REGION Network 26: Signal conditioning — Consolidate the auto or manual state request
   // ▀▀▀▀▀▀▀▀▀▀▀▀▀▀▀▀▀▀▀▀▀▀▀▀▀▀▀▀▀▀▀▀▀▀▀▀▀▀▀▀▀▀▀▀
   // Determine the valve state required by the automatic/manual mode selection:
   // 
   //    1.  If manual mode is active set wrkCtrlAutManOpCl to match the current manual 
   //      mode requested state (ctrl_Man_OpenClose)
   // 
   //    2.  If automatic mode is active set wrkCtrlAutManOpCl to match the current automatic 
   //      mode requested state (ctrl_Aut_OpenClose)
   // ▄▄▄▄▄▄▄▄▄▄▄▄▄▄▄▄▄▄▄▄▄▄▄▄▄▄▄▄▄▄▄▄▄▄▄▄▄▄▄▄▄▄▄▄
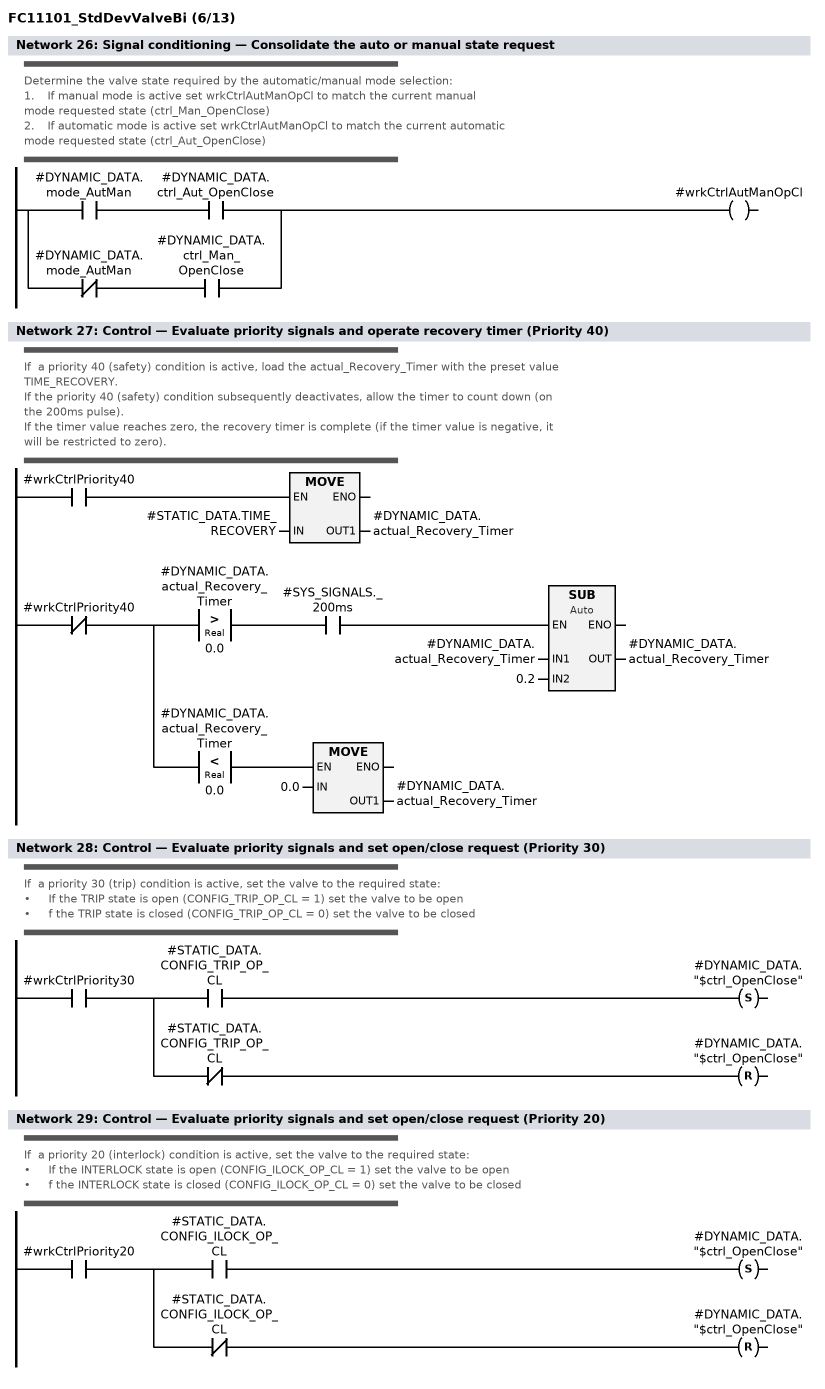
   RUNG wire#powerrail
      Contact( #DYNAMIC_DATA.mode_AutMan )
      Contact( #DYNAMIC_DATA.ctrl_Aut_OpenClose )
      wire#w1
      Coil( #wrkCtrlAutManOpCl )
   END_RUNG
   RUNG wire#powerrail
      I_Contact( #DYNAMIC_DATA.mode_AutMan )
      Contact( #DYNAMIC_DATA.ctrl_Man_OpenClose )
   END_RUNG wire#w1
   // the same network as SCL:
   #wrkCtrlAutManOpCl := (#DYNAMIC_DATA.mode_AutMan AND #DYNAMIC_DATA.ctrl_Aut_OpenClose) OR (NOT #DYNAMIC_DATA.mode_AutMan AND #DYNAMIC_DATA.ctrl_Man_OpenClose);
END_REGION

REGION Network 27: Control — Evaluate priority signals and operate recovery timer (Priority 40)
   // ▀▀▀▀▀▀▀▀▀▀▀▀▀▀▀▀▀▀▀▀▀▀▀▀▀▀▀▀▀▀▀▀▀▀▀▀▀▀▀▀▀▀▀▀
   // If  a priority 40 (safety) condition is active, load the actual_Recovery_Timer with the preset value 
   // TIME_RECOVERY.
   // 
   // If the priority 40 (safety) condition subsequently deactivates, allow the timer to count down (on 
   // the 200ms pulse).
   // 
   // If the timer value reaches zero, the recovery timer is complete (if the timer value is negative, it
   // will be restricted to zero).
   // ▄▄▄▄▄▄▄▄▄▄▄▄▄▄▄▄▄▄▄▄▄▄▄▄▄▄▄▄▄▄▄▄▄▄▄▄▄▄▄▄▄▄▄▄
   RUNG wire#powerrail
      Contact( #wrkCtrlPriority40 )
      Move(in := #STATIC_DATA.TIME_RECOVERY, out1 => #DYNAMIC_DATA.actual_Recovery_Timer)
   END_RUNG
   RUNG wire#powerrail
      I_Contact( #wrkCtrlPriority40 )
      wire#w1
      { S7_Templates := "SrcType := Real" } GT_Contact(in1 := #DYNAMIC_DATA.actual_Recovery_Timer, in2 := 0.0)
      Contact( #SYS_SIGNALS._200ms )
      Sub(in1 := #DYNAMIC_DATA.actual_Recovery_Timer, in2 := 0.2, out => #DYNAMIC_DATA.actual_Recovery_Timer)
   END_RUNG
   RUNG wire#w1
      { S7_Templates := "SrcType := Real" } LT_Contact(in1 := #DYNAMIC_DATA.actual_Recovery_Timer, in2 := 0.0)
      Move(in := 0.0, out1 => #DYNAMIC_DATA.actual_Recovery_Timer)
   END_RUNG
   // the same network as SCL:
   IF #wrkCtrlPriority40 THEN #DYNAMIC_DATA.actual_Recovery_Timer := #STATIC_DATA.TIME_RECOVERY; END_IF;
   IF NOT #wrkCtrlPriority40 AND (#DYNAMIC_DATA.actual_Recovery_Timer > 0.0) AND #SYS_SIGNALS._200ms THEN
       #DYNAMIC_DATA.actual_Recovery_Timer := #DYNAMIC_DATA.actual_Recovery_Timer - 0.2;
   END_IF;
   IF NOT #wrkCtrlPriority40 AND (#DYNAMIC_DATA.actual_Recovery_Timer < 0.0) THEN
       #DYNAMIC_DATA.actual_Recovery_Timer := 0.0;
   END_IF;
END_REGION

REGION Network 28: Control — Evaluate priority signals and set open/close request (Priority 30)
   // ▀▀▀▀▀▀▀▀▀▀▀▀▀▀▀▀▀▀▀▀▀▀▀▀▀▀▀▀▀▀▀▀▀▀▀▀▀▀▀▀▀▀▀▀
   // If  a priority 30 (trip) condition is active, set the valve to the required state:
   // 
   //    •   If the TRIP state is open (CONFIG_TRIP_OP_CL = 1) set the valve to be open
   // 
   //    •   f the TRIP state is closed (CONFIG_TRIP_OP_CL = 0) set the valve to be closed
   // ▄▄▄▄▄▄▄▄▄▄▄▄▄▄▄▄▄▄▄▄▄▄▄▄▄▄▄▄▄▄▄▄▄▄▄▄▄▄▄▄▄▄▄▄
   RUNG wire#powerrail
      Contact( #wrkCtrlPriority30 )
      wire#w1
      Contact( #STATIC_DATA.CONFIG_TRIP_OP_CL )
      S_Coil( #DYNAMIC_DATA."$ctrl_OpenClose" )
   END_RUNG
   RUNG wire#w1
      I_Contact( #STATIC_DATA.CONFIG_TRIP_OP_CL )
      R_Coil( #DYNAMIC_DATA."$ctrl_OpenClose" )
   END_RUNG
   // the same network as SCL:
   IF #wrkCtrlPriority30 AND #STATIC_DATA.CONFIG_TRIP_OP_CL THEN
       #DYNAMIC_DATA."$ctrl_OpenClose" := TRUE;
   END_IF;
   IF #wrkCtrlPriority30 AND NOT #STATIC_DATA.CONFIG_TRIP_OP_CL THEN
       #DYNAMIC_DATA."$ctrl_OpenClose" := FALSE;
   END_IF;
END_REGION

REGION Network 29: Control — Evaluate priority signals and set open/close request (Priority 20)
   // ▀▀▀▀▀▀▀▀▀▀▀▀▀▀▀▀▀▀▀▀▀▀▀▀▀▀▀▀▀▀▀▀▀▀▀▀▀▀▀▀▀▀▀▀
   // If  a priority 20 (interlock) condition is active, set the valve to the required state:
   // 
   //    •   If the INTERLOCK state is open (CONFIG_ILOCK_OP_CL = 1) set the valve to be open
   // 
   //    •   f the INTERLOCK state is closed (CONFIG_ILOCK_OP_CL = 0) set the valve to be closed
   // ▄▄▄▄▄▄▄▄▄▄▄▄▄▄▄▄▄▄▄▄▄▄▄▄▄▄▄▄▄▄▄▄▄▄▄▄▄▄▄▄▄▄▄▄
   RUNG wire#powerrail
      Contact( #wrkCtrlPriority20 )
      wire#w1
      Contact( #STATIC_DATA.CONFIG_ILOCK_OP_CL )
      S_Coil( #DYNAMIC_DATA."$ctrl_OpenClose" )
   END_RUNG
   RUNG wire#w1
      I_Contact( #STATIC_DATA.CONFIG_ILOCK_OP_CL )
      R_Coil( #DYNAMIC_DATA."$ctrl_OpenClose" )
   END_RUNG
   // the same network as SCL:
   IF #wrkCtrlPriority20 AND #STATIC_DATA.CONFIG_ILOCK_OP_CL THEN
       #DYNAMIC_DATA."$ctrl_OpenClose" := TRUE;
   END_IF;
   IF #wrkCtrlPriority20 AND NOT #STATIC_DATA.CONFIG_ILOCK_OP_CL THEN
       #DYNAMIC_DATA."$ctrl_OpenClose" := FALSE;
   END_IF;
END_REGION

REGION Network 30: Control — Evaluate priority signals and set open/close request (Priority 10)
   // ▀▀▀▀▀▀▀▀▀▀▀▀▀▀▀▀▀▀▀▀▀▀▀▀▀▀▀▀▀▀▀▀▀▀▀▀▀▀▀▀▀▀▀▀
   // If  a priority 10 (permissive) condition is active, set the valve to the required state:
   // 
   // 
   // PERMITTED STATE IS OPEN — CONDITIONS:
   // 
   //    •   If the Permitted state is open and Aut/Man request is for open, 
   //      set the valve to be open [Branch 1]
   // 
   //    •   If the Permitted state is open and Aut/Man request is for closed, and the current
   //      valve output matches this state (closed), set the valve to be closed (maintain the
   //      current state) [Branch 6]
   // 
   //    •   If the Permitted state is open and Aut/Man request is for closed, and the current
   //      valve output matches the open state, set the valve to be open (override the
   //      auto/man request [Branch 2]
   // 
   // PERMITTED STATE IS CLOSED — CONDITIONS:
   // 
   //    •   If the Permitted state is closed and Aut/Man request is for closed,
   //      set the valve to be  closed [Branch 4]
   // 
   //    •   If the Permitted state is closed and Aut/Man request is for open, and the current
   //      valve output matches this state (open), set the valve to be open (maintain the
   //      current state) [Branch 3]
   // 
   //    •   If the Permitted state is closed and Aut/Man request is for open, and the current
   //      valve output matches the closed state, set the valve to be closed (override the
   //      auto/man request [Branch 5]
   // ▄▄▄▄▄▄▄▄▄▄▄▄▄▄▄▄▄▄▄▄▄▄▄▄▄▄▄▄▄▄▄▄▄▄▄▄▄▄▄▄▄▄▄▄
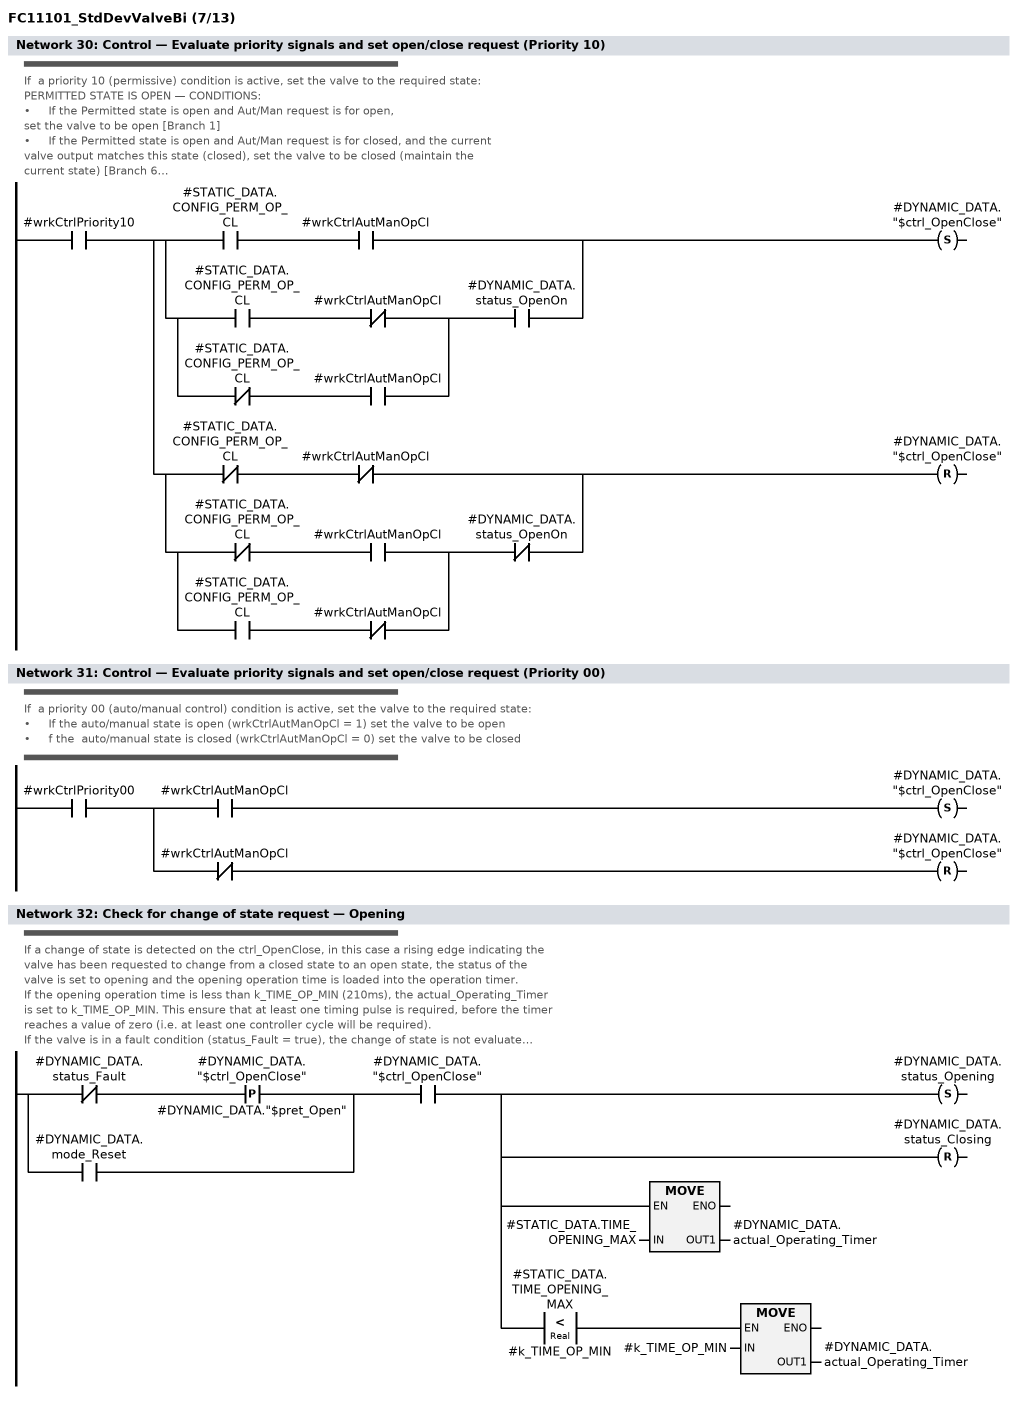
   RUNG wire#powerrail
      Contact( #wrkCtrlPriority10 )
      wire#w1
      Contact( #STATIC_DATA.CONFIG_PERM_OP_CL )
      Contact( #wrkCtrlAutManOpCl )
      wire#w2
      S_Coil( #DYNAMIC_DATA."$ctrl_OpenClose" )
   END_RUNG
   RUNG wire#w1
      Contact( #STATIC_DATA.CONFIG_PERM_OP_CL )
      I_Contact( #wrkCtrlAutManOpCl )
      wire#w3
      Contact( #DYNAMIC_DATA.status_OpenOn )
   END_RUNG wire#w2
   RUNG wire#w1
      I_Contact( #STATIC_DATA.CONFIG_PERM_OP_CL )
      Contact( #wrkCtrlAutManOpCl )
   END_RUNG wire#w3
   RUNG wire#w1
      I_Contact( #STATIC_DATA.CONFIG_PERM_OP_CL )
      I_Contact( #wrkCtrlAutManOpCl )
      wire#w4
      R_Coil( #DYNAMIC_DATA."$ctrl_OpenClose" )
   END_RUNG
   RUNG wire#w1
      I_Contact( #STATIC_DATA.CONFIG_PERM_OP_CL )
      Contact( #wrkCtrlAutManOpCl )
      wire#w5
      I_Contact( #DYNAMIC_DATA.status_OpenOn )
   END_RUNG wire#w4
   RUNG wire#w1
      Contact( #STATIC_DATA.CONFIG_PERM_OP_CL )
      I_Contact( #wrkCtrlAutManOpCl )
   END_RUNG wire#w5
   // the same network as SCL:
   IF #wrkCtrlPriority10 AND ((#STATIC_DATA.CONFIG_PERM_OP_CL AND #wrkCtrlAutManOpCl) OR (((#STATIC_DATA.CONFIG_PERM_OP_CL AND NOT #wrkCtrlAutManOpCl) OR (NOT #STATIC_DATA.CONFIG_PERM_OP_CL AND #wrkCtrlAutManOpCl)) AND #DYNAMIC_DATA.status_OpenOn)) THEN
       #DYNAMIC_DATA."$ctrl_OpenClose" := TRUE;
   END_IF;
   IF #wrkCtrlPriority10 AND ((NOT #STATIC_DATA.CONFIG_PERM_OP_CL AND NOT #wrkCtrlAutManOpCl) OR (((NOT #STATIC_DATA.CONFIG_PERM_OP_CL AND #wrkCtrlAutManOpCl) OR (#STATIC_DATA.CONFIG_PERM_OP_CL AND NOT #wrkCtrlAutManOpCl)) AND NOT #DYNAMIC_DATA.status_OpenOn)) THEN
       #DYNAMIC_DATA."$ctrl_OpenClose" := FALSE;
   END_IF;
END_REGION

REGION Network 31: Control — Evaluate priority signals and set open/close request (Priority 00)
   // ▀▀▀▀▀▀▀▀▀▀▀▀▀▀▀▀▀▀▀▀▀▀▀▀▀▀▀▀▀▀▀▀▀▀▀▀▀▀▀▀▀▀▀▀
   // If  a priority 00 (auto/manual control) condition is active, set the valve to the required state:
   // 
   //    •   If the auto/manual state is open (wrkCtrlAutManOpCl = 1) set the valve to be open
   // 
   //    •   f the  auto/manual state is closed (wrkCtrlAutManOpCl = 0) set the valve to be closed
   // ▄▄▄▄▄▄▄▄▄▄▄▄▄▄▄▄▄▄▄▄▄▄▄▄▄▄▄▄▄▄▄▄▄▄▄▄▄▄▄▄▄▄▄▄
   RUNG wire#powerrail
      Contact( #wrkCtrlPriority00 )
      wire#w1
      Contact( #wrkCtrlAutManOpCl )
      S_Coil( #DYNAMIC_DATA."$ctrl_OpenClose" )
   END_RUNG
   RUNG wire#w1
      I_Contact( #wrkCtrlAutManOpCl )
      R_Coil( #DYNAMIC_DATA."$ctrl_OpenClose" )
   END_RUNG
   // the same network as SCL:
   IF #wrkCtrlPriority00 AND #wrkCtrlAutManOpCl THEN #DYNAMIC_DATA."$ctrl_OpenClose" := TRUE; END_IF;
   IF #wrkCtrlPriority00 AND NOT #wrkCtrlAutManOpCl THEN #DYNAMIC_DATA."$ctrl_OpenClose" := FALSE; END_IF;
END_REGION

REGION Network 32: Check for change of state request — Opening
   // ▀▀▀▀▀▀▀▀▀▀▀▀▀▀▀▀▀▀▀▀▀▀▀▀▀▀▀▀▀▀▀▀▀▀▀▀▀▀▀▀▀▀▀▀
   // If a change of state is detected on the ctrl_OpenClose, in this case a rising edge indicating the
   // valve has been requested to change from a closed state to an open state, the status of the
   // valve is set to opening and the opening operation time is loaded into the operation timer.
   // 
   // If the opening operation time is less than k_TIME_OP_MIN (210ms), the actual_Operating_Timer 
   // is set to k_TIME_OP_MIN. This ensure that at least one timing pulse is required, before the timer 
   // reaches a value of zero (i.e. at least one controller cycle will be required).
   // 
   // If the valve is in a fault condition (status_Fault = true), the change of state is not evaluated
   // until the fault condition has cleared
   // 
   // Note: the timer is also triggered if the Reset signal is received and the valve is requested open.
   // ▄▄▄▄▄▄▄▄▄▄▄▄▄▄▄▄▄▄▄▄▄▄▄▄▄▄▄▄▄▄▄▄▄▄▄▄▄▄▄▄▄▄▄▄
   RUNG wire#powerrail
      I_Contact( #DYNAMIC_DATA.status_Fault )
      P_Contact(operand := #DYNAMIC_DATA."$ctrl_OpenClose", bit := #DYNAMIC_DATA."$pret_Open")
      wire#w1
      Contact( #DYNAMIC_DATA."$ctrl_OpenClose" )
      wire#w2
      S_Coil( #DYNAMIC_DATA.status_Opening )
   END_RUNG
   RUNG wire#powerrail
      Contact( #DYNAMIC_DATA.mode_Reset )
   END_RUNG wire#w1
   RUNG wire#w2
      R_Coil( #DYNAMIC_DATA.status_Closing )
   END_RUNG
   RUNG wire#w2
      Move(in := #STATIC_DATA.TIME_OPENING_MAX, out1 => #DYNAMIC_DATA.actual_Operating_Timer)
   END_RUNG
   RUNG wire#w2
      { S7_Templates := "SrcType := Real" } LT_Contact(in1 := #STATIC_DATA.TIME_OPENING_MAX, in2 := #k_TIME_OP_MIN)
      Move(in := #k_TIME_OP_MIN, out1 => #DYNAMIC_DATA.actual_Operating_Timer)
   END_RUNG
   // the same network as SCL:
   #_w1 := NOT #DYNAMIC_DATA.status_Fault AND #DYNAMIC_DATA."$ctrl_OpenClose" AND NOT #DYNAMIC_DATA."$pret_Open";   // rising edge of #DYNAMIC_DATA."$ctrl_OpenClose"
   #DYNAMIC_DATA."$pret_Open" := #DYNAMIC_DATA."$ctrl_OpenClose";
   #_w2 := (#_w1 OR #DYNAMIC_DATA.mode_Reset) AND #DYNAMIC_DATA."$ctrl_OpenClose";
   IF #_w2 THEN
       #DYNAMIC_DATA.status_Opening := TRUE;
       #DYNAMIC_DATA.status_Closing := FALSE;
       #DYNAMIC_DATA.actual_Operating_Timer := #STATIC_DATA.TIME_OPENING_MAX;
   END_IF;
   IF #_w2 AND (#STATIC_DATA.TIME_OPENING_MAX < #k_TIME_OP_MIN) THEN
       #DYNAMIC_DATA.actual_Operating_Timer := #k_TIME_OP_MIN;
   END_IF;
END_REGION

REGION Network 33: Check for change of state request — Closing
   // ▀▀▀▀▀▀▀▀▀▀▀▀▀▀▀▀▀▀▀▀▀▀▀▀▀▀▀▀▀▀▀▀▀▀▀▀▀▀▀▀▀▀▀▀
   // If a change of state is detected on the ctrl_OpenClose, in this case a falling edge indicating the
   // valve has been requested to change from an open state to a closed state, the status of the
   // valve is set to closing and the closing operation time is loaded into the operation timer.
   // 
   // If the closing operation time is less than k_TIME_OP_MIN (210ms), the actual_Operating_Timer 
   // is set to k_TIME_OP_MIN. This ensure that at least one timing pulse is required, before the timer 
   // reaches a value of zero (i.e. at least one controller cycle will be required).
   // 
   // If the valve is in a fault condition (status_Fault = true), the change of state is not evaluated
   // until the fault condition has cleared
   // 
   // Note: the timer is also triggered if the Reset signal is received and the valve is requested closed.
   // ▄▄▄▄▄▄▄▄▄▄▄▄▄▄▄▄▄▄▄▄▄▄▄▄▄▄▄▄▄▄▄▄▄▄▄▄▄▄▄▄▄▄▄▄
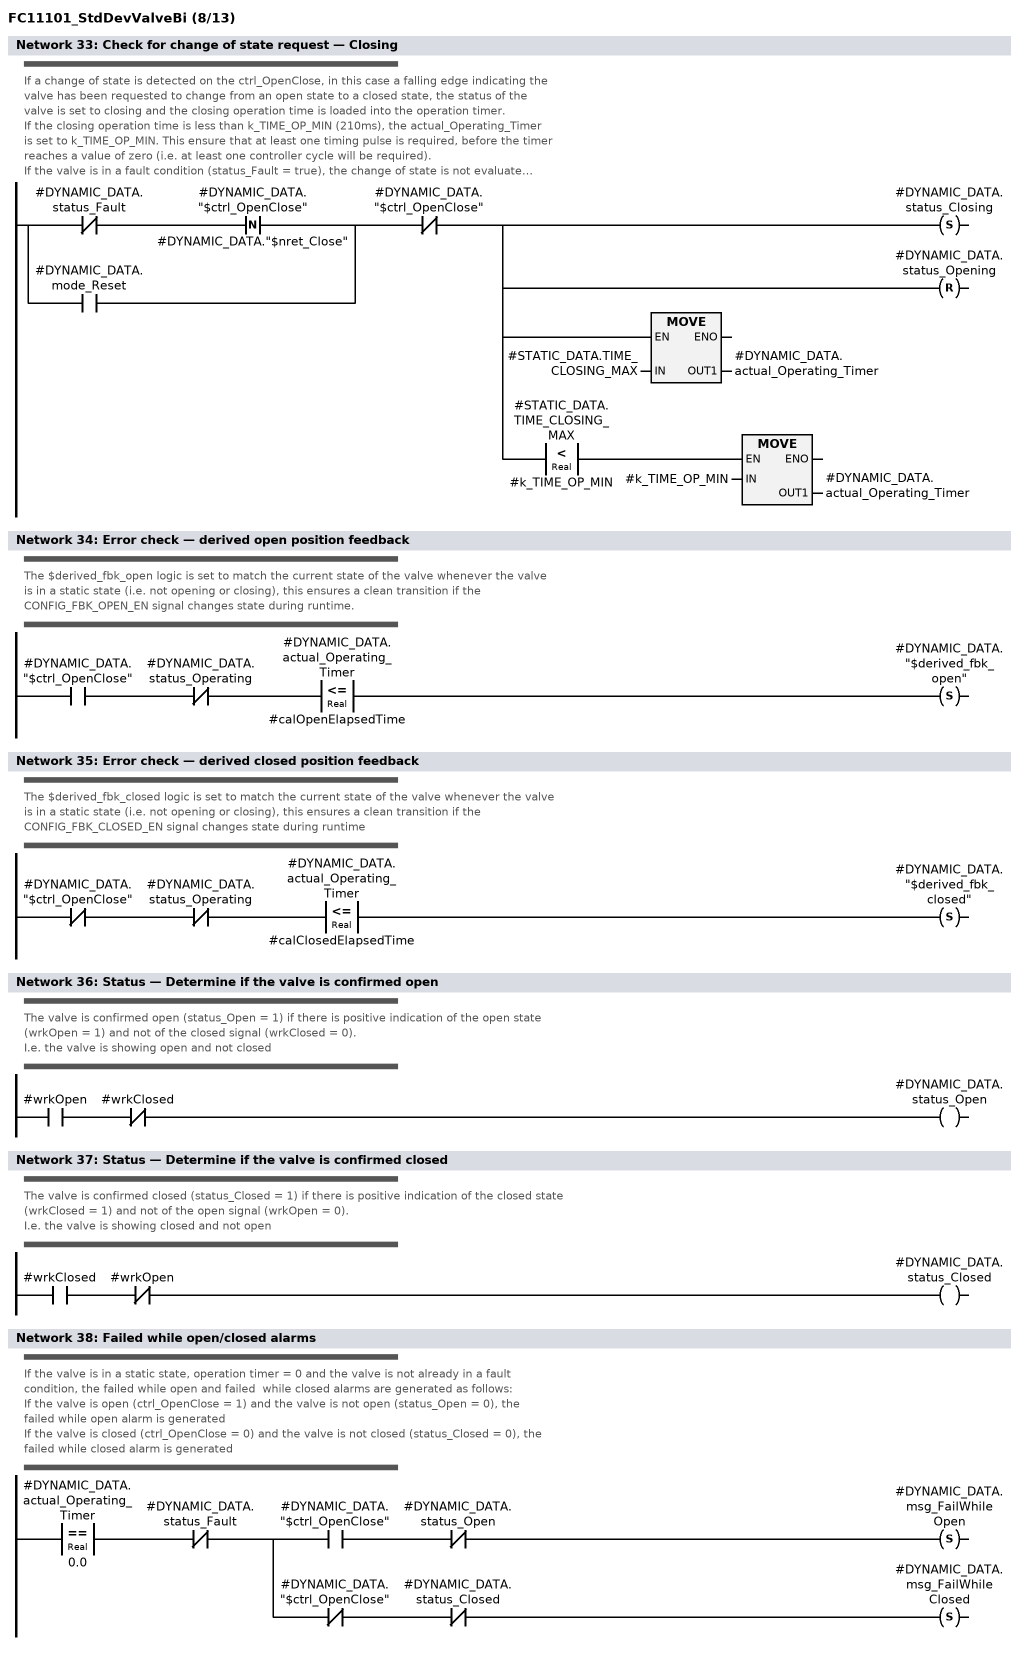
   RUNG wire#powerrail
      I_Contact( #DYNAMIC_DATA.status_Fault )
      N_Contact(operand := #DYNAMIC_DATA."$ctrl_OpenClose", bit := #DYNAMIC_DATA."$nret_Close")
      wire#w1
      I_Contact( #DYNAMIC_DATA."$ctrl_OpenClose" )
      wire#w2
      S_Coil( #DYNAMIC_DATA.status_Closing )
   END_RUNG
   RUNG wire#powerrail
      Contact( #DYNAMIC_DATA.mode_Reset )
   END_RUNG wire#w1
   RUNG wire#w2
      R_Coil( #DYNAMIC_DATA.status_Opening )
   END_RUNG
   RUNG wire#w2
      Move(in := #STATIC_DATA.TIME_CLOSING_MAX, out1 => #DYNAMIC_DATA.actual_Operating_Timer)
   END_RUNG
   RUNG wire#w2
      { S7_Templates := "SrcType := Real" } LT_Contact(in1 := #STATIC_DATA.TIME_CLOSING_MAX, in2 := #k_TIME_OP_MIN)
      Move(in := #k_TIME_OP_MIN, out1 => #DYNAMIC_DATA.actual_Operating_Timer)
   END_RUNG
   // the same network as SCL:
   #_w1 := NOT #DYNAMIC_DATA.status_Fault AND NOT #DYNAMIC_DATA."$ctrl_OpenClose" AND #DYNAMIC_DATA."$nret_Close";   // falling edge of #DYNAMIC_DATA."$ctrl_OpenClose"
   #DYNAMIC_DATA."$nret_Close" := #DYNAMIC_DATA."$ctrl_OpenClose";
   #_w2 := (#_w1 OR #DYNAMIC_DATA.mode_Reset) AND NOT #DYNAMIC_DATA."$ctrl_OpenClose";
   IF #_w2 THEN
       #DYNAMIC_DATA.status_Closing := TRUE;
       #DYNAMIC_DATA.status_Opening := FALSE;
       #DYNAMIC_DATA.actual_Operating_Timer := #STATIC_DATA.TIME_CLOSING_MAX;
   END_IF;
   IF #_w2 AND (#STATIC_DATA.TIME_CLOSING_MAX < #k_TIME_OP_MIN) THEN
       #DYNAMIC_DATA.actual_Operating_Timer := #k_TIME_OP_MIN;
   END_IF;
END_REGION

REGION Network 34: Error check — derived open position feedback
   // ▀▀▀▀▀▀▀▀▀▀▀▀▀▀▀▀▀▀▀▀▀▀▀▀▀▀▀▀▀▀▀▀▀▀▀▀▀▀▀▀▀▀▀▀
   // The $derived_fbk_open logic is set to match the current state of the valve whenever the valve
   // is in a static state (i.e. not opening or closing), this ensures a clean transition if the 
   // CONFIG_FBK_OPEN_EN signal changes state during runtime.
   // ▄▄▄▄▄▄▄▄▄▄▄▄▄▄▄▄▄▄▄▄▄▄▄▄▄▄▄▄▄▄▄▄▄▄▄▄▄▄▄▄▄▄▄▄
   RUNG wire#powerrail
      Contact( #DYNAMIC_DATA."$ctrl_OpenClose" )
      I_Contact( #DYNAMIC_DATA.status_Operating )
      { S7_Templates := "SrcType := Real" } LE_Contact(in1 := #DYNAMIC_DATA.actual_Operating_Timer, in2 := #calOpenElapsedTime)
      S_Coil( #DYNAMIC_DATA."$derived_fbk_open" )
   END_RUNG
   // the same network as SCL:
   IF #DYNAMIC_DATA."$ctrl_OpenClose" AND NOT #DYNAMIC_DATA.status_Operating AND (#DYNAMIC_DATA.actual_Operating_Timer <= #calOpenElapsedTime) THEN
       #DYNAMIC_DATA."$derived_fbk_open" := TRUE;
   END_IF;
END_REGION

REGION Network 35: Error check — derived closed position feedback
   // ▀▀▀▀▀▀▀▀▀▀▀▀▀▀▀▀▀▀▀▀▀▀▀▀▀▀▀▀▀▀▀▀▀▀▀▀▀▀▀▀▀▀▀▀
   // The $derived_fbk_closed logic is set to match the current state of the valve whenever the valve
   // is in a static state (i.e. not opening or closing), this ensures a clean transition if the 
   // CONFIG_FBK_CLOSED_EN signal changes state during runtime
   // ▄▄▄▄▄▄▄▄▄▄▄▄▄▄▄▄▄▄▄▄▄▄▄▄▄▄▄▄▄▄▄▄▄▄▄▄▄▄▄▄▄▄▄▄
   RUNG wire#powerrail
      I_Contact( #DYNAMIC_DATA."$ctrl_OpenClose" )
      I_Contact( #DYNAMIC_DATA.status_Operating )
      { S7_Templates := "SrcType := Real" } LE_Contact(in1 := #DYNAMIC_DATA.actual_Operating_Timer, in2 := #calClosedElapsedTime)
      S_Coil( #DYNAMIC_DATA."$derived_fbk_closed" )
   END_RUNG
   // the same network as SCL:
   IF NOT #DYNAMIC_DATA."$ctrl_OpenClose" AND NOT #DYNAMIC_DATA.status_Operating AND (#DYNAMIC_DATA.actual_Operating_Timer <= #calClosedElapsedTime) THEN
       #DYNAMIC_DATA."$derived_fbk_closed" := TRUE;
   END_IF;
END_REGION

REGION Network 36: Status — Determine if the valve is confirmed open
   // ▀▀▀▀▀▀▀▀▀▀▀▀▀▀▀▀▀▀▀▀▀▀▀▀▀▀▀▀▀▀▀▀▀▀▀▀▀▀▀▀▀▀▀▀
   // The valve is confirmed open (status_Open = 1) if there is positive indication of the open state 
   // (wrkOpen = 1) and not of the closed signal (wrkClosed = 0). 
   // 
   // I.e. the valve is showing open and not closed
   // ▄▄▄▄▄▄▄▄▄▄▄▄▄▄▄▄▄▄▄▄▄▄▄▄▄▄▄▄▄▄▄▄▄▄▄▄▄▄▄▄▄▄▄▄
   RUNG wire#powerrail
      Contact( #wrkOpen )
      I_Contact( #wrkClosed )
      Coil( #DYNAMIC_DATA.status_Open )
   END_RUNG
   // the same network as SCL:
   #DYNAMIC_DATA.status_Open := #wrkOpen AND NOT #wrkClosed;
END_REGION

REGION Network 37: Status — Determine if the valve is confirmed closed
   // ▀▀▀▀▀▀▀▀▀▀▀▀▀▀▀▀▀▀▀▀▀▀▀▀▀▀▀▀▀▀▀▀▀▀▀▀▀▀▀▀▀▀▀▀
   // The valve is confirmed closed (status_Closed = 1) if there is positive indication of the closed state 
   // (wrkClosed = 1) and not of the open signal (wrkOpen = 0). 
   // 
   // I.e. the valve is showing closed and not open
   // ▄▄▄▄▄▄▄▄▄▄▄▄▄▄▄▄▄▄▄▄▄▄▄▄▄▄▄▄▄▄▄▄▄▄▄▄▄▄▄▄▄▄▄▄
   RUNG wire#powerrail
      Contact( #wrkClosed )
      I_Contact( #wrkOpen )
      Coil( #DYNAMIC_DATA.status_Closed )
   END_RUNG
   // the same network as SCL:
   #DYNAMIC_DATA.status_Closed := #wrkClosed AND NOT #wrkOpen;
END_REGION

REGION Network 38: Failed while open/closed alarms
   // ▀▀▀▀▀▀▀▀▀▀▀▀▀▀▀▀▀▀▀▀▀▀▀▀▀▀▀▀▀▀▀▀▀▀▀▀▀▀▀▀▀▀▀▀
   // If the valve is in a static state, operation timer = 0 and the valve is not already in a fault
   // condition, the failed while open and failed  while closed alarms are generated as follows:
   // 
   // If the valve is open (ctrl_OpenClose = 1) and the valve is not open (status_Open = 0), the 
   // failed while open alarm is generated
   // 
   // If the valve is closed (ctrl_OpenClose = 0) and the valve is not closed (status_Closed = 0), the 
   // failed while closed alarm is generated
   // ▄▄▄▄▄▄▄▄▄▄▄▄▄▄▄▄▄▄▄▄▄▄▄▄▄▄▄▄▄▄▄▄▄▄▄▄▄▄▄▄▄▄▄▄
   RUNG wire#powerrail
      { S7_Templates := "SrcType := Real" } EQ_Contact(in1 := #DYNAMIC_DATA.actual_Operating_Timer, in2 := 0.0)
      I_Contact( #DYNAMIC_DATA.status_Fault )
      wire#w1
      Contact( #DYNAMIC_DATA."$ctrl_OpenClose" )
      I_Contact( #DYNAMIC_DATA.status_Open )
      S_Coil( #DYNAMIC_DATA.msg_FailWhileOpen )
   END_RUNG
   RUNG wire#w1
      I_Contact( #DYNAMIC_DATA."$ctrl_OpenClose" )
      I_Contact( #DYNAMIC_DATA.status_Closed )
      S_Coil( #DYNAMIC_DATA.msg_FailWhileClosed )
   END_RUNG
   // the same network as SCL:
   #_w1 := (#DYNAMIC_DATA.actual_Operating_Timer = 0.0) AND NOT #DYNAMIC_DATA.status_Fault;
   IF #_w1 AND #DYNAMIC_DATA."$ctrl_OpenClose" AND NOT #DYNAMIC_DATA.status_Open THEN
       #DYNAMIC_DATA.msg_FailWhileOpen := TRUE;
   END_IF;
   IF #_w1 AND NOT #DYNAMIC_DATA."$ctrl_OpenClose" AND NOT #DYNAMIC_DATA.status_Closed THEN
       #DYNAMIC_DATA.msg_FailWhileClosed := TRUE;
   END_IF;
END_REGION

REGION Network 39: Operation timer and Failed to open/close alarms
   // ▀▀▀▀▀▀▀▀▀▀▀▀▀▀▀▀▀▀▀▀▀▀▀▀▀▀▀▀▀▀▀▀▀▀▀▀▀▀▀▀▀▀▀▀
   // If the valve is opening or closing, decrement the current operation timer value on each 200ms
   // pulse.
   // 
   // If the timer reaches zero, and the valve is opening, generate the failed to open alarm.
   // 
   // If the timer reaches zero, and the valve is closing, generate the failed to close alarm
   // ▄▄▄▄▄▄▄▄▄▄▄▄▄▄▄▄▄▄▄▄▄▄▄▄▄▄▄▄▄▄▄▄▄▄▄▄▄▄▄▄▄▄▄▄
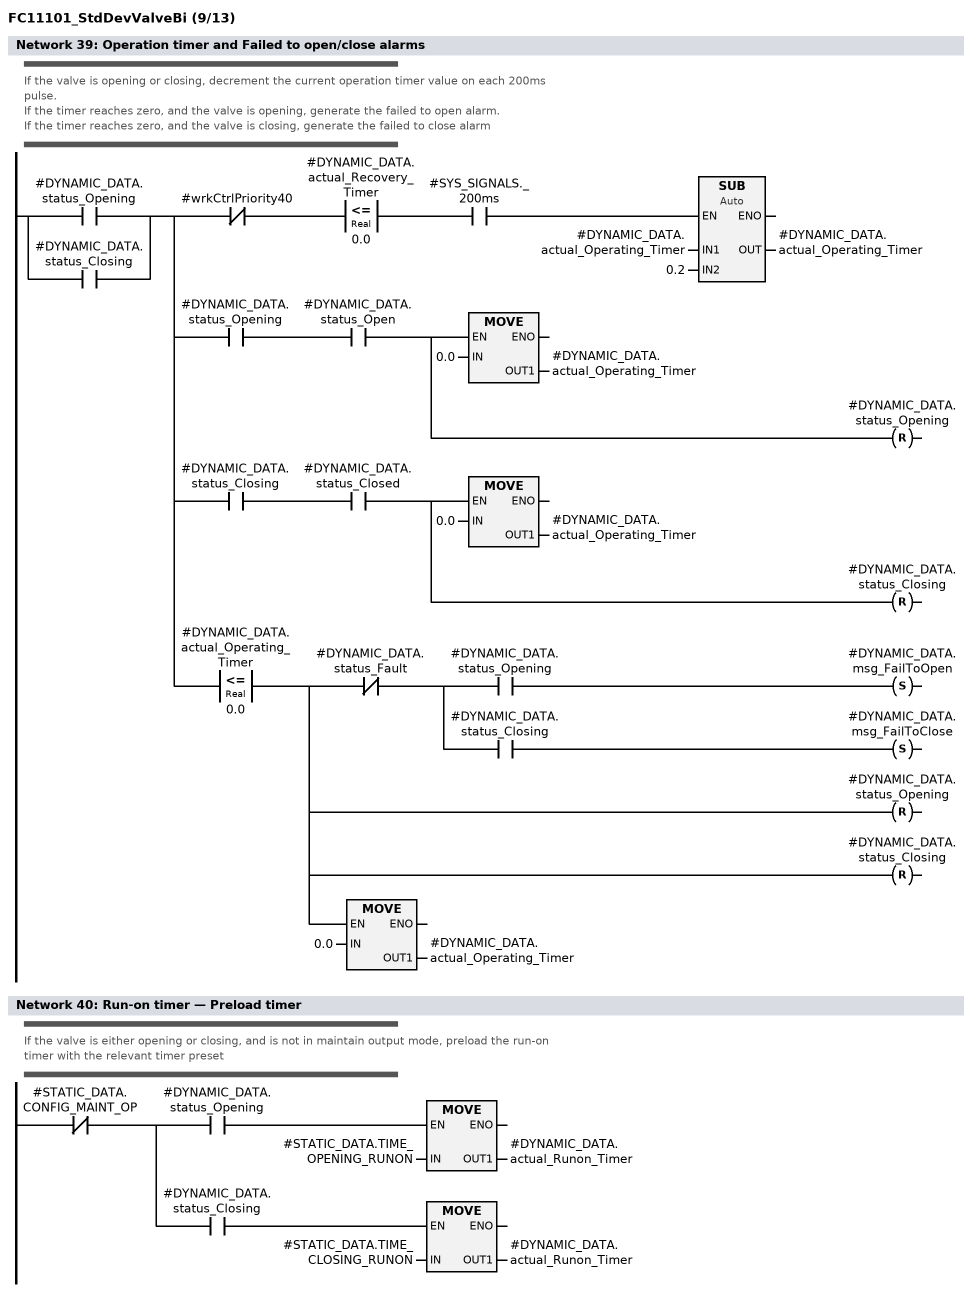
   RUNG wire#powerrail
      Contact( #DYNAMIC_DATA.status_Opening )
      wire#w1
      I_Contact( #wrkCtrlPriority40 )
      { S7_Templates := "SrcType := Real" } LE_Contact(in1 := #DYNAMIC_DATA.actual_Recovery_Timer, in2 := 0.0)
      Contact( #SYS_SIGNALS._200ms )
      Sub(in1 := #DYNAMIC_DATA.actual_Operating_Timer, in2 := 0.2, out => #DYNAMIC_DATA.actual_Operating_Timer)
   END_RUNG
   RUNG wire#powerrail
      Contact( #DYNAMIC_DATA.status_Closing )
   END_RUNG wire#w1
   RUNG wire#w1
      Contact( #DYNAMIC_DATA.status_Opening )
      Contact( #DYNAMIC_DATA.status_Open )
      wire#w2
      Move(in := 0.0, out1 => #DYNAMIC_DATA.actual_Operating_Timer)
   END_RUNG
   RUNG wire#w2
      R_Coil( #DYNAMIC_DATA.status_Opening )
   END_RUNG
   RUNG wire#w1
      Contact( #DYNAMIC_DATA.status_Closing )
      Contact( #DYNAMIC_DATA.status_Closed )
      wire#w3
      Move(in := 0.0, out1 => #DYNAMIC_DATA.actual_Operating_Timer)
   END_RUNG
   RUNG wire#w3
      R_Coil( #DYNAMIC_DATA.status_Closing )
   END_RUNG
   RUNG wire#w1
      { S7_Templates := "SrcType := Real" } LE_Contact(in1 := #DYNAMIC_DATA.actual_Operating_Timer, in2 := 0.0)
      wire#w4
      I_Contact( #DYNAMIC_DATA.status_Fault )
      wire#w5
      Contact( #DYNAMIC_DATA.status_Opening )
      S_Coil( #DYNAMIC_DATA.msg_FailToOpen )
   END_RUNG
   RUNG wire#w5
      Contact( #DYNAMIC_DATA.status_Closing )
      S_Coil( #DYNAMIC_DATA.msg_FailToClose )
   END_RUNG
   RUNG wire#w4
      R_Coil( #DYNAMIC_DATA.status_Opening )
   END_RUNG
   RUNG wire#w4
      R_Coil( #DYNAMIC_DATA.status_Closing )
   END_RUNG
   RUNG wire#w4
      Move(in := 0.0, out1 => #DYNAMIC_DATA.actual_Operating_Timer)
   END_RUNG
   // the same network as SCL:
   #_w1 := #DYNAMIC_DATA.status_Opening OR #DYNAMIC_DATA.status_Closing;
   IF #_w1 AND NOT #wrkCtrlPriority40 AND (#DYNAMIC_DATA.actual_Recovery_Timer <= 0.0) AND #SYS_SIGNALS._200ms THEN
       #DYNAMIC_DATA.actual_Operating_Timer := #DYNAMIC_DATA.actual_Operating_Timer - 0.2;
   END_IF;
   IF #_w1 AND #DYNAMIC_DATA.status_Opening AND #DYNAMIC_DATA.status_Open THEN
       #DYNAMIC_DATA.actual_Operating_Timer := 0.0;
       #DYNAMIC_DATA.status_Opening := FALSE;
   END_IF;
   IF #_w1 AND #DYNAMIC_DATA.status_Closing AND #DYNAMIC_DATA.status_Closed THEN
       #DYNAMIC_DATA.actual_Operating_Timer := 0.0;
       #DYNAMIC_DATA.status_Closing := FALSE;
   END_IF;
   #_w2 := #_w1 AND (#DYNAMIC_DATA.actual_Operating_Timer <= 0.0);
   #_w3 := #_w2 AND NOT #DYNAMIC_DATA.status_Fault;
   IF #_w3 AND #DYNAMIC_DATA.status_Opening THEN #DYNAMIC_DATA.msg_FailToOpen := TRUE; END_IF;
   IF #_w3 AND #DYNAMIC_DATA.status_Closing THEN #DYNAMIC_DATA.msg_FailToClose := TRUE; END_IF;
   IF #_w2 THEN
       #DYNAMIC_DATA.status_Opening := FALSE;
       #DYNAMIC_DATA.status_Closing := FALSE;
       #DYNAMIC_DATA.actual_Operating_Timer := 0.0;
   END_IF;
END_REGION

REGION Network 40: Run-on timer — Preload timer
   // ▀▀▀▀▀▀▀▀▀▀▀▀▀▀▀▀▀▀▀▀▀▀▀▀▀▀▀▀▀▀▀▀▀▀▀▀▀▀▀▀▀▀▀▀
   // If the valve is either opening or closing, and is not in maintain output mode, preload the run-on
   // timer with the relevant timer preset
   // ▄▄▄▄▄▄▄▄▄▄▄▄▄▄▄▄▄▄▄▄▄▄▄▄▄▄▄▄▄▄▄▄▄▄▄▄▄▄▄▄▄▄▄▄
   RUNG wire#powerrail
      I_Contact( #STATIC_DATA.CONFIG_MAINT_OP )
      wire#w1
      Contact( #DYNAMIC_DATA.status_Opening )
      Move(in := #STATIC_DATA.TIME_OPENING_RUNON, out1 => #DYNAMIC_DATA.actual_Runon_Timer)
   END_RUNG
   RUNG wire#w1
      Contact( #DYNAMIC_DATA.status_Closing )
      Move(in := #STATIC_DATA.TIME_CLOSING_RUNON, out1 => #DYNAMIC_DATA.actual_Runon_Timer)
   END_RUNG
   // the same network as SCL:
   #_w1 := NOT #STATIC_DATA.CONFIG_MAINT_OP;
   IF #_w1 AND #DYNAMIC_DATA.status_Opening THEN
       #DYNAMIC_DATA.actual_Runon_Timer := #STATIC_DATA.TIME_OPENING_RUNON;
   END_IF;
   IF #_w1 AND #DYNAMIC_DATA.status_Closing THEN
       #DYNAMIC_DATA.actual_Runon_Timer := #STATIC_DATA.TIME_CLOSING_RUNON;
   END_IF;
END_REGION

REGION Network 41: Run-on timer — Count down
   // ▀▀▀▀▀▀▀▀▀▀▀▀▀▀▀▀▀▀▀▀▀▀▀▀▀▀▀▀▀▀▀▀▀▀▀▀▀▀▀▀▀▀▀▀
   // If the valve is either closed or open, is not in fault and is not configured to maintain outputs, the 
   // run-on timer will count down from its preset value.
   // 
   // If an emergency stop is activated whilst the run-on timer is active, it will pause at the last 
   // elapsed value.
   // 
   // If a fault condition is active or if the valve is configured to maintain outputs, the run-on timer is
   // set to zero.
   // ▄▄▄▄▄▄▄▄▄▄▄▄▄▄▄▄▄▄▄▄▄▄▄▄▄▄▄▄▄▄▄▄▄▄▄▄▄▄▄▄▄▄▄▄
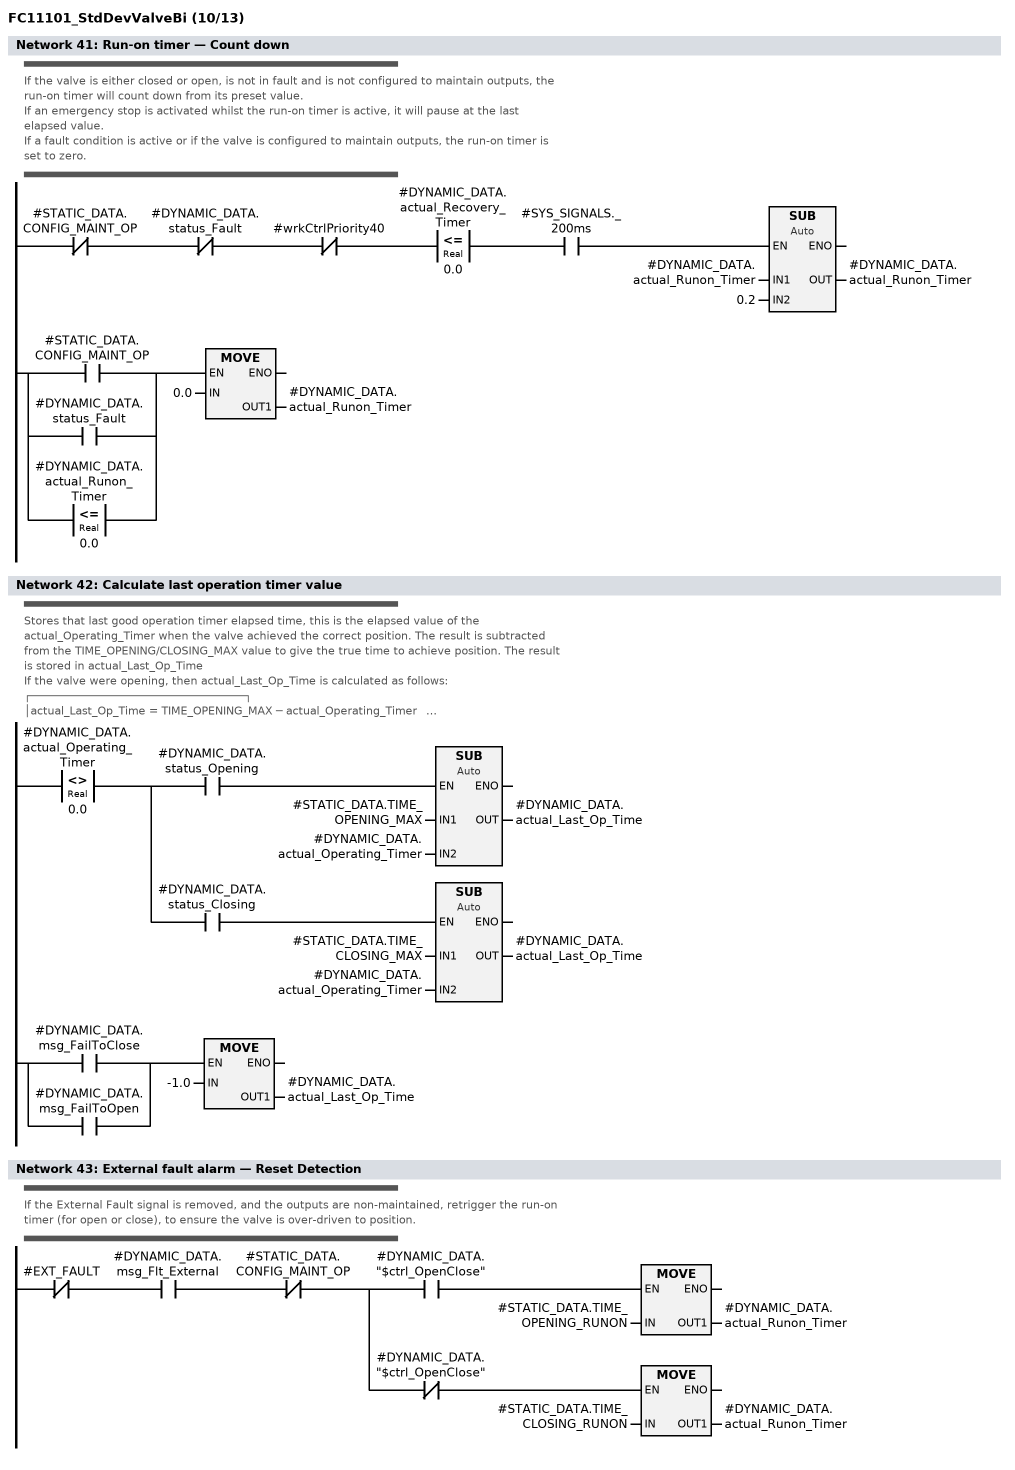
   RUNG wire#powerrail
      I_Contact( #STATIC_DATA.CONFIG_MAINT_OP )
      I_Contact( #DYNAMIC_DATA.status_Fault )
      I_Contact( #wrkCtrlPriority40 )
      { S7_Templates := "SrcType := Real" } LE_Contact(in1 := #DYNAMIC_DATA.actual_Recovery_Timer, in2 := 0.0)
      Contact( #SYS_SIGNALS._200ms )
      Sub(in1 := #DYNAMIC_DATA.actual_Runon_Timer, in2 := 0.2, out => #DYNAMIC_DATA.actual_Runon_Timer)
   END_RUNG
   RUNG wire#powerrail
      Contact( #STATIC_DATA.CONFIG_MAINT_OP )
      wire#w1
      Move(in := 0.0, out1 => #DYNAMIC_DATA.actual_Runon_Timer)
   END_RUNG
   RUNG wire#powerrail
      Contact( #DYNAMIC_DATA.status_Fault )
   END_RUNG wire#w1
   RUNG wire#powerrail
      { S7_Templates := "SrcType := Real" } LE_Contact(in1 := #DYNAMIC_DATA.actual_Runon_Timer, in2 := 0.0)
   END_RUNG wire#w1
   // the same network as SCL:
   IF NOT #STATIC_DATA.CONFIG_MAINT_OP AND NOT #DYNAMIC_DATA.status_Fault AND NOT #wrkCtrlPriority40 AND (#DYNAMIC_DATA.actual_Recovery_Timer <= 0.0) AND #SYS_SIGNALS._200ms THEN
       #DYNAMIC_DATA.actual_Runon_Timer := #DYNAMIC_DATA.actual_Runon_Timer - 0.2;
   END_IF;
   IF #STATIC_DATA.CONFIG_MAINT_OP OR #DYNAMIC_DATA.status_Fault OR (#DYNAMIC_DATA.actual_Runon_Timer <= 0.0) THEN
       #DYNAMIC_DATA.actual_Runon_Timer := 0.0;
   END_IF;
END_REGION

REGION Network 42: Calculate last operation timer value
   // ▀▀▀▀▀▀▀▀▀▀▀▀▀▀▀▀▀▀▀▀▀▀▀▀▀▀▀▀▀▀▀▀▀▀▀▀▀▀▀▀▀▀▀▀
   // Stores that last good operation timer elapsed time, this is the elapsed value of the 
   // actual_Operating_Timer when the valve achieved the correct position. The result is subtracted
   // from the TIME_OPENING/CLOSING_MAX value to give the true time to achieve position. The result
   // is stored in actual_Last_Op_Time
   // 
   // If the valve were opening, then actual_Last_Op_Time is calculated as follows:
   // 
   // ┌─────────────────────────────────┐
   // │actual_Last_Op_Time = TIME_OPENING_MAX ─ actual_Operating_Timer   │
   // └─────────────────────────────────┘
   // 
   // If the valve were closing, then actual_Last_Op_Time is calculated as follows:
   // 
   // ┌─────────────────────────────────┐
   // │actual_Last_Op_Time = TIME_CLOSING_MAX ─ actual_Operating_Timer   │
   // └─────────────────────────────────┘
   // 
   // If the valve either fails to open or fails to close,  then actual_Last_Op_Time is set to -1.0 to 
   // indicate a fault state.
   // ▄▄▄▄▄▄▄▄▄▄▄▄▄▄▄▄▄▄▄▄▄▄▄▄▄▄▄▄▄▄▄▄▄▄▄▄▄▄▄▄▄▄▄▄
   RUNG wire#powerrail
      { S7_Templates := "SrcType := Real" } NE_Contact(in1 := #DYNAMIC_DATA.actual_Operating_Timer, in2 := 0.0)
      wire#w1
      Contact( #DYNAMIC_DATA.status_Opening )
      Sub(in1 := #STATIC_DATA.TIME_OPENING_MAX, in2 := #DYNAMIC_DATA.actual_Operating_Timer, out => #DYNAMIC_DATA.actual_Last_Op_Time)
   END_RUNG
   RUNG wire#w1
      Contact( #DYNAMIC_DATA.status_Closing )
      Sub(in1 := #STATIC_DATA.TIME_CLOSING_MAX, in2 := #DYNAMIC_DATA.actual_Operating_Timer, out => #DYNAMIC_DATA.actual_Last_Op_Time)
   END_RUNG
   RUNG wire#powerrail
      Contact( #DYNAMIC_DATA.msg_FailToClose )
      wire#w2
      Move(in := -1.0, out1 => #DYNAMIC_DATA.actual_Last_Op_Time)
   END_RUNG
   RUNG wire#powerrail
      Contact( #DYNAMIC_DATA.msg_FailToOpen )
   END_RUNG wire#w2
   // the same network as SCL:
   #_w1 := #DYNAMIC_DATA.actual_Operating_Timer <> 0.0;
   IF #_w1 AND #DYNAMIC_DATA.status_Opening THEN
       #DYNAMIC_DATA.actual_Last_Op_Time := #STATIC_DATA.TIME_OPENING_MAX - #DYNAMIC_DATA.actual_Operating_Timer;
   END_IF;
   IF #_w1 AND #DYNAMIC_DATA.status_Closing THEN
       #DYNAMIC_DATA.actual_Last_Op_Time := #STATIC_DATA.TIME_CLOSING_MAX - #DYNAMIC_DATA.actual_Operating_Timer;
   END_IF;
   IF #DYNAMIC_DATA.msg_FailToClose OR #DYNAMIC_DATA.msg_FailToOpen THEN
       #DYNAMIC_DATA.actual_Last_Op_Time := -1.0;
   END_IF;
END_REGION

REGION Network 43: External fault alarm — Reset Detection
   // ▀▀▀▀▀▀▀▀▀▀▀▀▀▀▀▀▀▀▀▀▀▀▀▀▀▀▀▀▀▀▀▀▀▀▀▀▀▀▀▀▀▀▀▀
   // If the External Fault signal is removed, and the outputs are non-maintained, retrigger the run-on 
   // timer (for open or close), to ensure the valve is over-driven to position.
   // ▄▄▄▄▄▄▄▄▄▄▄▄▄▄▄▄▄▄▄▄▄▄▄▄▄▄▄▄▄▄▄▄▄▄▄▄▄▄▄▄▄▄▄▄
   RUNG wire#powerrail
      I_Contact( #EXT_FAULT )
      Contact( #DYNAMIC_DATA.msg_Flt_External )
      I_Contact( #STATIC_DATA.CONFIG_MAINT_OP )
      wire#w1
      Contact( #DYNAMIC_DATA."$ctrl_OpenClose" )
      Move(in := #STATIC_DATA.TIME_OPENING_RUNON, out1 => #DYNAMIC_DATA.actual_Runon_Timer)
   END_RUNG
   RUNG wire#w1
      I_Contact( #DYNAMIC_DATA."$ctrl_OpenClose" )
      Move(in := #STATIC_DATA.TIME_CLOSING_RUNON, out1 => #DYNAMIC_DATA.actual_Runon_Timer)
   END_RUNG
   // the same network as SCL:
   #_w1 := NOT #EXT_FAULT AND #DYNAMIC_DATA.msg_Flt_External AND NOT #STATIC_DATA.CONFIG_MAINT_OP;
   IF #_w1 AND #DYNAMIC_DATA."$ctrl_OpenClose" THEN
       #DYNAMIC_DATA.actual_Runon_Timer := #STATIC_DATA.TIME_OPENING_RUNON;
   END_IF;
   IF #_w1 AND NOT #DYNAMIC_DATA."$ctrl_OpenClose" THEN
       #DYNAMIC_DATA.actual_Runon_Timer := #STATIC_DATA.TIME_CLOSING_RUNON;
   END_IF;
END_REGION

REGION Network 44: External fault alarm
   // ▀▀▀▀▀▀▀▀▀▀▀▀▀▀▀▀▀▀▀▀▀▀▀▀▀▀▀▀▀▀▀▀▀▀▀▀▀▀▀▀▀▀▀▀
   // If the external fault signal (EXT_FAULT) is active, generate the external fault alarm
   // ▄▄▄▄▄▄▄▄▄▄▄▄▄▄▄▄▄▄▄▄▄▄▄▄▄▄▄▄▄▄▄▄▄▄▄▄▄▄▄▄▄▄▄▄
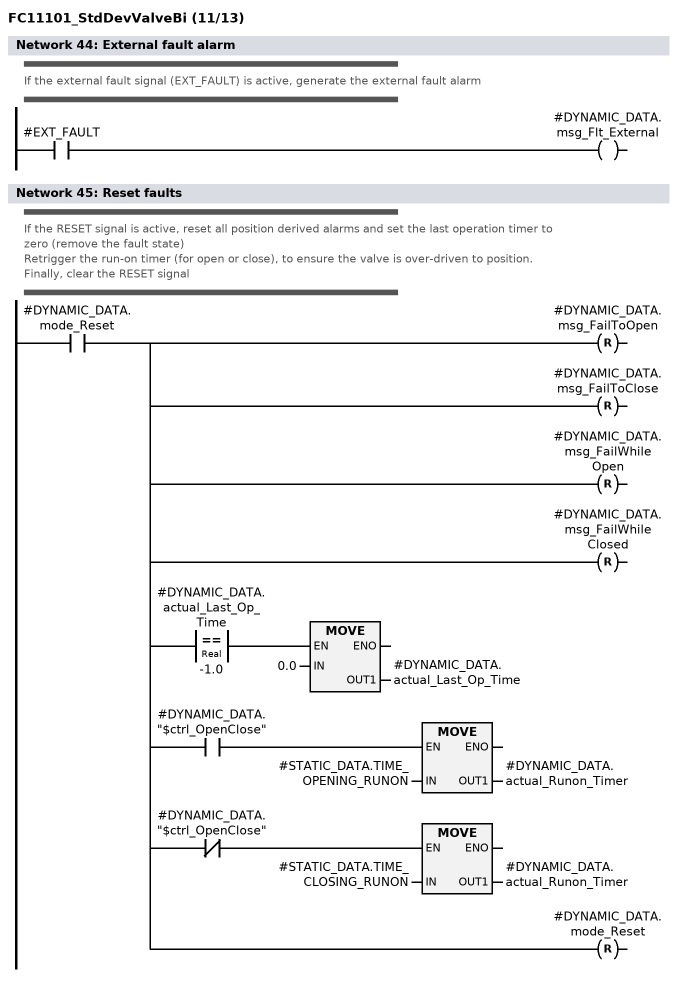
   RUNG wire#powerrail
      Contact( #EXT_FAULT )
      Coil( #DYNAMIC_DATA.msg_Flt_External )
   END_RUNG
   // the same network as SCL:
   #DYNAMIC_DATA.msg_Flt_External := #EXT_FAULT;
END_REGION

REGION Network 45: Reset faults
   // ▀▀▀▀▀▀▀▀▀▀▀▀▀▀▀▀▀▀▀▀▀▀▀▀▀▀▀▀▀▀▀▀▀▀▀▀▀▀▀▀▀▀▀▀
   // If the RESET signal is active, reset all position derived alarms and set the last operation timer to
   // zero (remove the fault state)
   // 
   // Retrigger the run-on timer (for open or close), to ensure the valve is over-driven to position.
   // 
   // Finally, clear the RESET signal
   // ▄▄▄▄▄▄▄▄▄▄▄▄▄▄▄▄▄▄▄▄▄▄▄▄▄▄▄▄▄▄▄▄▄▄▄▄▄▄▄▄▄▄▄▄
   RUNG wire#powerrail
      Contact( #DYNAMIC_DATA.mode_Reset )
      wire#w1
      R_Coil( #DYNAMIC_DATA.msg_FailToOpen )
   END_RUNG
   RUNG wire#w1
      R_Coil( #DYNAMIC_DATA.msg_FailToClose )
   END_RUNG
   RUNG wire#w1
      R_Coil( #DYNAMIC_DATA.msg_FailWhileOpen )
   END_RUNG
   RUNG wire#w1
      R_Coil( #DYNAMIC_DATA.msg_FailWhileClosed )
   END_RUNG
   RUNG wire#w1
      { S7_Templates := "SrcType := Real" } EQ_Contact(in1 := #DYNAMIC_DATA.actual_Last_Op_Time, in2 := -1.0)
      Move(in := 0.0, out1 => #DYNAMIC_DATA.actual_Last_Op_Time)
   END_RUNG
   RUNG wire#w1
      Contact( #DYNAMIC_DATA."$ctrl_OpenClose" )
      Move(in := #STATIC_DATA.TIME_OPENING_RUNON, out1 => #DYNAMIC_DATA.actual_Runon_Timer)
   END_RUNG
   RUNG wire#w1
      I_Contact( #DYNAMIC_DATA."$ctrl_OpenClose" )
      Move(in := #STATIC_DATA.TIME_CLOSING_RUNON, out1 => #DYNAMIC_DATA.actual_Runon_Timer)
   END_RUNG
   RUNG wire#w1
      R_Coil( #DYNAMIC_DATA.mode_Reset )
   END_RUNG
   // the same network as SCL:
   IF #DYNAMIC_DATA.mode_Reset THEN
       #DYNAMIC_DATA.msg_FailToOpen := FALSE;
       #DYNAMIC_DATA.msg_FailToClose := FALSE;
       #DYNAMIC_DATA.msg_FailWhileOpen := FALSE;
       #DYNAMIC_DATA.msg_FailWhileClosed := FALSE;
   END_IF;
   IF #DYNAMIC_DATA.mode_Reset AND (#DYNAMIC_DATA.actual_Last_Op_Time = (-1.0)) THEN
       #DYNAMIC_DATA.actual_Last_Op_Time := 0.0;
   END_IF;
   IF #DYNAMIC_DATA.mode_Reset AND #DYNAMIC_DATA."$ctrl_OpenClose" THEN
       #DYNAMIC_DATA.actual_Runon_Timer := #STATIC_DATA.TIME_OPENING_RUNON;
   END_IF;
   IF #DYNAMIC_DATA.mode_Reset AND NOT #DYNAMIC_DATA."$ctrl_OpenClose" THEN
       #DYNAMIC_DATA.actual_Runon_Timer := #STATIC_DATA.TIME_CLOSING_RUNON;
   END_IF;
   IF #DYNAMIC_DATA.mode_Reset THEN #DYNAMIC_DATA.mode_Reset := FALSE; END_IF;
END_REGION

REGION Network 46: Status signals
   // ▀▀▀▀▀▀▀▀▀▀▀▀▀▀▀▀▀▀▀▀▀▀▀▀▀▀▀▀▀▀▀▀▀▀▀▀▀▀▀▀▀▀▀▀
   // The status signals for faults, alarms and warnings are either duplicates of the message signals 
   // (signals beginning with msg_) or logical combinations of them.
   // 
   // The following is a full list of the status signals:
   // 
   //  UT31101_Dy_DevValveBi (full contents)
   //  ――――――――――――――――――――――――――――――――――――――――――
   //  SIGNAL NAME          FUNCTION                     TYPE
   //  ――――――――――――――――――――――――――――――――――――――――――
   //  status_Operating        STATUS — Valve is changing state           Bool
   //                      (1 = changing state, 0 = fixed state)
   //  status_Fault            STATUS — Valve is in fault              Bool
   //                      (1 = fault present, 0 = healthy)
   //  status_Energised        STATUS — Valve output is on              Bool
   //                      (1 = energised, 0 = deenergised)
   //  status_Aut           STATUS — Automatic mode active           Bool
   //                      (1 = auto mode on, 0 = auto mode off)
   //  status_Man          STATUS — Manual mode active             Bool
   //                      (1 = man mode on, 0 = man mode off)
   //  status_EStop          STATUS — E_STOP safety signal is active         Bool
   //                      (1 = active, 0 = healthy)
   //  status_Trip        STATUS — TRIP signal is active             Bool
   //                      (1 = active, 0 = healthy)
   //  status_Ilock         STATUS — INTERLOCK signal is active            Bool
   //                      (1 = active, 0 = healthy)
   //  status_Perm        STATUS — PERMISSIVE signal is active           Bool
   //                      (1 = active, 0 = healthy)
   //  status_BypassOn        STATUS — Valve is in bypass mode          Bool
   //                      (1 = Simulation mode, 0 = normal)
   //  status_SimOn           STATUS — Valve is in simulation mode               Bool
   //                      (1 = Simulation mode, 0 = normal)
   //  status_RemoteOn       STATUS — Valve is in remote mode                  Bool
   //                      (1 = Remote mode, 0 = normal)
   //  status_LocalOn         STATUS — Valve is in local mode                    Bool
   //                      (1 = Local mode, 0 = normal)
   //  status_RLOff         STATUS — Valve is in ALL mode                   Bool
   //                      (1 = ALL mode, 0 = normal)
   //  ――――――――――――――――――――――――――――――――――――――――――
   // ▄▄▄▄▄▄▄▄▄▄▄▄▄▄▄▄▄▄▄▄▄▄▄▄▄▄▄▄▄▄▄▄▄▄▄▄▄▄▄▄▄▄▄▄
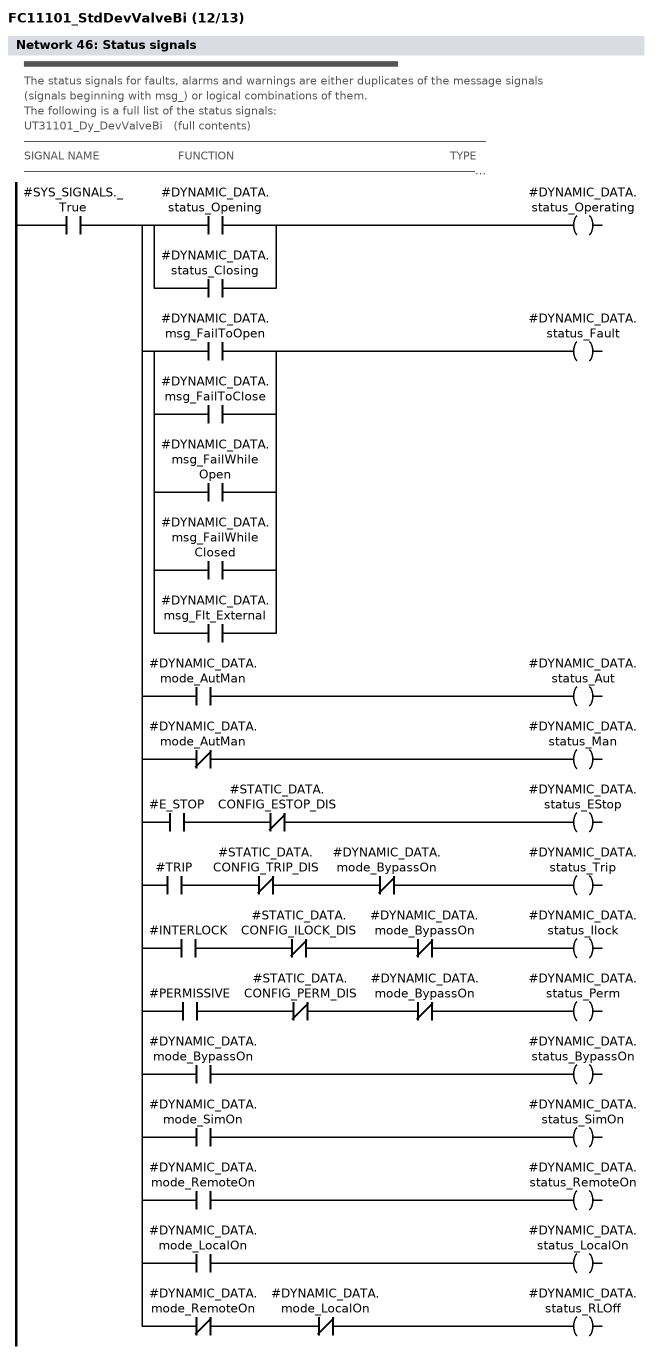
   RUNG wire#powerrail
      Contact( #SYS_SIGNALS._True )
      wire#w1
      Contact( #DYNAMIC_DATA.status_Opening )
      wire#w2
      Coil( #DYNAMIC_DATA.status_Operating )
   END_RUNG
   RUNG wire#w1
      Contact( #DYNAMIC_DATA.status_Closing )
   END_RUNG wire#w2
   RUNG wire#w1
      Contact( #DYNAMIC_DATA.msg_FailToOpen )
      wire#w3
      Coil( #DYNAMIC_DATA.status_Fault )
   END_RUNG
   RUNG wire#w1
      Contact( #DYNAMIC_DATA.msg_FailToClose )
   END_RUNG wire#w3
   RUNG wire#w1
      Contact( #DYNAMIC_DATA.msg_FailWhileOpen )
   END_RUNG wire#w3
   RUNG wire#w1
      Contact( #DYNAMIC_DATA.msg_FailWhileClosed )
   END_RUNG wire#w3
   RUNG wire#w1
      Contact( #DYNAMIC_DATA.msg_Flt_External )
   END_RUNG wire#w3
   RUNG wire#w1
      Contact( #DYNAMIC_DATA.mode_AutMan )
      Coil( #DYNAMIC_DATA.status_Aut )
   END_RUNG
   RUNG wire#w1
      I_Contact( #DYNAMIC_DATA.mode_AutMan )
      Coil( #DYNAMIC_DATA.status_Man )
   END_RUNG
   RUNG wire#w1
      Contact( #E_STOP )
      I_Contact( #STATIC_DATA.CONFIG_ESTOP_DIS )
      Coil( #DYNAMIC_DATA.status_EStop )
   END_RUNG
   RUNG wire#w1
      Contact( #TRIP )
      I_Contact( #STATIC_DATA.CONFIG_TRIP_DIS )
      I_Contact( #DYNAMIC_DATA.mode_BypassOn )
      Coil( #DYNAMIC_DATA.status_Trip )
   END_RUNG
   RUNG wire#w1
      Contact( #INTERLOCK )
      I_Contact( #STATIC_DATA.CONFIG_ILOCK_DIS )
      I_Contact( #DYNAMIC_DATA.mode_BypassOn )
      Coil( #DYNAMIC_DATA.status_Ilock )
   END_RUNG
   RUNG wire#w1
      Contact( #PERMISSIVE )
      I_Contact( #STATIC_DATA.CONFIG_PERM_DIS )
      I_Contact( #DYNAMIC_DATA.mode_BypassOn )
      Coil( #DYNAMIC_DATA.status_Perm )
   END_RUNG
   RUNG wire#w1
      Contact( #DYNAMIC_DATA.mode_BypassOn )
      Coil( #DYNAMIC_DATA.status_BypassOn )
   END_RUNG
   RUNG wire#w1
      Contact( #DYNAMIC_DATA.mode_SimOn )
      Coil( #DYNAMIC_DATA.status_SimOn )
   END_RUNG
   RUNG wire#w1
      Contact( #DYNAMIC_DATA.mode_RemoteOn )
      Coil( #DYNAMIC_DATA.status_RemoteOn )
   END_RUNG
   RUNG wire#w1
      Contact( #DYNAMIC_DATA.mode_LocalOn )
      Coil( #DYNAMIC_DATA.status_LocalOn )
   END_RUNG
   RUNG wire#w1
      I_Contact( #DYNAMIC_DATA.mode_RemoteOn )
      I_Contact( #DYNAMIC_DATA.mode_LocalOn )
      Coil( #DYNAMIC_DATA.status_RLOff )
   END_RUNG
   // the same network as SCL:
   #DYNAMIC_DATA.status_Operating := #SYS_SIGNALS._True AND (#DYNAMIC_DATA.status_Opening OR #DYNAMIC_DATA.status_Closing);
   #DYNAMIC_DATA.status_Fault := #SYS_SIGNALS._True AND (#DYNAMIC_DATA.msg_FailToOpen OR #DYNAMIC_DATA.msg_FailToClose OR #DYNAMIC_DATA.msg_FailWhileOpen OR #DYNAMIC_DATA.msg_FailWhileClosed OR #DYNAMIC_DATA.msg_Flt_External);
   #DYNAMIC_DATA.status_Aut := #SYS_SIGNALS._True AND #DYNAMIC_DATA.mode_AutMan;
   #DYNAMIC_DATA.status_Man := #SYS_SIGNALS._True AND NOT #DYNAMIC_DATA.mode_AutMan;
   #DYNAMIC_DATA.status_EStop := #SYS_SIGNALS._True AND #E_STOP AND NOT #STATIC_DATA.CONFIG_ESTOP_DIS;
   #DYNAMIC_DATA.status_Trip := #SYS_SIGNALS._True AND #TRIP AND NOT #STATIC_DATA.CONFIG_TRIP_DIS AND NOT #DYNAMIC_DATA.mode_BypassOn;
   #DYNAMIC_DATA.status_Ilock := #SYS_SIGNALS._True AND #INTERLOCK AND NOT #STATIC_DATA.CONFIG_ILOCK_DIS AND NOT #DYNAMIC_DATA.mode_BypassOn;
   #DYNAMIC_DATA.status_Perm := #SYS_SIGNALS._True AND #PERMISSIVE AND NOT #STATIC_DATA.CONFIG_PERM_DIS AND NOT #DYNAMIC_DATA.mode_BypassOn;
   #DYNAMIC_DATA.status_BypassOn := #SYS_SIGNALS._True AND #DYNAMIC_DATA.mode_BypassOn;
   #DYNAMIC_DATA.status_SimOn := #SYS_SIGNALS._True AND #DYNAMIC_DATA.mode_SimOn;
   #DYNAMIC_DATA.status_RemoteOn := #SYS_SIGNALS._True AND #DYNAMIC_DATA.mode_RemoteOn;
   #DYNAMIC_DATA.status_LocalOn := #SYS_SIGNALS._True AND #DYNAMIC_DATA.mode_LocalOn;
   #DYNAMIC_DATA.status_RLOff := #SYS_SIGNALS._True AND NOT #DYNAMIC_DATA.mode_RemoteOn AND NOT #DYNAMIC_DATA.mode_LocalOn;
END_REGION

REGION Network 47: OPEN_CMD output driver
   // ▀▀▀▀▀▀▀▀▀▀▀▀▀▀▀▀▀▀▀▀▀▀▀▀▀▀▀▀▀▀▀▀▀▀▀▀▀▀▀▀▀▀▀▀
   // The OPEN_CMD output drive will activate if all the following are true:
   // 
   //    1.  ESTOP is healthy or disabled (#wrkCtrlPriority40 = 1)
   // 
   //    2.  There is no fault condition (status_Fault = 0)
   // 
   //    3.  The valve is requested open ($ctrl_OpenClose = 1)
   // 
   //    4. The valve is opening (status_Opening =1)
   //         OR
   //      The valve is open (status_Open = 1) and either the run-on timer is active
   //      or the valve is configured to maintain outputs (CONFIG_MAINT_OP = 1)
   // 
   // The status_OpenOn signal is set to match the state of the OPEN_CMD
   // ▄▄▄▄▄▄▄▄▄▄▄▄▄▄▄▄▄▄▄▄▄▄▄▄▄▄▄▄▄▄▄▄▄▄▄▄▄▄▄▄▄▄▄▄
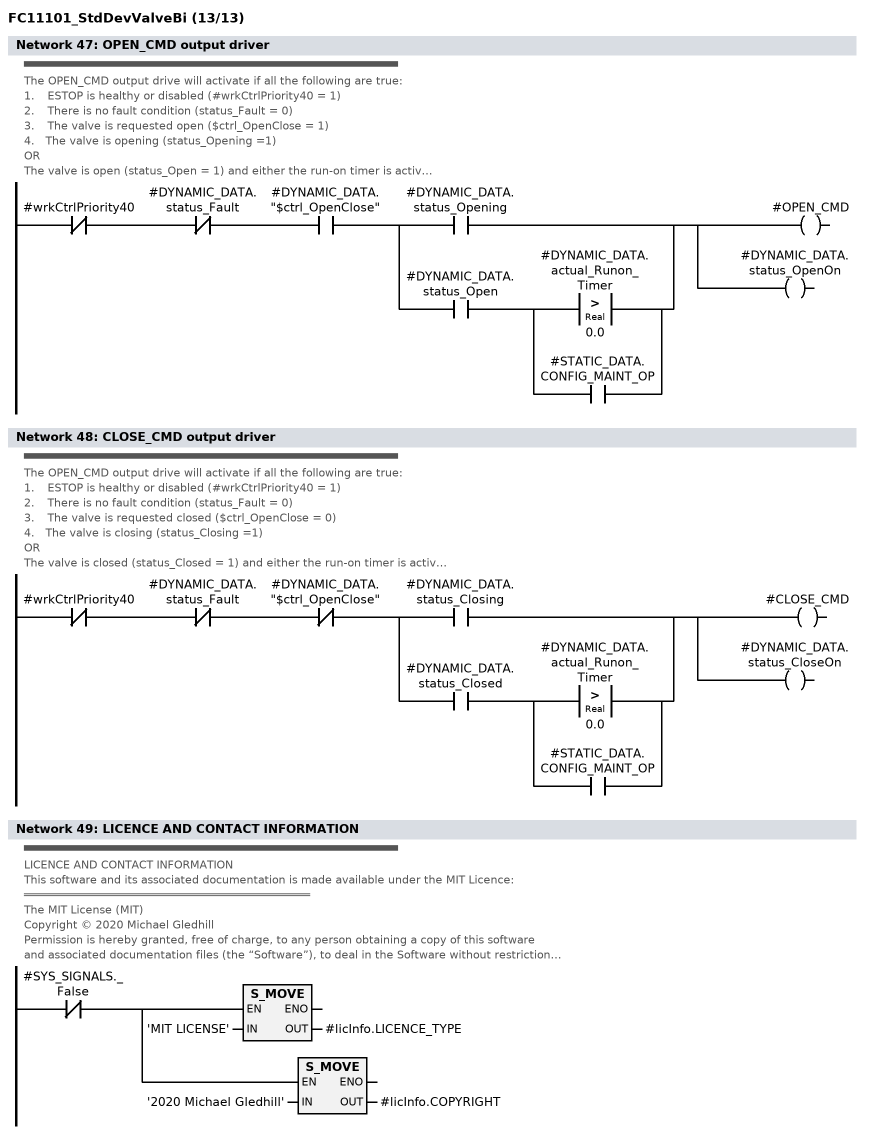
   RUNG wire#powerrail
      I_Contact( #wrkCtrlPriority40 )
      I_Contact( #DYNAMIC_DATA.status_Fault )
      Contact( #DYNAMIC_DATA."$ctrl_OpenClose" )
      wire#w1
      Contact( #DYNAMIC_DATA.status_Opening )
      wire#w2
      Coil( #OPEN_CMD )
   END_RUNG
   RUNG wire#w1
      Contact( #DYNAMIC_DATA.status_Open )
      wire#w3
      { S7_Templates := "SrcType := Real" } GT_Contact(in1 := #DYNAMIC_DATA.actual_Runon_Timer, in2 := 0.0)
   END_RUNG wire#w2
   RUNG wire#w3
      Contact( #STATIC_DATA.CONFIG_MAINT_OP )
   END_RUNG wire#w2
   RUNG wire#w2
      Coil( #DYNAMIC_DATA.status_OpenOn )
   END_RUNG
   // the same network as SCL:
   #OPEN_CMD := NOT #wrkCtrlPriority40 AND NOT #DYNAMIC_DATA.status_Fault AND #DYNAMIC_DATA."$ctrl_OpenClose" AND (#DYNAMIC_DATA.status_Opening OR (#DYNAMIC_DATA.status_Open AND ((#DYNAMIC_DATA.actual_Runon_Timer > 0.0) OR #STATIC_DATA.CONFIG_MAINT_OP)));
   #DYNAMIC_DATA.status_OpenOn := #OPEN_CMD;
END_REGION

REGION Network 48: CLOSE_CMD output driver
   // ▀▀▀▀▀▀▀▀▀▀▀▀▀▀▀▀▀▀▀▀▀▀▀▀▀▀▀▀▀▀▀▀▀▀▀▀▀▀▀▀▀▀▀▀
   // The OPEN_CMD output drive will activate if all the following are true:
   // 
   //    1.  ESTOP is healthy or disabled (#wrkCtrlPriority40 = 1)
   // 
   //    2.  There is no fault condition (status_Fault = 0)
   // 
   //    3.  The valve is requested closed ($ctrl_OpenClose = 0)
   // 
   //    4. The valve is closing (status_Closing =1)
   //         OR
   //      The valve is closed (status_Closed = 1) and either the run-on timer is active
   //      or the valve is configured to maintain outputs (CONFIG_MAINT_OP = 1)
   // 
   // The status_CloseOn signal is set to match the state of the CLOSE_CMD
   // ▄▄▄▄▄▄▄▄▄▄▄▄▄▄▄▄▄▄▄▄▄▄▄▄▄▄▄▄▄▄▄▄▄▄▄▄▄▄▄▄▄▄▄▄
   RUNG wire#powerrail
      I_Contact( #wrkCtrlPriority40 )
      I_Contact( #DYNAMIC_DATA.status_Fault )
      I_Contact( #DYNAMIC_DATA."$ctrl_OpenClose" )
      wire#w1
      Contact( #DYNAMIC_DATA.status_Closing )
      wire#w2
      Coil( #CLOSE_CMD )
   END_RUNG
   RUNG wire#w1
      Contact( #DYNAMIC_DATA.status_Closed )
      wire#w3
      { S7_Templates := "SrcType := Real" } GT_Contact(in1 := #DYNAMIC_DATA.actual_Runon_Timer, in2 := 0.0)
   END_RUNG wire#w2
   RUNG wire#w3
      Contact( #STATIC_DATA.CONFIG_MAINT_OP )
   END_RUNG wire#w2
   RUNG wire#w2
      Coil( #DYNAMIC_DATA.status_CloseOn )
   END_RUNG
   // the same network as SCL:
   #CLOSE_CMD := NOT #wrkCtrlPriority40 AND NOT #DYNAMIC_DATA.status_Fault AND NOT #DYNAMIC_DATA."$ctrl_OpenClose" AND (#DYNAMIC_DATA.status_Closing OR (#DYNAMIC_DATA.status_Closed AND ((#DYNAMIC_DATA.actual_Runon_Timer > 0.0) OR #STATIC_DATA.CONFIG_MAINT_OP)));
   #DYNAMIC_DATA.status_CloseOn := #CLOSE_CMD;
END_REGION

REGION Network 49: LICENCE AND CONTACT INFORMATION
   // ▀▀▀▀▀▀▀▀▀▀▀▀▀▀▀▀▀▀▀▀▀▀▀▀▀▀▀▀▀▀▀▀▀▀▀▀▀▀▀▀▀▀▀▀
   // LICENCE AND CONTACT INFORMATION
   // 
   // This software and its associated documentation is made available under the MIT Licence:
   // 
   // ════════════════════════════════════════════
   // 
   // The MIT License (MIT)
   // 
   // Copyright © 2020 Michael Gledhill
   // 
   // Permission is hereby granted, free of charge, to any person obtaining a copy of this software 
   // and associated documentation files (the “Software”), to deal in the Software without restriction, 
   // including without limitation the rights to use, copy, modify, merge, publish, distribute, 
   // sublicense, and/or sell copies of the Software, and to permit persons to whom the Software is 
   // furnished to do so, subject to the following conditions: 
   // 
   // The above copyright notice and this permission notice shall be included in all copies or 
   // substantial portions of the Software.
   // 
   // THE SOFTWARE IS PROVIDED “AS IS”, WITHOUT WARRANTY OF ANY KIND, EXPRESS OR IMPLIED, 
   // INCLUDING BUT NOT LIMITED TO THE WARRANTIES OF MERCHANTABILITY, FITNESS FOR A 
   // PARTICULAR PURPOSE AND NON-INFRINGEMENT. IN NO EVENT SHALL THE AUTHORS OR COPYRIGHT 
   // HOLDERS BE LIABLE FOR ANY CLAIM, DAMAGES OR OTHER LIABILITY, WHETHER IN AN ACTION OF 
   // CONTRACT, TORT OR OTHERWISE, ARISING FROM, OUT OF OR IN CONNECTION WITH THE SOFTWARE 
   // OR THE USE OR OTHER DEALINGS IN THE SOFTWARE.
   // 
   // ════════════════════════════════════════════
   //                    ┌────────────┐
   // You can reach the author by email here:   │  mg@practicalseries.com  │
   //                    └────────────┘
   // Questions, corrections, constructive criticism and complaints (polite ones) are invited.
   RUNG wire#powerrail
      I_Contact( #SYS_SIGNALS._False )
      wire#w1
      S_Move(in := 'MIT LICENSE', out => #licInfo.LICENCE_TYPE)
   END_RUNG
   RUNG wire#w1
      S_Move(in := '2020 Michael Gledhill', out => #licInfo.COPYRIGHT)
   END_RUNG
   // the same network as SCL:
   IF NOT #SYS_SIGNALS._False THEN
       #licInfo.LICENCE_TYPE := 'MIT LICENSE';
       #licInfo.COPYRIGHT := '2020 Michael Gledhill';
   END_IF;
END_REGION
END_FUNCTION

FUNCTION "FC19511_StdDebugInst1Order" : Void   // FC19511, LAD
TITLE = Standard Module [DEBUG] — First Order Response Simulation
{ S7_Optimized_Access := 'TRUE' }
AUTHOR : M_Gledhill
FAMILY : Debug
NAME : StdDebugInst1Order
VERSION : 0.1
// PRACTICAL SERIES AUTOMATION LIBRARY (PAL)   —   COPYRIGHT 2020 – M. GLEDHILL (MIT LICENCE)
//                   ———— ◆ ————
// FULL ONLINE DOCUMENTATION IS AVAILABLE AT: https://practicalseries.com/2001-pal/index.html
// stored: AutoNumber false, IsIECCheckEnabled true, SetENOAutomatically false, UDAEnableTagReadback false
   VAR_INPUT
      SYS_SIGNALS : "UT21000_Dy_SysSignals";   // Common system signals — logic and timing signals
      TRIGGER : Bool;   // Starts the simulation (rising edge starts the sim)
      INPUT : Real;   // The input function, x in the calculations
   END_VAR
   VAR_OUTPUT
      OUTPUT : Real;   // The output response, y in the calculations
   END_VAR
   VAR_IN_OUT
      DYNAMIC_DATA : "UT39511_Dy_DebugInst1Order";   // Dynamic data storage (UDT)
   END_VAR
   VAR_TEMP
      revInfo : "UT01000_St_SysRevision";   // Revision information for this block
      licInfo : "UT01001_St_SysLicence";   // Licensing information for this block
      act_CPUTime : DTL;   // Current CPU time (this block call)
      cal_01 : Real;   // Partial calculation see § 3.5 for details
      cal_02 : Real;   // Partial calculation see § 3.5 for details
      cal_03 : Real;   // Partial calculation see § 3.5 for details
      cal_04 : Real;   // Partial calculation see § 3.5 for details
      cal_05 : Real;   // Partial calculation see § 3.5 for details
      cal_06 : Real;   // Partial calculation see § 3.5 for details
      wrkElapsedTime : LTime;   // Working storage area (current elapsed time)
      wrkDeltaTime : LTime;   // Working storage area (current ΔT)
      wrkInt : Int;   // Working storage area (integer)
      wrkLInt : ULInt;   // Working storage area (long integer)
      wrkReal : Real;   // Working storage (real)
   END_VAR
   VAR CONSTANT
      k_NEG_MAX : Real := 3.4E-38;   // Largest negative number available to the REAL type
   END_VAR
   VAR_TEMP   // added for the SCL form of the ladder/FBD networks
      _w1 : Bool;
   END_VAR
BEGIN

REGION Network 1: Block description — Sections 1 to 2 inclusive
   // ▄▄▄▄▄▄▄▄▄▄▄▄▄▄▄▄▄▄▄▄▄▄▄▄▄▄▄▄▄▄▄▄▄  ＳＴＡＮＤＡＲＤ  ▄▄ 
   // 
   // 
   // TITLE:    DEBUG — FIRST ORDER RESPONSE SIMULATION
   // 
   // 
   // ▀▀▀▀▀▀▀▀▀▀▀▀▀▀▀▀▀▀▀▀▀▀▀▀▀▀▀▀▀▀▀▀▀▀▀▀▀▀▀▀▀▀▀▀ 
   // 
   // ┌──────────────────────────────────────────┐
   // │                                          │
   // │          FC19511 — SOFTWARE MODULE DESIGN SPECIFICATION (SMDS)            │
   // │                                          │
   // │      The PDF version of the SMDS for this module is available online here:        │
   // │              https://psop.uk/pal-smds-fc19511-p               │
   // │                                          │
   // │      It is also available as part of the Project User Defined Documentation,      │
   // │      it can be accessed by selecting this module in the Project Tree          │
   // │      (on the left) and pressing SHIFT+F1                        │
   // │                                          │
   // └─────────────────────────────────────── ʷᴵᴰ⁻ᶜᵇᶻ ┘
   // 
   // FC19511_StdDebugInst1Order is a debug simulation subroutine.
   // 
   // The module simulates a first order process reaction in response to an input signal.
   // 
   // The simulation is adjustable in terms of the system gain and the system time constant.
   // The output of the first order response simulation is in the form of a real number and is 
   // constrained to the resolution and range limits applicable to this number type within the Siemens 
   // Simatic S7-1500 controller.
   // 
   // The module will simulate a 1st order response to any type of input signal (step, ramp, sinusoid, 
   // freeform &c.).
   // 
   // The module also has a manual mode that can simulate an output at any specific time in 
   // response to a step input.
   // 
   // 
   // 
   // 
   // 
   // ▄▄▄▄▄▄▄▄▄▄▄▄▄▄▄▄▄▄▄▄▄▄▄▄▄▄▄▄▄▄▄▄▄▄▄▄▄▄▄▄▄▄▄▄
   // 1.     BLOCK TECHNICAL SUMMARY
   // 
   // 
   //  ――――――――――――――――――――――――――――――――――――――――――
   //  NOMENCLATURE & ADDRESSING
   //  ――――――――――――――――――――――――――――――――――――――――――
   //  BLOCK TITLE         1st Order Response Simulation
   //  BLOCK FUNCTION GROUP    Debug  
   //  BLOCK ADDRESS       FC19511
   //  BLOCK SYMBOL        FC19511_StdDebugInst1Order
   //  BLOCK USER ID         StdDebugInst1Order
   // 
   //  ――――――――――――――――――――――――――――――――――――――――――
   //  BLOCK TYPE & USAGE
   //  ――――――――――――――――――――――――――――――――――――――――――
   //  BLOCK TYPE         Function (FC)
   //  BLOCK NUMBER        19511
   //  LANGUAGE           LAD
   //  OPTIMISED ACCESS     Yes
   //  PAL USAGE TYPE       Standard block
   // 
   //  ――――――――――――――――――――――――――――――――――――――――――
   //  METRICS
   //  ――――――――――――――――――――――――――――――――――――――――――
   //  EXECUTION TIME        091.0 μs¹    (Note: = 14.4µs if TRIGGER is FALSE)
   //  LOAD MEMORY       46.0 kB
   //  WORK MEMORY           0.9 kB  
   //  ――――――――――――――――――――――――――――――――――――――――――
   //                ¹ Measured on: CPU-1515-2PN (order no. 6ES7512-2AM02-0AB0) 
   //                             https://psop.uk/pal-ds-cpu1515
   // 
   // 
   // 
   // ▂▂▂▂▂▂▂▂▂▂▂▂▂▂▂▂▂▂▂▂▂▂▂▂▂▂▂▂▂▂▂▂▂▂▂▂▂▂▂▂▂▂▂▂
   // 1.1      Additional referenced documents
   // 
   // 
   // In addition to the documents referenced in OB1 (section DOCUMENT REFERENCES), the 
   // following documents are associated with this module:
   // 
   // 
   //  ――――――――――――――――――――――――――――――――――――――――――
   //  REF.     DOCUMENT NO.         TITLE
   //  ――――――――――――――――――――――――――――――――――――――――――
   //  101  PS2001-5-2331-fc19511      FC19511 Calculation Sheet
   //  102  PS2001-5-2331-fc19511-011    FC19511 1st Order Response Simulation Spreadsheet
   //  ――――――――――――――――――――――――――――――――――――――――――
   // 
   // 
   // 
   //                ━━━   ⬙⬙⬙⬙⬙⬙   ━━━
   // 
   // 
   // 
   // ▄▄▄▄▄▄▄▄▄▄▄▄▄▄▄▄▄▄▄▄▄▄▄▄▄▄▄▄▄▄▄▄▄▄▄▄▄▄▄▄▄▄▄▄
   // 2.     FUNCTIONAL DESCRIPTION
   // 
   // 
   // ████████████████████████████████████████████
   // █                                          █
   // █ Note:   The following descriptions are taken from the associated Software Module     █
   // █     Design Specification [PS2001-5-2312-fc19511], the SMDS contains various     █
   // █     graphs that cannot be easily reproduced in these module comments. Where    █
   // █     essential, some rudimentary images have been included; however,        █
   // █     these are better viewed directly in the SMDS.                   █
   // █                                          █
   // █     Where images of the graphs are included, these are generated using           █
   // █     the Unicode braille characters and were generated by the following web site:     █
   // █     https://505e06b2.github.io/Image-to-Braille/                  █
   // █     (the images are 100 braille characters wide)                   █
   // █                                          █
   // █     The SMDS can be accessed directly by selecting this module (FC19511) in the     █
   // █     Project Tree (on the left) and pressing SHIFT+F1.                 █
   // █                                          █
   // █      The PDF version of the SMDS for this module is available online here:        █
   // █              https://psop.uk/pal-smds-fc19511-p               █
   // █                                          █
   // ████████████████████████████████████████████
   // 
   // FC19511 is the 1st Order Response Simulation module. The purpose of this module is to simulate 
   // a “first order” process reaction in response to an input signal.
   // 
   // First order systems are the most common type of system response for process control systems 
   // (for example the response generated when heating a tank of liquid). First order systems are often 
   // referred to as “first order lag” systems and generally reflect systems whereby the response of the 
   // system (the temperature of the water in the above example) follows the input (the temperature 
   // of the heating element) but with some delay (or lag). First order systems do not produce an 
   // oscillatory response to a step change of input and do not overshoot the input.
   // 
   // First order systems are so called because the equation linking the input to the out-put is always 
   // defined by a first order differential equation.
   // 
   // The following graphs show typical first order responses to a step change input:
   // 
   // 
   // 
   // Output y(t)
   // │⠄⠄⠄⠄⠄⠄⠄⠄⠄⠄⠄⠄⠄⠄⠄⠄⠄⠄⠄⠄⠄⠄⠄⠄⠄⠄⠄⠄⠄⠄⠄⠄⠄⠄⠄⠄⠄⠄⠄⠄⠄⠄⠄⠄⠄⠄⠄⠄⠄⠄⠄⠄⠄⠄⠄⠄⠄⠄⠄⠄⠄⠄⠄⠄⠄⠄⠄⠄⠄⠄⠄⠄⠄⠄⠄⠄⠄⠄⠄⠄⠄⠄⠄⠄⠄⠄⠄⠄⠄⠄⠄⠄⠄⠄⠄⠄⠄⠄⠄⠄
   // │⠤⠤⠤⠤⠤⠤⠤⠤⠤⠤⠤⠤⠤⠤⠤⠤⠤⠤⠤⠤⠤⠤⠤⠤⠤⠤⠤⠤⠤⠤⠤⠤⠤⠤⠤⠤⠤⠤⠤⠤⠤⠤⠤⠤⠤⠤⠤⠤⠤⠤⠤⢀⣀⣀⣀⣀⣀⣠⣤⣤⣤⣤⣤⣤⣤⣤⣤⣤⣤⣤⣤⣤⣤⣤⣤⠤⠤⠤⠤⠤⠤⠤⠤⠤⠤⠤⠤⠤⠤⠤⠤⠤⠤⠤⠤⠤⠤⠤⠤⠤
   // │⡇⠄⠄⠄⠄⠄⠄⠄⠄⠄⠄⠄⠄⠄⠄⠄⠄⠄⠄⠄⠄⠄⠄⠄⠄⠄⠄⠄⠄⠄⠄⠄⠄⠄⠄⠄⠄⠄⠄⣀⣀⣤⣤⡶⠶⠶⠒⠒⠛⠉⠉⠉⠉⠉⠉⠉⠉⠉⠉⠁⠄⠄⠄⠄⠄⠄⠄⠄⠄⠄⠄⠄⠄⠄⠄⠄⠄⠄⠄⠄⠄⠄⠄⠄⠄⠄⠄⠄⠄⠄⠄⠄⠄⠄⠄⠄⠄⠄⠄⠄
   // │⡇←— STEP INPUT  ⠄⠄⠄⠄⠄⠄⠄⠄⠄⠄⠄⠄⠄⠄⠄⠄⠄⠄⠄⠄⣀⣤⡶⠖⠚⠉⠉⠉⠁⠄⠄⠄⠄⠄⠄⠄⠄⠄⠄⠄⠄⠄⠄⠄⠄⠄⠄⠄⠄⠄⠄⠄⠄⠄⠄⠄⠄⠄⠄⠄⠄⠄⠄⠄⠄⠄⠄⠄⠄⠄⠄⠄⠄⠄⠄⠄⠄⠄⠄⠄⠄⠄⠄⠄⠄⠄⠄
   // │⡇⠄⠄⠄⠄⠄⠄⠄⠄⠄⠄⠄⠄⠄⠄⠄⠄⠄⠄⠄⠄⠄⠄⠄⠄⠄⠄⠄⢀⣠⡴⠖⠋⠉⠁⠄⠄⠄⠄⠄⠄⠄⠄⠄⠄⠄⠄⠄⠄⠄⠄⠄⠄⠄⠄⠄⠄⠄⠄⠄⠄⠄⠄⠄⠄⠄⠄⠄⠄⠄⠄⠄⠄⠄⠄⠄⠄⠄⠄⠄⠄⠄⠄⠄⠄⠄⠄⠄⠄⠄⠄⠄⠄⠄⠄⠄⠄⠄⠄⠄
   // │⡇⠄⠄⠄⠄⠄⠄⠄⠄⠄⠄⠄⠄⠄⠄⠄⠄⠄⠄⠄⠄⠄⠄⠄⠄⠄⣠⠾⠋⠄⠄⠄⠄⠄⠄⠄⠄⠄⠄⠄⠄⠄⠄⠄⠄⠄⠄⠄⠄⠄⠄⠄⠄⠄⠄⠄⠄⠄⠄⠄⠄⠄⠄⠄⠄⠄⠄⠄⠄⠄⠄⠄⠄⠄⠄⠄⠄⠄⠄⠄⠄⠄⠄⠄⠄⠄⠄⠄⠄⠄⠄⠄⠄⠄⠄⠄⠄⠄⠄⠄
   // │⡇⠄⠄⠄⠄⠄⠄⠄⠄⠄⠄⠄⠄⠄⠄⠄⠄⠄⠄⠄⠄⠄⠄⣀⡴⠋⠁⠄⠄⠄⠄⠄⠄⠄⠄⠄⠄⠄⠄⠄⠄⠄⠄⠄⠄⠄⠄⠄⠄⠄⠄⠄⠄⠄⠄⠄⠄⠄⠄⠄⠄⠄⠄⠄⠄⠄⠄⠄⠄⠄⠄⠄⠄⠄⠄⠄⠄⠄⠄⠄⠄⠄⠄⠄⠄⠄⠄⠄⠄⠄⠄⠄⠄⠄⠄⠄⠄⠄⠄⠄
   // │⡇⠄⠄⠄⠄⠄⠄⠄⠄⠄⠄⠄⠄⠄⠄⠄⠄⠄⠄⠄⠄⣠⠾⠁←— DELAYED OUTPUT  ⠄⠄⠄⠄⠄⠄⠄⠄⠄⠄⠄⠄⠄⠄⠄⠄⠄⠄⠄⠄⠄⠄⠄⠄⠄⠄⠄⠄⠄⠄⠄⠄⠄⠄⠄⠄⠄⠄⠄⠄⠄⠄⠄⠄⠄⠄⠄⠄⠄⠄⠄⠄⠄⠄⠄⠄⠄⠄
   // │⡇⠄⠄⠄⠄⠄⠄⠄⠄⠄⠄⠄⠄⠄⠄⠄⠄⠄⠄⢀⡴⠏⠄⠄⠄⠄⠄⠄⠄⠄⠄⠄⠄⠄⠄⠄⠄⠄⠄⠄⠄⠄⠄⠄⠄⠄⠄⠄⠄⠄⠄⠄⠄⠄⠄⠄⠄⠄⠄⠄⠄⠄⠄⠄⠄⠄⠄⠄⠄⠄⠄⠄⠄⠄⠄⠄⠄⠄⠄⠄⠄⠄⠄⠄⠄⠄⠄⠄⠄⠄⠄⠄⠄⠄⠄⠄⠄⠄⠄⠄
   // │⡇⠄⠄⠄⠄⠄⠄⠄⠄⠄⠄⠄⠄⠄⠄⠄⠄⢀⣴⠏⠄⠄⠄⠄⠄⠄⠄⠄⠄⠄⠄⠄⠄⠄⠄⠄⠄⠄⠄⠄⠄⠄⠄⠄⠄⠄⠄⠄⠄⠄⠄⠄⠄⠄⠄⠄⠄⠄⠄⠄⠄⠄⠄⠄⠄⠄⠄⠄⠄⠄⠄⠄⠄⠄⠄⠄⠄⠄⠄⠄⠄⠄⠄⠄⠄⠄⠄⠄⠄⠄⠄⠄⠄⠄⠄⠄⠄⠄⠄⠄
   // │⡇⠄⠄⠄⠄⠄⠄⠄⠄⠄⠄⠄⠄⠄⠄⠄⢠⡜⠃⠄⠄⠄⠄⠄⠄⠄⠄⠄⠄⠄⠄⠄⠄⠄⠄⠄⠄⠄⠄⠄⠄⠄⠄⠄⠄⠄⠄⠄⠄⠄⠄⠄⠄⠄⠄⠄⠄⠄⠄⠄⠄⠄⠄⠄⠄⠄⠄⠄⠄⠄⠄⠄⠄⠄⠄⠄⠄⠄⠄⠄⠄⠄⠄⠄⠄⠄⠄⠄⠄⠄⠄⠄⠄⠄⠄⠄⠄⠄⠄⠄
   // │⡇⠄⠄⠄⠄⠄⠄⠄⠄⠄⠄⠄⠄⠄⠄⢰⠟⠁⠄⠄⠄⠄⠄⠄⠄⠄⠄⠄⠄⠄⠄⠄⠄⠄⠄⠄⠄⠄⠄⠄⠄⠄⠄⠄⠄⠄⠄⠄⠄⠄⠄⠄⠄⠄⠄⠄⠄⠄⠄⠄⠄⠄⠄⠄⠄⠄⠄⠄⠄⠄⠄⠄⠄⠄⠄⠄⠄⠄⠄⠄⠄⠄⠄⠄⠄⠄⠄⠄⠄⠄⠄⠄⠄⠄⠄⠄⠄⠄⠄⠄
   // │⡇⠄⠄⠄⠄⠄⠄⠄⠄⠄⠄⠄⠄⠄⣰⡏⠄⠄⠄⠄⠄⠄⠄⠄⠄⠄⠄⠄⠄⠄⠄⠄⠄⠄⠄⠄⠄⠄⠄⠄⠄⠄⠄⠄⠄⠄⠄⠄⠄⠄⠄⠄⠄⠄⠄⠄⠄⠄⠄⠄⠄⠄⠄⠄⠄⠄⠄⠄⠄⠄⠄⠄⠄⠄⠄⠄⠄⠄⠄⠄⠄⠄⠄⠄⠄⠄⠄⠄⠄⠄⠄⠄⠄⠄⠄⠄⠄⠄⠄⠄
   // │⡇⠄⠄⠄⠄⠄⠄⠄⠄⠄⠄⠄⠄⢠⠏⠄⠄⠄⠄⠄⠄⠄⠄⠄⠄⠄⠄⠄⠄⠄⠄⠄⠄⠄⠄⠄⠄⠄⠄⠄⠄⠄⠄⠄⠄⠄⠄⠄⠄⠄⠄⠄⠄⠄⠄⠄⠄⠄⠄⠄⠄⠄⠄⠄⠄⠄⠄⠄⠄⠄⠄⠄⠄⠄⠄⠄⠄⠄⠄⠄⠄⠄⠄⠄⠄⠄⠄⠄⠄⠄⠄⠄⠄⠄⠄⠄⠄⠄⠄⠄
   // │⡇⠄⠄⠄⠄⠄⠄⠄⠄⠄⠄⠄⣰⡟⠄⠄⠄⠄⠄⠄⠄⠄⠄⠄⠄⠄⠄⠄⠄⠄⠄⠄⠄⠄⠄⠄⠄⠄⠄⠄⠄⠄⠄⠄⠄⠄⠄⠄⠄⠄⠄⠄⠄⠄⠄⠄⠄⠄⠄⠄⠄⠄⠄⠄⠄⠄⠄⠄⠄⠄⠄⠄⠄⠄⠄⠄⠄⠄⠄⠄⠄⠄⠄⠄⠄⠄⠄⠄⠄⠄⠄⠄⠄⠄⠄⠄⠄⠄⠄⠄
   // │⡇⠄⠄⠄⠄⠄⠄⠄⠄⠄⠄⢠⠏⠄⠄⠄⠄⠄⠄⠄⠄⠄⠄⠄⠄⠄⠄⠄⠄⠄⠄⠄⠄⠄⠄⠄⠄⠄⠄⠄⠄⠄⠄⠄⠄⠄⠄⠄⠄⠄⠄⠄⠄⠄⠄⠄⠄⠄⠄⠄⠄⠄⠄⠄⠄⠄⠄⠄⠄⠄⠄⠄⠄⠄⠄⠄⠄⠄⠄⠄⠄⠄⠄⠄⠄⠄⠄⠄⠄⠄⠄⠄⠄⠄⠄⠄⠄⠄⠄⠄
   // │⡇⠄⠄⠄⠄⠄⠄⠄⠄⠄⢠⡿⠄⠄⠄⠄⠄⠄⠄⠄⠄⠄⠄⠄⠄⠄⠄⠄⠄⠄⠄⠄⠄⠄⠄⠄⠄⠄⠄⠄⠄⠄⠄⠄⠄⠄⠄⠄⠄⠄⠄⠄⠄⠄⠄⠄⠄⠄⠄⠄⠄⠄⠄⠄⠄⠄⠄⠄⠄⠄⠄⠄⠄⠄⠄⠄⠄⠄⠄⠄⠄⠄⠄⠄⠄⠄⠄⠄⠄⠄⠄⠄⠄⠄⠄⠄⠄⠄⠄⠄
   // │⡇⠄⠄⠄⠄⠄⠄⠄⠄⠄⡿⠁⠄⠄⠄⠄⠄⠄⠄⠄⠄⠄⠄⠄⠄⠄⠄⠄⠄⠄⠄⠄⠄⠄⠄⠄⠄⠄⠄⠄⠄⠄⠄⠄⠄⠄⠄⠄⠄⠄⠄⠄⠄⠄⠄⠄⠄⠄⠄⠄⠄⠄⠄⠄⠄⠄⠄⠄⠄⠄⠄⠄⠄⠄⠄⠄⠄⠄⠄⠄⠄⠄⠄⠄⠄⠄⠄⠄⠄⠄⠄⠄⠄⠄⠄⠄⠄⠄⠄⠄
   // │⡇⠄⠄⠄⠄⠄⠄⠄⠄⣼⠃⠄⠄⠄⠄⠄⠄⠄⠄⠄⠄⠄⠄⠄⠄⠄⠄⠄⠄⠄⠄⠄⠄⠄⠄⠄⠄⠄⠄⠄⠄⠄⠄⠄⠄⠄⠄⠄⠄⠄⠄⠄⠄⠄⠄⠄⠄⠄⠄⠄⠄⠄⠄⠄⠄⠄⠄⠄⠄⠄⠄⠄⠄⠄⠄⠄⠄⠄⠄⠄⠄⠄⠄⠄⠄⠄⠄⠄⠄⠄⠄⠄⠄⠄⠄⠄⠄⠄⠄⠄
   // │⡇⠄⠄⠄⠄⠄⠄⠄⢰⡟⠄⠄⠄⠄⠄⠄⠄⠄⠄⠄⠄⠄⠄⠄⠄⠄⠄⠄⠄⠄⠄⠄⠄⠄⠄⠄⠄⠄⠄⠄⠄⠄⠄⠄⠄⠄⠄⠄⠄⠄⠄⠄⠄⠄⠄⠄⠄⠄⠄⠄⠄⠄⠄⠄⠄⠄⠄⠄⠄⠄⠄⠄⠄⠄⠄⠄⠄⠄⠄⠄⠄⠄⠄⠄⠄⠄⠄⠄⠄⠄⠄⠄⠄⠄⠄⠄⠄⠄⠄⠄
   // │⡇⠄⠄⠄⠄⠄⠄⠄⡞⠄⠄⠄⠄⠄⠄⠄⠄⠄⠄⠄⠄⠄⠄⠄⠄⠄⠄⠄⠄⠄⠄⠄⠄⠄⠄⠄⠄⠄⠄⠄⠄⠄⠄⠄⠄⠄⠄⠄⠄⠄⠄⠄⠄⠄⠄⠄⠄⠄⠄⠄⠄⠄⠄⠄⠄⠄⠄⠄⠄⠄⠄⠄⠄⠄⠄⠄⠄⠄⠄⠄⠄⠄⠄⠄⠄⠄⠄⠄⠄⠄⠄⠄⠄⠄⠄⠄⠄⠄⠄⠄
   // │⡇⠄⠄⠄⠄⠄⠄⣰⡇⠄⠄⠄⠄⠄⠄⠄⠄⠄⠄⠄⠄⠄⠄⠄⠄⠄⠄⠄⠄⠄⠄⠄⠄⠄⠄⠄⠄⠄⠄⠄⠄⠄⠄⠄⠄⠄⠄⠄⠄⠄⠄⠄⠄⠄⠄⠄⠄⠄⠄⠄⠄⠄⠄⠄⠄⠄⠄⠄⠄⠄⠄⠄⠄⠄⠄⠄⠄⠄⠄⠄⠄⠄⠄⠄⠄⠄⠄⠄⠄⠄⠄⠄⠄⠄⠄⠄⠄⠄⠄⠄
   // │⡇⠄⠄⠄⠄⠄⢰⡟⠄⠄⠄⠄⠄⠄⠄⠄⠄⠄⠄⠄⠄⠄⠄⠄⠄⠄⠄⠄⠄⠄⠄⠄⠄⠄⠄⠄⠄⠄⠄⠄⠄⠄⠄⠄⠄⠄⠄⠄⠄⠄⠄⠄⠄⠄⠄⠄⠄⠄⠄⠄⠄⠄⠄⠄⠄⠄⠄⠄⠄⠄⠄⠄⠄⠄⠄⠄⠄⠄⠄⠄⠄⠄⠄⠄⠄⠄⠄⠄⠄⠄⠄⠄⠄⠄⠄⠄⠄⠄⠄⠄
   // │⡇⠄⠄⠄⠄⠄⣸⠁⠄⠄⠄⠄⠄⠄⠄⠄⠄⠄⠄⠄⠄⠄⠄⠄⠄⠄⠄⠄⠄⠄⠄⠄⠄⠄⠄⠄⠄⠄⠄⠄⠄⠄⠄⠄⠄⠄⠄⠄⠄⠄⠄⠄⠄⠄⠄⠄⠄⠄⠄⠄⠄⠄⠄⠄⠄⠄⠄⠄⠄⠄⠄⠄⠄⠄⠄⠄⠄⠄⠄⠄⠄⠄⠄⠄⠄⠄⠄⠄⠄⠄⠄⠄⠄⠄⠄⠄⠄⠄⠄⠄
   // │⡇⠄⠄⠄⠄⢠⡇⠄⠄⠄⠄⠄⠄⠄⠄⠄⠄⠄⠄⠄⠄⠄⠄⠄⠄⠄⠄⠄⠄⠄⠄⠄⠄⠄⠄⠄⠄⠄⠄⠄⠄⠄⠄⠄⠄⠄⠄⠄⠄⠄⠄⠄⠄⠄⠄⠄⠄⠄⠄⠄⠄⠄⠄⠄⠄⠄⠄⠄⠄⠄⠄⠄⠄⠄⠄⠄⠄⠄⠄⠄⠄⠄⠄⠄⠄⠄⠄⠄⠄⠄⠄⠄⠄⠄⠄⠄⠄⠄⠄⠄
   // │⡇⠄⠄⠄⠄⣿⠃⠄⠄⠄⠄⠄⠄⠄⠄⠄⠄⠄⠄⠄⠄⠄⠄⠄⠄⠄⠄⠄⠄⠄⠄⠄⠄⠄⠄⠄⠄⠄⠄⠄⠄⠄⠄⠄⠄⠄⠄⠄⠄⠄⠄⠄⠄⠄⠄⠄⠄⠄⠄⠄⠄⠄⠄⠄⠄⠄⠄⠄⠄⠄⠄⠄⠄⠄⠄⠄⠄⠄⠄⠄⠄⠄⠄⠄⠄⠄⠄⠄⠄⠄⠄⠄⠄⠄⠄⠄⠄⠄⠄⠄
   // │⡇⠄⠄⠄⢸⡏⠄⠄⠄⠄⠄⠄⠄⠄⠄⠄⠄⠄⠄⠄⠄⠄⠄⠄⠄⠄⠄⠄⠄⠄⠄⠄⠄⠄⠄⠄⠄⠄⠄⠄⠄⠄⠄⠄⠄⠄⠄⠄⠄⠄⠄⠄⠄⠄⠄⠄⠄⠄⠄⠄⠄⠄⠄⠄⠄⠄⠄⠄⠄⠄⠄⠄⠄⠄⠄⠄⠄⠄⠄⠄⠄⠄⠄⠄⠄⠄⠄⠄⠄⠄⠄⠄⠄⠄⠄⠄⠄⠄⠄⠄
   // │⡇⠄⠄⠄⣸⠁⠄⠄⠄⠄⠄⠄⠄⠄⠄⠄⠄⠄⠄⠄⠄⠄⠄⠄⠄⠄⠄⠄⠄⠄⠄⠄⠄⠄⠄⠄⠄⠄⠄⠄⠄⠄⠄⠄⠄⠄⠄⠄⠄⠄⠄⠄⠄⠄⠄⠄⠄⠄⠄⠄⠄⠄⠄⠄⠄⠄⠄⠄⠄⠄⠄⠄⠄⠄⠄⠄⠄⠄⠄⠄⠄⠄⠄⠄⠄⠄⠄⠄⠄⠄⠄⠄⠄⠄⠄⠄⠄⠄⠄⠄
   // │⡇⠄⠄⢠⡇⠄⠄⠄⠄⠄⠄⠄⠄⠄⠄⠄⠄⠄⠄⠄⠄⠄⠄⠄⠄⠄⠄⠄⠄⠄⠄⠄⠄⠄⠄⠄⠄⠄⠄⠄⠄⠄⠄⠄⠄⠄⠄⠄⠄⠄⠄⠄⠄⠄⠄⠄⠄⠄⠄⠄⠄⠄⠄⠄⠄⠄⠄⠄⠄⠄⠄⠄⠄⠄⠄⠄⠄⠄⠄⠄⠄⠄⠄⠄⠄⠄⠄⠄⠄⠄⠄⠄⠄⠄⠄⠄⠄⠄⠄⠄
   // │⡇⠄⠄⣼⠇⠄⠄⠄⠄⠄⠄⠄⠄⠄⠄⠄⠄⠄⠄⠄⠄⠄⠄⠄⠄⠄⠄⠄⠄⠄⠄⠄⠄⠄⠄⠄⠄⠄⠄⠄⠄⠄⠄⠄⠄⠄⠄⠄⠄⠄⠄⠄⠄⠄⠄⠄⠄⠄⠄⠄⠄⠄⠄⠄⠄⠄⠄⠄⠄⠄⠄⠄⠄⠄⠄⠄⠄⠄⠄⠄⠄⠄⠄⠄⠄⠄⠄⠄⠄⠄⠄⠄⠄⠄⠄⠄⠄⠄⠄⠄
   // │⡇⠄⠄⡿⠄⠄⠄⠄⠄⠄⠄⠄⠄⠄⠄⠄⠄⠄⠄⠄⠄⠄⠄⠄⠄⠄⠄⠄⠄⠄⠄⠄⠄⠄⠄⠄⠄⠄⠄⠄⠄⠄⠄⠄⠄⠄⠄⠄⠄⠄⠄⠄⠄⠄⠄⠄⠄⠄⠄⠄⠄⠄⠄⠄⠄⠄⠄⠄⠄⠄⠄⠄⠄⠄⠄⠄⠄⠄⠄⠄⠄⠄⠄⠄⠄⠄⠄⠄⠄⠄⠄⠄⠄⠄⠄⠄⠄⠄⠄⠄
   // │⡇⠄⢰⠃⠄⠄⠄⠄⠄⠄⠄⠄⠄⠄⠄⠄⠄⠄⠄⠄⠄⠄⠄⠄⠄⠄⠄⠄⠄⠄⠄⠄⠄⠄⠄⠄⠄⠄⠄⠄⠄⠄⠄⠄⠄⠄⠄⠄⠄⠄⠄⠄⠄⠄⠄⠄⠄⠄⠄⠄⠄⠄⠄⠄⠄⠄⠄⠄⠄⠄⠄⠄⠄⠄⠄⠄⠄⠄⠄⠄⠄⠄⠄⠄⠄⠄⠄⠄⠄⠄⠄⠄⠄⠄⠄⠄⠄⠄⠄⠄
   // │⡇⠄⣾⠄⠄⠄⠄⠄⠄⠄⠄⠄⠄⠄⠄⠄⠄⠄⠄⠄⠄⠄⠄⠄⠄⠄⠄⠄⠄⠄⠄⠄⠄⠄⠄⠄⠄⠄⠄⠄⠄⠄⠄⠄⠄⠄⠄⠄⠄⠄⠄⠄⠄⠄⠄⠄⠄⠄⠄⠄⠄⠄⠄⠄⠄⠄⠄⠄⠄⠄⠄⠄⠄⠄⠄⠄⠄⠄⠄⠄⠄⠄⠄⠄⠄⠄⠄⠄⠄⠄⠄⠄⠄⠄⠄⠄⠄⠄⠄⠄
   // │⡇⢰⡟⠄⠄⠄⠄⠄⠄⠄⠄⠄⠄⠄⠄⠄⠄⠄⠄⠄⠄⠄⠄⠄⠄⠄⠄⠄⠄⠄⠄⠄⠄⠄⠄⠄⠄⠄⠄⠄⠄⠄⠄⠄⠄⠄⠄⠄⠄⠄⠄⠄⠄⠄⠄⠄⠄⠄⠄⠄⠄⠄⠄⠄⠄⠄⠄⠄⠄⠄⠄⠄⠄⠄⠄⠄⠄⠄⠄⠄⠄⠄⠄⠄⠄⠄⠄⠄⠄⠄⠄⠄⠄⠄⠄⠄⠄⠄⠄⠄
   // │⡇⣾⠇⠄⠄⠄⠄⠄⠄⠄⠄⠄⠄⠄⠄⠄⠄⠄⠄⠄⠄⠄⠄⠄⠄⠄⠄⠄⠄⠄⠄⠄⠄⠄⠄⠄⠄⠄⠄⠄⠄⠄⠄⠄⠄⠄⠄⠄⠄⠄⠄⠄⠄⠄⠄⠄⠄⠄⠄⠄⠄⠄⠄⠄⠄⠄⠄⠄⠄⠄⠄⠄⠄⠄⠄⠄⠄⠄⠄⠄⠄⠄⠄⠄⠄⠄⠄⠄⠄⠄⠄⠄⠄⠄⠄⠄⠄⠄⠄⠄
   // │⡇⡿⠄⠄⠄⠄⠄⠄⠄⠄⠄⠄⠄⠄⠄⠄⠄⠄⠄⠄⠄⠄⠄⠄⠄⠄⠄⠄⠄⠄⠄⠄⠄⠄⠄⠄⠄⠄⠄⠄⠄⠄⠄⠄⠄⠄⠄⠄⠄⠄⠄⠄⠄⠄⠄⠄⠄⠄⠄⠄⠄⠄⠄⠄⠄⠄⠄⠄⠄⠄⠄⠄⠄⠄⠄⠄⠄⠄⠄⠄⠄⠄⠄⠄⠄⠄⠄⠄⠄⠄⠄⠄⠄⠄⠄⠄⠄⠄⠄⠄
   // │⡇⠃⠄⠄⠄⠄⠄⠄⠄⠄⠄⠄⠄⠄⠄⠄⠄⠄⠄⠄⠄⠄⠄⠄⠄⠄⠄⠄⠄⠄⠄⠄⠄⠄⠄⠄⠄⠄⠄⠄⠄⠄⠄⠄⠄⠄⠄⠄⠄⠄⠄⠄⠄⠄⠄⠄⠄⠄⠄⠄⠄⠄⠄⠄⠄⠄⠄⠄⠄⠄⠄⠄⠄⠄⠄⠄⠄⠄⠄⠄⠄⠄⠄⠄⠄⠄⠄⠄⠄⠄⠄⠄⠄⠄⠄⠄⠄⠄⠄⠄
   // ┼ ─ ─ ─ ─ ─ ─ ─ ─ ─ ─ ─ ─ ─ ─ ─ ─ ─ ─ ─ ─ ─ ─ ─ ─ ─ ─ ─ ─ ─ ─ ─ ─ ─ ─ ─ ─ ─ ─ ─ ─ ─ ─  ─ ─ ─ ─    Time (t)
   // 
   // 
   // 
   // ▂▂▂▂▂▂▂▂▂▂▂▂▂▂▂▂▂▂▂▂▂▂▂▂▂▂▂▂▂▂▂▂▂▂▂▂▂▂▂▂▂▂▂▂
   // 2.1      Scope and limitations of the simulation
   // 
   // 
   // The first order response simulation will provide a real time response for a first order simulation.
   // 
   // The simulation will be adjustable in terms of the system gain (K) and the time constant of the 
   // system (τ).
   // 
   // The output of the first order response simulation will be in the form of a real number.
   // 
   // 
   // 
   // 
   // ▁▁▁▁▁▁▁▁▁▁▁▁▁▁▁▁▁▁▁▁▁▁▁▁▁▁▁▁▁▁▁▁▁▁▁▁▁▁▁▁▁▁▁▁
   // 2.1.1     The limitations of the simulation
   // 
   // 
   // The output of the second order response simulation will be in the form of a real number and will 
   // be constrained to the limits applicable to this number type within the Siemens controller.
   // 
   // The S7-1500 range of Controllers supports real numbers as values, these are 32-bit numbers 
   // and, within a Controller, have the following range limits:
   // 
   // 
   //  ――――――――――――――――――――――――――――――――――――――――――
   //              LOWER RANGE LIMIT     UPPER RANGE LIMIT
   //  ――――――――――――――――――――――――――――――――――――――――――
   //  S7-1500 real number:     ±3.402323×10^(-38)           ±3.402323×10^(+38)
   //  ――――――――――――――――――――――――――――――――――――――――――
   // 
   // This range is considered acceptable for all practical uses of the module.
   // 
   // 
   // 
   // ▁▁▁▁▁▁▁▁▁▁▁▁▁▁▁▁▁▁▁▁▁▁▁▁▁▁▁▁▁▁▁▁▁▁▁▁▁▁▁▁▁▁▁▁
   // 2.1.2     The nature of the simulation calculations
   // 
   // 
   // The module will generate the correct responses for any first order system. The module uses a 
   // discrete time approximation calculation to determine the correct output for any given input. The 
   // calculation is an iterative algorithm, the formulae for which is derived in full in the associated 
   // calculations sheet [Ref. 101], available here:
   // 
   //          https://psop.uk/pal-calc-fc19511-p
   // 
   // These calculations are based around the mathematical functions available to the Controller 
   // (these are in addition to the standard mathematical operations: addition, subtraction, 
   // multiplication and division).
   // 
   // Each Controller supports the following common mathematical functions:
   // 
   // 
   //  ――――――――――――――――――――――――――――――――――――――――――
   //  OPERATION    EXAMPLE         DESCRIPTION
   //  ――――――――――――――――――――――――――――――――――――――――――
   //  SQR        x^2          Form the square
   //  SQRT         √x            Form the square root
   //  EXP        e^x          Exponential
   //  LN          log_e(⁡x)        Natural logarithm
   //  SIN         sin(⁡x)         Sine
   //  ASIN          sin^-1(x)          Arcsine, inverse sine
   //  COS          cos(⁡x)        Cosine
   //  ACOS        cos^-1(x)         Arccosine, inverse cosine
   //  TAN           tan(⁡x)         Tangent
   //  ATAN         tan^-1(x)         Arctangent, inverse tangent
   //  ABS        |x|            Modulus
   //  ――――――――――――――――――――――――――――――――――――――――――
   //  Table 2.1 S7 Controller — common mathematical functions
   // 
   // 
   // 
   // ▂▂▂▂▂▂▂▂▂▂▂▂▂▂▂▂▂▂▂▂▂▂▂▂▂▂▂▂▂▂▂▂▂▂▂▂▂▂▂▂▂▂▂▂
   // 2.2      The second order response
   // 
   // 
   // The response of a second order system (y) to an input (x) is defined using the general form of a 
   // second order system transfer function, this is expressed below in the time domain as a second 
   // order differential equation (see the calculation sheet [Ref. 101], Appendix B for details):
   // 
   //                 dy
   //             τ ----- ┼  y  =  Kx  (2.1)
   //                 dt
   // 
   // Where:    K is the system gain
   //      τ is referred to as the system time constant (seconds)
   // 
   // 
   // 
   // ▂▂▂▂▂▂▂▂▂▂▂▂▂▂▂▂▂▂▂▂▂▂▂▂▂▂▂▂▂▂▂▂▂▂▂▂▂▂▂▂▂▂▂▂
   // 2.3      The calculations
   // 
   // 
   // Two forms of calculation are needed to produce a model for a first order system. The first being a 
   // continuous simulation running in real-time with a varying or constant input signal.
   // 
   // The second being the discrete result for a step input under manual conditions (i.e. a fixed input 
   // and specific time are provided and a single, corresponding output value generated).
   // 
   // Both of these calculations are discussed in the following sections:
   // 
   // 
   // 
   // ▁▁▁▁▁▁▁▁▁▁▁▁▁▁▁▁▁▁▁▁▁▁▁▁▁▁▁▁▁▁▁▁▁▁▁▁▁▁▁▁▁▁▁▁
   // 2.3.1     Real-time simulation calculation for any input type
   // 
   // 
   // The normal operation of the module (in automatic mode) is to produce a continuous real-time 
   // model of a first order system that once triggered, runs continuously, producing an output 
   // response that mimics a first order system responding to a variable (or constant) input as time 
   // progresses, the simulation continues until the triggering condition is removed.
   // 
   // The calculation needed to produce a first order system response to any type of input signal is 
   // best achieved using a discrete time approximation method. The details of this method are given 
   // in [Ref. 101], Section 2.1, and the results are given below:
   // 
   // The final form of the calculations that will be used in the FC19511 software module for a real time 
   // simulation to any input type is:
   // 
   //    y[n] = Ka x[n]  ┼ (1-a) y[n-1]  (2.2)
   // 
   //              ΔT
   //    where:   a = ----------
   //            τ+ΔT
   // 
   //    K is the system gain (a constant number)
   //    τ is the system time constant (in seconds)
   //    Δt is the sampling interval between calculations (in seconds)
   //    x[n] is the input at the current iteration 
   //    y[n] is the output at the current iteration 
   //    y[n-1] is the output at the previous iteration 
   // 
   // 
   // It should be noted that this is an iterative algorithm, the previous value of the output must 
   // be retained between calculations.
   // 
   // For best results, Δt should be very much smaller than the system time constant, i.e.:
   // 
   //                    τ
   //    Δt ≪ τ      Typically, Δt ≤ ----
   //                      10
   // 
   // Note also, that Δt need not be constant between samples.
   // 
   // 
   // 
   // ▁▁▁▁▁▁▁▁▁▁▁▁▁▁▁▁▁▁▁▁▁▁▁▁▁▁▁▁▁▁▁▁▁▁▁▁▁▁▁▁▁▁▁▁
   // 2.3.2     Manual simulation calculation for a step input at a particular time
   // 
   // 
   // In manual mode, an instantaneous calculation is carried out using the first order equation at a 
   // particular time and for a particular input value.
   // 
   // Since, under manual control, both the time and the input are fixed single values, it is not possible 
   // to determine the nature of the input (i.e. is it a ramp, sinusoid &c.), hence for all manual 
   // operations within the simulation, the input is considered to be a step input that changed to the 
   // manually specified input value at time = 0, and that prior to this the input was zero¹. I.e. a step 
   // input that changed from zero to the specified value at time = 0.
   // 
   // To produce a specific output value in response to a fixed step input at a particular time, it is 
   // necessary to solve the first order differential equation given in equation (2.1), as a non-iterative, 
   // discreate calculation. To do this, it is necessary to convert the equation into the Laplace domain² 
   // (using standard Laplace transforms, see [Ref. 101], Appendix A) algebraically solve the equation 
   // and then convert the result back to the time domain (using the standard inverse Laplace 
   // transforms, again see [Ref. 101], Appendix A).
   // 
   // The final form of the manual calculations that will be used in the FC19511 software module for a 
   // single point input type is:
   // 
   //          ┌      -t/τ  ┐
   //    y(t) = KX│ 1 ─  e   │
   //          └       ┘
   // 
   //    K is the system gain (a constant number)
   //    τ is the system time constant (in seconds)
   //    X is the fixed input value
   // 
   // 
   // ――――――――――
   // ¹         A step response is the most common type of response
   // 
   // ²         The calculation sheet associated with this module [Ref. 101], explains the Laplace 
   //      transform mechanisms and how they are used within the calculations necessary for 
   //      the functioning of this module. Further explanation of the Laplace transform is not 
   //      given in this document, again the reader is referred to the calculation 
   //      sheet [Ref. 101].
   // ――――――――――
   // 
   // 
   // 
   // ▁▁▁▁▁▁▁▁▁▁▁▁▁▁▁▁▁▁▁▁▁▁▁▁▁▁▁▁▁▁▁▁▁▁▁▁▁▁▁▁▁▁▁▁
   // 2.3.3     Calculation spreadsheet model
   // 
   // 
   // An accompanying spreadsheet [Ref. 016] is available, this allows all the various responses to be 
   // graphically simulated with adjustable values (it was this spreadsheet that produced the various 
   // response plots used within this document), this spreadsheet is available here:
   // 
   //      http://psop.uk/pal-calc-fc19511-p
   // 
   // 
   // 
   // ▂▂▂▂▂▂▂▂▂▂▂▂▂▂▂▂▂▂▂▂▂▂▂▂▂▂▂▂▂▂▂▂▂▂▂▂▂▂▂▂▂▂▂▂
   // 2.4      Real-time responses for typical inputs
   // 
   // 
   // First order systems respond to various types of input (step, ramp, sinusoidal) in very predictable 
   // ways. First order systems never produce oscillatory responses (unless the input itself is 
   // oscillating) and never overshoot the input (cf. 2nd order systems, see FC19512). The general 
   // response of a first order system is that of an inherent delay (or lag) in the response of the output 
   // compared with the input.
   // 
   // This inherent delay is reflected in the system time constant (τ), measured in seconds.
   // 
   // The following sections consider how the system time constant affects the output for several 
   // typical input types:
   // 
   // 
   // STEP INPUT
   // 
   // │⠄⠄⠄⠄⠄⠄⠄⠄⠄⠄⠄⠄⠄⠄⠄⠄⠄⠄⠄⠄⠄⠄⠄τ = 20s⠄⠄⠄⠄⠄⠄⠄⠄⠄⠄⠄⠄⠄⠄⠄⠄⠄⠄⠄⠄⠄⠄⠄⠄⠄⠄⠄⠄⠄⠄⠄⠄⠄⠄⠄⠄⠄⠄⠄⠄⠄⠄⠄⠄⠄⠄⠄⠄⠄⠄⠄⠄⠄⠄⠄⠄⠄⠄⠄⠄⠄⠄⠄⠄⠄⠄⠄⠄⠄⠄⠄⠄
   // X─ ─ ─ ─ ─ ─ ─ ─ ─ ─ ─ ─ ─ ─ ─ ─ ─ ─ ─ ─ ─ ─ ─ ─ ─ ─ ─ ─ ─ ─ ─ ─ ─ ─ ─ ─ ─ ─ ─ ─ ─ ─ ─ ─ ─ ─ ─
   // │⠄⠄⠄⠄⠄⠄⠄⠄⠄⠄⠄⠄⠄⠄⠄⠄⠄⠄⠄⠄⠄⠄⠄⠄⠄⠄⠄⠄⠄⠄⠄⠄⠄⠄⠄⠄⠄⠄⠄⠄⠄⠄⠄⠄⠄⠄⠄⠄⠄⠄⠄⠄⠄⠄⠄⠄⠄⠄⠄⠄⠄⣀⣀⣀⣀⣠⣤⡤⠤⠤⠶⠶⠶⠶⠒⠒⠒⠒⠚⠛⠛⠛⠛⠉⠉⠉⠉⠉⠉⠉⠉⠉⠉⠉⠉⠉⠉⠉⠉⠉
   // │⠄⠄⠄⠄⠄⠄⠄⠄⠄⠄⠄⠄⠄⠄⠄⠄⠄⠄⠄⠄⠄⠄⠄⠄⠄⠄⠄⠄⠄⠄⠄⠄⠄⠄⠄⠄⠄⠄⠄⠄⠄⠄⠄⠄⠄⠄⠄⠄⠄⠄⢀⣀⣠⡤⠤⠶⠖⠒⠛⠄⠄⠄⠄⠄⠄⠄⠄⠄⠄⠄⠄⠄⠄⠄99% of steady state ─ ─ ─ ─ ╎⠄
   // │⠄⠄⠄⠄⠄⠄⠄⠄⠄⠄⠄⠄⠄⠄⠄⠄⠄⠄⠄⠄⠄⠄⠄⠄⠄⠄⠄⠄⠄⠄⠄⠄⠄⠄⠄⠄⠄⠄⠄⠄⠄⠄⠄⢀⣀⣠⠴⠖⠚⠋⠉⠁⠄⠄⠄⠄⠄⠄⠄⠄⠄⠄⠄⠄⠄⠄⠄⠄⠄⠄⠄⠄⠄⠄⠄⠄⠄⠄⠄⠄⠄⠄⠄⠄⠄⠄⠄⠄⠄⠄⠄⠄⠄⠄⠄⠄⠄⠄╎⠄
   // │⠄⠄⠄⠄⠄⠄⠄⠄⠄⠄⠄⠄⠄⠄⠄⠄⠄⠄⠄⠄⠄⠄⠄⠄⠄⠄⠄⠄⠄⠄⠄⠄⠄⠄⠄⠄⠄⠄⢀⣠⡤⠖⠚⠉⠁⠄⠄⠄⠄⠄⠄⠄⠄⠄⠄⠄⠄⠄⠄⠄⠄⠄⠄⠄⠄⠄⠄⠄⠄⠄⠄⠄⠄⠄⠄⠄⠄⠄⠄⠄⠄⠄⠄⠄⠄⠄⠄⠄⠄⠄⠄⠄⠄⠄⠄⠄⠄⠄╎⠄
   // │⠄⠄⠄⠄⠄⠄⠄⠄⠄⠄⠄⠄⠄⠄⠄⠄⠄⠄⠄⠄⠄⠄⠄⠄⠄⠄⠄⠄⠄⠄⠄⠄⠄⠄⠄⣠⡴⠚⠋⠁⠄⠄⠄⠄⠄⠄⠄⠄⠄⠄⠄⠄⠄⠄⠄⠄⠄⠄⠄⠄⠄⠄⠄⠄⠄⠄⠄⠄⠄⠄⠄⠄⠄⠄⠄⠄⠄⠄⠄⠄⠄⠄⠄⠄⠄⠄⠄⠄⠄⠄⠄⠄⠄⠄⠄⠄⠄⠄╎⠄
   // │⠄⠄⠄⠄⠄⠄⠄⠄⠄⠄⠄⠄⠄⠄⠄⠄⠄⠄⠄⠄⠄⠄⠄⠄⠄⠄⠄⠄⠄⠄⠄⢀⣠⠖⠋⠁⠄⠄⠄⠄⠄⠄⠄⠄⠄⠄⠄⠄⠄⠄⠄⠄⠄⠄⠄⠄⠄⠄⠄⠄⠄⠄⠄⠄⠄⠄⠄⠄⠄⠄⠄⠄⠄⠄⠄⠄⠄⠄⠄⠄⠄⠄⠄⠄⠄⠄⠄⠄⠄⠄⠄⠄⠄⠄⠄⠄⠄⠄╎⠄
   // │⠄⠄⠄⠄⠄⠄⠄⠄⠄⠄⠄⠄⠄⠄⠄⠄⠄⠄⠄⠄⠄⠄⠄⠄⠄⠄⠄⠄⠄⣠⠴⠋⠄⠄⠄⠄⠄⠄⠄⠄⠄⠄⠄⠄⠄⠄⠄⠄⠄⠄⠄⠄⠄⠄⠄⠄⠄⠄⠄⠄⠄⠄⠄⠄⠄⠄⠄⠄⠄⠄⠄⠄⠄⠄⠄⠄⠄⠄⠄⠄⠄⠄⠄⠄⠄⠄⠄⠄⠄⠄⠄⠄⠄⠄⠄⠄⠄⠄╎⠄
   // │⠄⠄⠄⠄⠄⠄⠄⠄⠄⠄⠄⠄⠄⠄⠄⠄⠄⠄⠄⠄⠄⠄⠄⠄⠄⠄⢀⡤⠚⠁⠄⠄⠄⠄⠄⠄⠄⠄⠄⠄⠄⠄⠄⠄⠄⠄⠄⠄⠄⠄⠄⠄⠄⠄⠄⠄⠄⠄⠄⠄⠄⠄⠄⠄⠄⠄⠄⠄⠄⠄⠄⠄⠄⠄⠄⠄⠄⠄⠄⠄⠄⠄⠄⠄⠄⠄⠄⠄⠄⠄⠄⠄⠄⠄⠄⠄⠄⠄╎⠄
   // │⠄⠄⠄⠄⠄⠄⠄⠄⠄⠄⠄⠄⠄⠄⠄⠄⠄⠄⠄⠄⠄⠄⠄⠄⢀⡴⠋⠄⠄⠄⠄⠄⠄⠄⠄⠄⠄⠄⠄⠄⠄⠄⠄⠄⠄⠄⠄⠄⠄⠄⠄⠄⠄⠄⠄⠄⠄⠄⠄⠄⠄⠄⠄⠄⠄⠄⠄⠄⠄⠄⠄⠄⠄⠄⠄⠄⠄⠄⠄⠄⠄⠄⠄⠄⠄⠄⠄⠄⠄⠄⠄⠄⠄⠄⠄⠄⠄⠄╎⠄
   // │⠄⠄⠄⠄⠄⠄⠄⠄⠄⠄⠄⠄⠄⠄⠄⠄⠄⠄⠄⠄⠄⠄⢀⡴⠋⠄⠄⠄⠄⠄⠄⠄⠄⠄⠄⠄⠄⠄⠄⠄⠄⠄⠄⠄⠄⠄⠄⠄⠄⠄⠄⠄⠄⠄⠄⠄⠄⠄⠄⠄⠄⠄⠄⠄⠄⠄⠄⠄⠄⠄⠄⠄⠄⠄⠄⠄⠄⠄⠄⠄⠄⠄⠄⠄⠄⠄⠄⠄⠄⠄⠄⠄⠄⠄⠄⠄⠄⠄╎⠄
   // │⠄⠄⠄⠄⠄⠄⠄⠄⠄⠄⠄⠄⠄⠄⠄⠄⠄⠄⠄⠄⠄⣠⠋⠄⠄⠄⠄⠄⠄⠄⠄⠄⠄⠄⠄⠄⠄⠄⠄⠄⠄⠄⠄⠄⠄⠄⠄⠄⠄⠄⠄⠄⠄⠄⠄⠄⠄⠄⠄⠄⠄⠄⠄⠄⠄⠄⠄⠄⠄⠄⠄⠄⠄⠄⠄⠄⠄⠄⠄⠄⠄⠄⠄⠄⠄⠄⠄⠄⠄⠄⠄⠄⠄⠄⠄⠄⠄⠄╎⠄
   // │⠄⠄⠄⠄⠄⠄⠄⠄⠄⠄⠄⠄⠄⠄⠄⠄⠄⠄⠄⢀⠞⠁⠄⠄⠄⠄⠄⠄⠄⠄⠄⠄⠄⠄⠄⠄⠄⠄⠄⠄⠄⠄⠄⠄⠄⠄⠄⠄⠄⠄⠄⠄⠄⠄⠄⠄⠄⠄⠄⠄⠄⠄⠄⠄⠄⠄⠄⠄⠄⠄⠄⠄⠄⠄⠄⠄⠄⠄⠄⠄⠄⠄⠄⠄⠄⠄⠄⠄⠄⠄⠄⠄⠄⠄⠄⠄⠄⠄╎⠄
   // │⠄⠄⠄⠄⠄⠄⠄⠄⠄⠄⠄⠄⠄⠄⠄⠄⠄⠄⣴⠋─ ─ ─ ─ ─  63% of steady state  ⠄⠄⠄⠄⠄⠄⠄⠄⠄⠄⠄⠄⠄⠄⠄⠄⠄⠄⠄⠄⠄⠄⠄⠄⠄⠄⠄⠄⠄⠄⠄⠄⠄⠄⠄⠄⠄⠄⠄⠄⠄⠄⠄⠄⠄⠄⠄⠄⠄⠄⠄╎⠄
   // │⠄⠄⠄⠄⠄⠄⠄⠄⠄⠄⠄⠄⠄⠄⠄⠄⢀⡾⠁⠄⠄⠄⠄⠄⠄⠄⠄⠄⠄⠄⠄⠄⠄⠄⠄⠄⠄⠄⠄⠄⠄⠄⠄⠄⠄⠄⠄⠄⠄⠄⠄⠄⠄⠄⠄⠄⠄⠄⠄⠄⠄⠄⠄⠄⠄⠄⠄⠄⠄⠄⠄⠄⠄⠄⠄⠄⠄⠄⠄⠄⠄⠄⠄⠄⠄⠄⠄⠄⠄⠄⠄⠄⠄⠄⠄⠄⠄⠄╎⠄
   // │⠄⠄⠄⠄⠄⠄⠄⠄⠄⠄⠄⠄⠄⠄⠄⢠⠞⠄ ╎⠄⠄⠄⠄⠄⠄⠄⠄⠄⠄⠄⠄⠄⠄⠄⠄⠄⠄⠄⠄⠄⠄⠄⠄⠄⠄⠄⠄⠄⠄⠄⠄⠄⠄⠄⠄⠄⠄⠄⠄⠄⠄⠄⠄⠄⠄⠄⠄⠄⠄⠄⠄⠄⠄⠄⠄⠄⠄⠄⠄⠄⠄⠄⠄⠄⠄⠄⠄⠄⠄⠄⠄⠄⠄⠄⠄⠄⠄╎⠄
   // │⠄⠄⠄⠄⠄⠄⠄⠄⠄⠄⠄⠄⠄⠄⣠⠏⠄⠄ ╎⠄⠄⠄⠄⠄⠄⠄⠄⠄⠄⠄⠄⠄⠄⠄⠄⠄⠄⠄⠄⠄⠄⠄⠄⠄⠄⠄⠄⠄⠄⠄⠄⠄⠄⠄⠄⠄⠄⠄⠄⠄⠄⠄⠄⠄⠄⠄⠄⠄⠄⠄⠄⠄⠄⠄⠄⠄⠄⠄⠄⠄⠄⠄⠄⠄⠄⠄⠄⠄⠄⠄⠄⠄⠄⠄⠄⠄⠄╎⠄
   // │⠄⠄⠄⠄⠄⠄⠄⠄⠄⠄⠄⠄⠄⣰⠋⠄⠄⠄ ╎⠄⠄⠄⠄⠄⠄⠄⠄⠄⠄⠄⠄⠄⠄⠄⠄⠄⠄⠄⠄⠄⠄⠄⠄⠄⠄⠄⠄⠄⠄⠄⠄⠄⠄⠄⠄⠄⠄⠄⠄⠄⠄⠄⠄⠄⠄⠄⠄⠄⠄⠄⠄⠄⠄⠄⠄⠄⠄⠄⠄⠄⠄⠄⠄⠄⠄⠄⠄⠄⠄⠄⠄⠄⠄⠄⠄⠄⠄╎⠄
   // │⠄⠄⠄⠄⠄⠄⠄⠄⠄⠄⠄⠄⣰⠃⠄⠄⠄⠄ ╎⠄⠄⠄⠄⠄⠄⠄⠄⠄⠄⠄⠄⠄⠄⠄⠄⠄⠄⠄⠄⠄⠄⠄⠄⠄⠄⠄⠄⠄⠄⠄⠄⠄⠄⠄⠄⠄⠄⠄⠄⠄⠄⠄⠄⠄⠄⠄⠄⠄⠄⠄⠄⠄⠄⠄⠄⠄⠄⠄⠄⠄⠄⠄⠄⠄⠄⠄⠄⠄⠄⠄⠄⠄⠄⠄⠄⠄⠄╎⠄
   // │⠄⠄⠄⠄⠄⠄⠄⠄⠄⠄⠄⣸⠃⠄⠄⠄⠄⠄ ╎⠄⠄⠄⠄⠄⠄⠄⠄⠄⠄⠄⠄⠄⠄⠄⠄⠄⠄⠄⠄⠄⠄⠄⠄⠄⠄⠄⠄⠄⠄⠄⠄⠄⠄⠄⠄⠄⠄⠄⠄⠄⠄⠄⠄⠄⠄⠄⠄⠄⠄⠄⠄⠄⠄⠄⠄⠄⠄⠄⠄⠄⠄⠄⠄⠄⠄⠄⠄⠄⠄⠄⠄⠄⠄⠄⠄⠄⠄╎⠄
   // │⠄⠄⠄⠄⠄⠄⠄⠄⠄⠄⣰⠃⠄⠄⠄⠄⠄⠄ ╎⠄⠄⠄⠄⠄⠄⠄⠄⠄⠄⠄⠄⠄⠄⠄⠄⠄⠄⠄⠄⠄⠄⠄⠄⠄⠄⠄⠄⠄⠄⠄⠄⠄⠄⠄⠄⠄⠄⠄⠄⠄⠄⠄⠄⠄⠄⠄⠄⠄⠄⠄⠄⠄⠄⠄⠄⠄⠄⠄⠄⠄⠄⠄⠄⠄⠄⠄⠄⠄⠄⠄⠄⠄⠄⠄⠄⠄⠄╎⠄
   // │⠄⠄⠄⠄⠄⠄⠄⠄⠄⣰⠃⠄⠄⠄⠄⠄⠄⠄ ╎⠄⠄⠄⠄⠄⠄⠄⠄⠄⠄⠄⠄⠄⠄⠄⠄⠄⠄⠄⠄⠄⠄⠄⠄⠄⠄⠄⠄⠄⠄⠄⠄⠄⠄⠄⠄⠄⠄⠄⠄⠄⠄⠄⠄⠄⠄⠄⠄⠄⠄⠄⠄⠄⠄⠄⠄⠄⠄⠄⠄⠄⠄⠄⠄⠄⠄⠄⠄⠄⠄⠄⠄⠄⠄⠄⠄⠄⠄╎⠄
   // │⠄⠄⠄⠄⠄⠄⠄⠄⢰⠇⠄⠄⠄⠄⠄⠄⠄⠄ ╎⠄⠄⠄⠄⠄⠄⠄⠄⠄⠄⠄⠄⠄⠄⠄⠄⠄⠄⠄⠄⠄⠄⠄⠄⠄⠄⠄⠄⠄⠄⠄⠄⠄⠄⠄⠄⠄⠄⠄⠄⠄⠄⠄⠄⠄⠄⠄⠄⠄⠄⠄⠄⠄⠄⠄⠄⠄⠄⠄⠄⠄⠄⠄⠄⠄⠄⠄⠄⠄⠄⠄⠄⠄⠄⠄⠄⠄⠄╎⠄
   // │⠄⠄⠄⠄⠄⠄⠄⢠⡏⠄⠄⠄⠄⠄⠄⠄⠄⠄ ╎⠄⠄⠄⠄⠄⠄⠄⠄⠄⠄⠄⠄⠄⠄⠄⠄⠄⠄⠄⠄⠄⠄⠄⠄⠄⠄⠄⠄⠄⠄⠄⠄⠄⠄⠄⠄⠄⠄⠄⠄⠄⠄⠄⠄⠄⠄⠄⠄⠄⠄⠄⠄⠄⠄⠄⠄⠄⠄⠄⠄⠄⠄⠄⠄⠄⠄⠄⠄⠄⠄⠄⠄⠄⠄⠄⠄⠄⠄╎⠄
   // │⠄⠄⠄⠄⠄⠄⠄⡞⠄⠄⠄⠄⠄⠄⠄⠄⠄⠄ ╎⠄⠄⠄⠄⠄⠄⠄⠄⠄⠄⠄⠄⠄⠄⠄⠄⠄⠄⠄⠄⠄⠄⠄⠄⠄⠄⠄⠄⠄⠄⠄⠄⠄⠄⠄⠄⠄⠄⠄⠄⠄⠄⠄⠄⠄⠄⠄⠄⠄⠄⠄⠄⠄⠄⠄⠄⠄⠄⠄⠄⠄⠄⠄⠄⠄⠄⠄⠄⠄⠄⠄⠄⠄⠄⠄⠄⠄⠄╎⠄
   // │⠄⠄⠄⠄⠄⠄⣸⠃⠄⠄⠄⠄⠄⠄⠄⠄⠄⠄ ╎⠄⠄⠄⠄⠄⠄⠄⠄⠄⠄⠄⠄⠄⠄⠄⠄⠄⠄⠄⠄⠄⠄⠄⠄⠄⠄⠄⠄⠄⠄⠄⠄⠄⠄⠄⠄⠄⠄⠄⠄⠄⠄⠄⠄⠄⠄⠄⠄⠄⠄⠄⠄⠄⠄⠄⠄⠄⠄⠄⠄⠄⠄⠄⠄⠄⠄⠄⠄⠄⠄⠄⠄⠄⠄⠄⠄⠄⠄╎⠄
   // │⠄⠄⠄⠄⠄⢰⠇⠄⠄⠄⠄⠄⠄⠄⠄⠄⠄⠄ ╎⠄⠄⠄⠄⠄⠄⠄⠄⠄⠄⠄⠄⠄⠄⠄⠄⠄⠄⠄⠄⠄⠄⠄⠄⠄⠄⠄⠄⠄⠄⠄⠄⠄⠄⠄⠄⠄⠄⠄⠄⠄⠄⠄⠄⠄⠄⠄⠄⠄⠄⠄⠄⠄⠄⠄⠄⠄⠄⠄⠄⠄⠄⠄⠄⠄⠄⠄⠄⠄⠄⠄⠄⠄⠄⠄⠄⠄⠄╎⠄
   // │⠄⠄⠄⠄⢀⡟⠄⠄⠄⠄⠄⠄⠄⠄⠄⠄⠄⠄ ╎⠄⠄⠄⠄⠄⠄⠄⠄⠄⠄⠄⠄⠄⠄⠄⠄⠄⠄⠄⠄⠄⠄⠄⠄⠄⠄⠄⠄⠄⠄⠄⠄⠄⠄⠄⠄⠄⠄⠄⠄⠄⠄⠄⠄⠄⠄⠄⠄⠄⠄⠄⠄⠄⠄⠄⠄⠄⠄⠄⠄⠄⠄⠄⠄⠄⠄⠄⠄⠄⠄⠄⠄⠄⠄⠄⠄⠄⠄╎⠄
   // │⠄⠄⠄⠄⡼⠁⠄⠄⠄⠄⠄⠄⠄⠄⠄⠄⠄⠄ ╎⠄⠄⠄⠄⠄⠄⠄⠄⠄⠄⠄⠄⠄⠄⠄⠄⠄⠄⠄⠄⠄⠄⠄⠄⠄⠄⠄⠄⠄⠄⠄⠄⠄⠄⠄⠄⠄⠄⠄⠄⠄⠄⠄⠄⠄⠄⠄⠄⠄⠄⠄⠄⠄⠄⠄⠄⠄⠄⠄⠄⠄⠄⠄⠄⠄⠄⠄⠄⠄⠄⠄⠄⠄⠄⠄⠄⠄⠄╎⠄
   // │⠄⠄⠄⢰⠇⠄⠄⠄⠄⠄⠄⠄⠄⠄⠄⠄⠄⠄ ╎⠄⠄⠄⠄⠄⠄⠄⠄⠄⠄⠄⠄⠄⠄⠄⠄⠄⠄⠄⠄⠄⠄⠄⠄⠄⠄⠄⠄⠄⠄⠄⠄⠄⠄⠄⠄⠄⠄⠄⠄⠄⠄⠄⠄⠄⠄⠄⠄⠄⠄⠄⠄⠄⠄⠄⠄⠄⠄⠄⠄⠄⠄⠄⠄⠄⠄⠄⠄⠄⠄⠄⠄⠄⠄⠄⠄⠄⠄╎⠄
   // │⠄⠄⢀⡏⠄⠄⠄⠄⠄⠄⠄⠄⠄⠄⠄⠄⠄⠄ ╎⠄⠄⠄⠄⠄⠄⠄⠄⠄⠄⠄⠄⠄⠄⠄⠄⠄⠄⠄⠄⠄⠄⠄⠄⠄⠄⠄⠄⠄⠄⠄⠄⠄⠄⠄⠄⠄⠄⠄⠄⠄⠄⠄⠄⠄⠄⠄⠄⠄⠄⠄⠄⠄⠄⠄⠄⠄⠄⠄⠄⠄⠄⠄⠄⠄⠄⠄⠄⠄⠄⠄⠄⠄⠄⠄⠄⠄⠄╎⠄
   // │⠄⠄⡼⠁⠄⠄⠄⠄⠄⠄⠄⠄⠄⠄⠄⠄⠄⠄ ╎⠄⠄⠄⠄⠄⠄⠄⠄⠄⠄⠄⠄⠄⠄⠄⠄⠄⠄⠄⠄⠄⠄⠄⠄⠄⠄⠄⠄⠄⠄⠄⠄⠄⠄⠄⠄⠄⠄⠄⠄⠄⠄⠄⠄⠄⠄⠄⠄⠄⠄⠄⠄⠄⠄⠄⠄⠄⠄⠄⠄⠄⠄⠄⠄⠄⠄⠄⠄⠄⠄⠄⠄⠄⠄⠄⠄⠄⠄╎⠄
   // │⠄⣸⠃⠄⠄⠄⠄⠄⠄⠄⠄⠄⠄⠄⠄⠄⠄⠄ ╎⠄⠄⠄⠄⠄⠄⠄⠄⠄⠄⠄⠄⠄⠄⠄⠄⠄⠄⠄⠄⠄⠄⠄⠄⠄⠄⠄⠄⠄⠄⠄⠄⠄⠄⠄⠄⠄⠄⠄⠄⠄⠄⠄⠄⠄⠄⠄⠄⠄⠄⠄⠄⠄⠄⠄⠄⠄⠄⠄⠄⠄⠄⠄⠄⠄⠄⠄⠄⠄⠄⠄⠄⠄⠄⠄⠄⠄⠄╎⠄
   // │⡴⠃⠄⠄⠄⠄⠄⠄⠄⠄⠄⠄⠄⠄⠄⠄⠄⠄ ╎⠄⠄⠄⠄⠄⠄⠄⠄⠄⠄⠄⠄⠄⠄⠄⠄⠄⠄⠄⠄⠄⠄⠄⠄⠄⠄⠄⠄⠄⠄⠄⠄⠄⠄⠄⠄⠄⠄⠄⠄⠄⠄⠄⠄⠄⠄⠄⠄⠄⠄⠄⠄⠄⠄⠄⠄⠄⠄⠄⠄⠄⠄⠄⠄⠄⠄⠄⠄⠄⠄⠄⠄⠄⠄⠄⠄⠄⠄╎⠄
   // ┼ ─ ─ ─ ─ ┼ ─ ─ ─ ─ ┼ ─ ─ ─ ─ ┼ ─ ─ ─ ─ ┼ ─ ─ ─ ─ ┼ ─ ─ ─ ─ ┼ ─ ─ ─ ─ ┼ ─ ─ ─ ─ ┼ ─ ─ ─ ─ ┼ ─ ─ ─ ─ ┼
   // 0.0     10       20       30       40       50       60       70       80       90      100 s
   //               τ                                               5τ
   //    Increasing τ gives a slower response.
   // 
   //                1
   //    Initial rate of change = ---   Time to reach 63% of input (X) = τ   Time to reach steady state = 5τ
   //                τ
   // 
   // 
   // RAMP INPUT
   // 
   // │⠄⠄⠄⠄⠄⠄⠄⠄⠄⠄⠄⠄⠄⠄⠄⠄⠄⠄⠄⠄⠄⠄⠄τ = 20s ⠄⠄⠄⠄⠄⠄⠄⠄⠄⠄⠄⠄⠄⠄⠄⠄⠄⠄⠄⠄⠄⠄⠄⠄⠄⠄⠄⠄⠄⠄⠄⠄⠄⠄⠄⠄⠄⠄⠄⠄⠄⠄⠄⠄⠄⠄⠄⠄⠄⠄⠄⠄⠄⠄⠄⠄⠄⠄⠄⠄⠄⠄⠄⠄⠄⠄⠄⠄⢀⡠⠔
   // │⠄⠄⠄⠄⠄⠄⠄⠄⠄⠄⠄⠄⠄⠄⠄⠄⠄⠄⠄⠄⠄⠄⠄⠄⠄⠄⠄⠄⠄⠄⠄⠄⠄⠄⠄⠄⠄⠄⠄⠄⠄⠄⠄⠄⠄⠄⠄⠄⠄⠄⠄⠄⠄⠄⠄⠄⠄⠄⠄⠄⠄⠄⠄⠄⠄⠄⠄⠄⠄⠄⠄⠄⠄⠄⠄⠄⠄⠄⠄⠄⠄⠄⠄⠄⠄⠄⠄⠄⠄⠄⠄⠄⠄⢀⣠⠴⠊⠉⠄⠄
   // │⠄⠄⠄⠄⠄⠄⠄⠄⠄⠄⠄⠄⠄⠄⠄⠄⠄⠄⠄⠄⠄⠄⠄⠄⠄⠄⠄⠄⠄⠄⠄⠄⠄⠄⠄⠄⠄⠄⠄⠄⠄⠄⠄⠄⠄⠄⠄⠄⠄⠄⠄⠄⠄⠄⠄⠄⠄⠄⠄⠄⠄⠄⠄⠄⠄⠄⠄⠄⠄⠄⠄⠄⠄⠄⠄⠄⠄⠄⠄⠄⠄⠄⠄⠄⠄⠄⠄⠄⠄⢀⣀⠴⠊⠉⠄⠄⠄⠄⠄⠄
   // │⠄⠄⠄⠄⠄⠄⠄⠄⠄⠄⠄⠄⠄⠄⠄⠄⠄⠄⠄⠄⠄⠄⠄⠄⠄⠄⠄⠄⠄⠄⠄⠄⠄⠄⠄⠄⠄⠄⠄⠄⠄⠄⠄⠄⠄⠄⠄⠄⠄⠄⠄⠄⠄⠄⠄⠄⠄⠄⠄⠄⠄⠄⠄⠄⠄⠄⠄⠄⠄⠄⠄⠄⠄⠄⠄⠄⠄⠄⠄⠄⠄⠄⠄⠄⠄⠄⣀⡤⠒⠋← ─ INPUT
   // │⠄⠄⠄⠄⠄⠄⠄⠄⠄⠄⠄⠄⠄⠄⠄⠄⠄⠄⠄⠄⠄⠄⠄⠄⠄⠄⠄⠄⠄⠄⠄⠄⠄⠄⠄⠄⠄⠄⠄⠄⠄⠄⠄⠄⠄⠄⠄⠄⠄⠄⠄⠄⠄⠄⠄⠄⠄⠄⠄⠄⠄⠄⠄⠄⠄⠄⠄⠄⠄⠄⠄⠄⠄⠄⠄⠄⠄⠄⠄⠄⠄⠄⢀⡤⠖⠋⠁⠄⠄⠄⠄⠄⠄⠄⠄⠄⠄⠄⠄⠄
   // │⠄⠄⠄⠄⠄⠄⠄⠄⠄⠄⠄⠄⠄⠄⠄⠄⠄⠄⠄⠄⠄⠄⠄⠄⠄⠄⠄⠄⠄⠄⠄⠄⠄⠄⠄⠄⠄⠄⠄⠄⠄⠄⠄⠄⠄⠄⠄⠄⠄⠄⠄⠄⠄⠄⠄⠄⠄⠄⠄⠄⠄⠄⠄⠄⠄⠄⠄⠄⠄⠄⠄⠄⠄⠄⠄⠄⠄⠄⢀⣠⠔⠊⠁⠄⠄⠄⠄⠄⠄⠄⠄⠄⠄⠄⠄⠄⠄⣀⣤⡾
   // │⠄⠄⠄⠄⠄⠄⠄⠄⠄⠄⠄⠄⠄⠄⠄⠄⠄⠄⠄⠄⠄⠄⠄⠄⠄⠄⠄⠄⠄⠄⠄⠄⠄⠄⠄⠄⠄⠄⠄⠄⠄⠄⠄⠄⠄⠄⠄⠄⠄⠄⠄⠄⠄⠄⠄⠄⠄⠄⠄⠄⠄⠄⠄⠄⠄⠄⠄⠄⠄⠄⠄⠄⠄⠄⢀⣠⠔⠚⠁← ─ ─  τ  ─ ─→⢀⣤⡶⠟⠋⠄⠄
   // │⠄⠄⠄⠄⠄⠄⠄⠄⠄⠄⠄⠄⠄⠄⠄⠄⠄⠄⠄⠄⠄⠄⠄⠄⠄⠄⠄⠄⠄⠄⠄⠄⠄⠄⠄⠄⠄⠄⠄⠄⠄⠄⠄⠄⠄⠄⠄⠄⠄⠄⠄⠄⠄⠄⠄⠄⠄⠄⠄⠄⠄⠄⠄⠄⠄⠄⠄⠄⠄⠄⠄⣠⠤⠚⠉⠄⠄⠄⠄⠄⠄⠄⠄⠄⠄⠄⠄⠄⠄⢀⣤⡶⠟⠋⠁⠄⠄⠄⠄⠄
   // │⠄⠄⠄⠄⠄⠄⠄⠄⠄⠄⠄⠄⠄⠄⠄⠄⠄⠄⠄⠄⠄⠄⠄⠄⠄⠄⠄⠄⠄⠄⠄⠄⠄⠄⠄⠄⠄⠄⠄⠄⠄⠄⠄⠄⠄⠄⠄⠄⠄⠄⠄⠄⠄⠄⠄⠄⠄⠄⠄⠄⠄⠄⠄⠄⠄⠄⠄⣀⡤⠒⠉⠄⠄⠄⠄⠄⠄⠄⠄⠄⠄⠄⠄⠄⠄⢀⣠⣴⠞⠋⠁⠄⠄⠄⠄⠄⠄⠄⠄⠄
   // │⠄⠄⠄⠄⠄⠄⠄⠄⠄⠄⠄⠄⠄⠄⠄⠄⠄⠄⠄⠄⠄⠄⠄⠄⠄⠄⠄⠄⠄⠄⠄⠄⠄⠄⠄⠄⠄⠄⠄⠄⠄⠄⠄⠄⠄⠄⠄⠄⠄⠄⠄⠄⠄⠄⠄⠄⠄⠄⠄⠄⠄⠄⠄⣀⡤⠖⠋⠄⠄⠄⠄⠄⠄⠄⠄⠄⠄⠄⠄⠄⠄⢀⣠⣴⠞⠛⠁← ─ OUTPUT
   // │⠄⠄⠄⠄⠄⠄⠄⠄⠄⠄⠄⠄⠄⠄⠄⠄⠄⠄⠄⠄⠄⠄⠄⠄⠄⠄⠄⠄⠄⠄⠄⠄⠄⠄⠄⠄⠄⠄⠄⠄⠄⠄⠄⠄⠄⠄⠄⠄⠄⠄⠄⠄⠄⠄⠄⠄⠄⠄⠄⣀⡠⠴⠊⠁⠄⠄⠄⠄⠄⠄⠄⠄⠄⠄⠄⠄⠄⢀⣀⣤⠶⠛⠉⠄⠄⠄⠄⠄⠄⠄⠄⠄⠄⠄⠄⠄⠄⠄⠄⠄
   // │⠄⠄⠄⠄⠄⠄⠄⠄⠄⠄⠄⠄⠄⠄⠄⠄⠄⠄⠄⠄⠄⠄⠄⠄⠄⠄⠄⠄⠄⠄⠄⠄⠄⠄⠄⠄⠄⠄⠄⠄⠄⠄⠄⠄⠄⠄⠄⠄⠄⠄⠄⠄⠄⠄⠄⢀⣀⠴⠊⠁⠄⠄⠄⠄⠄⠄⠄⠄⠄⠄⠄⠄⠄⠄⣀⣴⠶⠛⠉⠄⠄⠄⠄⠄⠄⠄⠄⠄⠄⠄⠄⠄⠄⠄⠄⠄⠄⠄⠄⠄
   // │⠄⠄⠄⠄⠄⠄⠄⠄⠄⠄⠄⠄⠄⠄⠄⠄⠄⠄⠄⠄⠄⠄⠄⠄⠄⠄⠄⠄⠄⠄⠄⠄⠄⠄⠄⠄⠄⠄⠄⠄⠄⠄⠄⠄⠄⠄⠄⠄⠄⠄⠄⠄⣀⠴⠚⠉⠄⠄⠄⠄⠄⠄⠄⠄⠄⠄⠄⠄⠄⠄⣀⣴⠶⠛⠉⠄⠄⠄⠄⠄⠄⠄⠄⠄⠄⠄⠄⠄⠄⠄⠄⠄⠄⠄⠄⠄⠄⠄⠄⠄
   // │⠄⠄⠄⠄⠄⠄⠄⠄⠄⠄⠄⠄⠄⠄⠄⠄⠄⠄⠄⠄⠄⠄⠄⠄⠄⠄⠄⠄⠄⠄⠄⠄⠄⠄⠄⠄⠄⠄⠄⠄⠄⠄⠄⠄⠄⠄⠄⠄⣀⡤⠒⠉⠁⠄⠄⠄⠄⠄⠄⠄⠄⠄⠄⠄⠄⠄⣀⣤⠶⠟⠉⠁⠄⠄⠄⠄⠄⠄⠄⠄⠄⠄⠄⠄⠄⠄⠄⠄⠄⠄⠄⠄⠄⠄⠄⠄⠄⠄⠄⠄
   // │⠄⠄⠄⠄⠄⠄⠄⠄⠄⠄⠄⠄⠄⠄⠄⠄⠄⠄⠄⠄⠄⠄⠄⠄⠄⠄⠄⠄⠄⠄⠄⠄⠄⠄⠄⠄⠄⠄⠄⠄⠄⠄⠄⠄⣀⡤⠖⠋⠁⠄⠄⠄⠄⠄⠄⠄⠄⠄⠄⠄⠄⠄⣀⣤⡶⠟⠉⠁⠄⠄⠄⠄⠄⠄⠄⠄⠄⠄⠄⠄⠄⠄⠄⠄⠄⠄⠄⠄⠄⠄⠄⠄⠄⠄⠄⠄⠄⠄⠄⠄
   // │⠄⠄⠄⠄⠄⠄⠄⠄⠄⠄⠄⠄⠄⠄⠄⠄⠄⠄⠄⠄⠄⠄⠄⠄⠄⠄⠄⠄⠄⠄⠄⠄⠄⠄⠄⠄⠄⠄⠄⠄⢀⡠⠖⠋⠁⠄⠄⠄⠄⠄⠄⠄⠄⠄⠄⠄⠄⠄⣀⣤⡶⠞⠋⠁⠄⠄⠄⠄⠄⠄⠄⠄⠄⠄⠄⠄⠄⠄⠄⠄⠄⠄⠄⠄⠄⠄⠄⠄⠄⠄⠄⠄⠄⠄⠄⠄⠄⠄⠄⠄
   // │⠄⠄⠄⠄⠄⠄⠄⠄⠄⠄⠄⠄⠄⠄⠄⠄⠄⠄⠄⠄⠄⠄⠄⠄⠄⠄⠄⠄⠄⠄⠄⠄⠄⠄⠄⠄⠄⣠⠖⠊⠉⠄⠄⠄⠄⠄⠄⠄⠄⠄⠄⠄⠄⠄⣀⣤⡶⠟⠉⠁⠄⠄⠄⠄⠄⠄⠄⠄⠄⠄⠄⠄⠄⠄⠄⠄⠄⠄⠄⠄⠄⠄⠄⠄⠄⠄⠄⠄⠄⠄⠄⠄⠄⠄⠄⠄⠄⠄⠄⠄
   // │⠄⠄⠄⠄⠄⠄⠄⠄⠄⠄⠄⠄⠄⠄⠄⠄⠄⠄⠄⠄⠄⠄⠄⠄⠄⠄⠄⠄⠄⠄⠄⠄⠄⣠⠤⠚⠉⠄⠄⠄⠄⠄⠄⠄⠄⠄⠄⠄⠄⠄⢀⣤⡶⠟⠋⠁⠄⠄⠄⠄⠄⠄⠄⠄⠄⠄⠄⠄⠄⠄⠄⠄⠄⠄⠄⠄⠄⠄⠄⠄⠄⠄⠄⠄⠄⠄⠄⠄⠄⠄⠄⠄⠄⠄⠄⠄⠄⠄⠄⠄
   // │⠄⠄⠄⠄⠄⠄⠄⠄⠄⠄⠄⠄⠄⠄⠄⠄⠄⠄⠄⠄⠄⠄⠄⠄⠄⠄⠄⠄⠄⣀⡤⠖⠋⠄⠄⠄⠄⠄⠄⠄⠄⠄⠄⠄⠄⠄⣀⣤⡶⠟⠋⠁⠄⠄⠄⠄⠄⠄⠄⠄⠄⠄⠄⠄⠄⠄⠄⠄⠄⠄⠄⠄⠄⠄⠄⠄⠄⠄⠄⠄⠄⠄⠄⠄⠄⠄⠄⠄⠄⠄⠄⠄⠄⠄⠄⠄⠄⠄⠄⠄
   // │⠄⠄⠄⠄⠄⠄⠄⠄⠄⠄⠄⠄⠄⠄⠄⠄⠄⠄⠄⠄⠄⠄⠄⠄⠄⣀⡤⠖⠋⠄⠄⠄⠄⠄⠄⠄⠄⠄⠄⠄⠄⢀⣠⣤⠾⠛⠉⠄⠄⠄⠄⠄⠄⠄⠄⠄⠄⠄⠄⠄⠄⠄⠄⠄⠄⠄⠄⠄⠄⠄⠄⠄⠄⠄⠄⠄⠄⠄⠄⠄⠄⠄⠄⠄⠄⠄⠄⠄⠄⠄⠄⠄⠄⠄⠄⠄⠄⠄⠄⠄
   // │⠄⠄⠄⠄⠄⠄⠄⠄⠄⠄⠄⠄⠄⠄⠄⠄⠄⠄⠄⠄⠄⢀⣠⠔⠋⠁⠄⠄⠄⠄⠄⠄⠄⠄⠄⠄⠄⢀⣤⡴⠞⠛⠉⠄⠄⠄⠄⠄⠄⠄⠄⠄⠄⠄⠄⠄⠄⠄⠄⠄⠄⠄⠄⠄⠄⠄⠄⠄⠄⠄⠄⠄⠄⠄⠄⠄⠄⠄⠄⠄⠄⠄⠄⠄⠄⠄⠄⠄⠄⠄⠄⠄⠄⠄⠄⠄⠄⠄⠄⠄
   // │⠄⠄⠄⠄⠄⠄⠄⠄⠄⠄⠄⠄⠄⠄⠄⠄⠄⢀⣠⠔⠋⠁⠄⠄⠄⠄⠄⠄⠄⠄⠄⠄⢀⣠⣤⡶⠟⠋⠁⠄⠄⠄⠄⠄⠄⠄⠄⠄⠄⠄⠄⠄⠄⠄⠄⠄⠄⠄⠄⠄⠄⠄⠄⠄⠄⠄⠄⠄⠄⠄⠄⠄⠄⠄⠄⠄⠄⠄⠄⠄⠄⠄⠄⠄⠄⠄⠄⠄⠄⠄⠄⠄⠄⠄⠄⠄⠄⠄⠄⠄
   // │⠄⠄⠄⠄⠄⠄⠄⠄⠄⠄⠄⠄⠄⠄⣠⠴⠚⠉⠄⠄⠄⠄⠄⠄⠄⠄⠄⠄⣀⣤⡶⠞⠛⠉⠄⠄⠄⠄⠄⠄⠄⠄⠄⠄⠄⠄⠄⠄⠄⠄⠄⠄⠄⠄⠄⠄⠄⠄⠄⠄⠄⠄⠄⠄⠄⠄⠄⠄⠄⠄⠄⠄⠄⠄⠄⠄⠄⠄⠄⠄⠄⠄⠄⠄⠄⠄⠄⠄⠄⠄⠄⠄⠄⠄⠄⠄⠄⠄⠄⠄
   // │⠄⠄⠄⠄⠄⠄⠄⠄⠄⠄⣀⠤⠖⠉⠄⠄⠄⠄⠄⠄⠄⠄⢀⣀⣤⡶⠿⠛⠉⠄⠄⠄⠄⠄⠄⠄⠄⠄⠄⠄⠄⠄⠄⠄⠄⠄⠄⠄⠄⠄⠄⠄⠄⠄⠄⠄⠄⠄⠄⠄⠄⠄⠄⠄⠄⠄⠄⠄⠄⠄⠄⠄⠄⠄⠄⠄⠄⠄⠄⠄⠄⠄⠄⠄⠄⠄⠄⠄⠄⠄⠄⠄⠄⠄⠄⠄⠄⠄⠄⠄
   // │⠄⠄⠄⠄⠄⠄⢀⡠⠖⠉⠁⠄⠄⠄⠄⠄⢀⣀⣠⣤⠶⠞⠋⠉⠁⠄⠄⠄⠄⠄⠄⠄⠄⠄⠄⠄⠄⠄⠄⠄⠄⠄⠄⠄⠄⠄⠄⠄⠄⠄⠄⠄⠄⠄⠄⠄⠄⠄⠄⠄⠄⠄⠄⠄⠄⠄⠄⠄⠄⠄⠄⠄⠄⠄⠄⠄⠄⠄⠄⠄⠄⠄⠄⠄⠄⠄⠄⠄⠄⠄⠄⠄⠄⠄⠄⠄⠄⠄⠄⠄
   // │⠄⠄⢀⡠⠖⠊⠁⠄⠄⣀⣀⣠⣤⠶⠶⠛⠋⠉⠉⠄⠄⠄⠄⠄⠄⠄⠄⠄⠄⠄⠄⠄⠄⠄⠄⠄⠄⠄⠄⠄⠄⠄⠄⠄⠄⠄⠄⠄⠄⠄⠄⠄⠄⠄⠄⠄⠄⠄⠄⠄⠄⠄⠄⠄⠄⠄⠄⠄⠄⠄⠄⠄⠄⠄⠄⠄⠄⠄⠄⠄⠄⠄⠄⠄⠄⠄⠄⠄⠄⠄⠄⠄⠄⠄⠄⠄⠄⠄⠄⠄
   // │⠴⠾⠿⠶⠶⠶⠞⠛⠛⠉⠉⠁⠄⠄⠄⠄⠄⠄⠄⠄⠄⠄⠄⠄⠄⠄⠄⠄⠄⠄⠄⠄⠄⠄⠄⠄⠄⠄⠄⠄⠄⠄⠄⠄⠄⠄⠄⠄⠄⠄⠄⠄⠄⠄⠄⠄⠄⠄⠄⠄⠄⠄⠄⠄⠄⠄⠄⠄⠄⠄⠄⠄⠄⠄⠄⠄⠄⠄⠄⠄⠄⠄⠄⠄⠄⠄⠄⠄⠄⠄⠄⠄⠄⠄⠄⠄⠄⠄⠄⠄
   // ┼ ─ ─ ─ ─ ┼ ─ ─ ─ ─ ┼ ─ ─ ─ ─ ┼ ─ ─ ─ ─ ┼ ─ ─ ─ ─ ┼ ─ ─ ─ ─ ┼ ─ ─ ─ ─ ┼ ─ ─ ─ ─ ┼ ─ ─ ─ ─ ┼ ─ ─ ─ ─ ┼
   // 0.0     10       20       30       40       50       60       70       80       90      100 s
   // 
   //    Increasing τ gives a slower response.
   // 
   //    Output follows input with a lag = τ   Time to reach steady state = 5τ
   // 
   // 
   // SINUSOIDAL INPUT
   // 
   // │⠄τ = 10s ⠄⠄⠄⠄⠄⠄⠄⠄⠄⠄⠄⠄⠄⠄⠄⠄⣀⣀⣀⣀⠄← ─ INPUT ⠄⠄⠄⠄⠄⠄⠄⠄⠄⠄⠄⠄⠄⠄⠄⠄⠄⠄⠄⠄⠄⠄⠄⠄⠄⠄⠄⠄⠄⠄⠄⠄⠄⠄⠄⠄⠄⠄⠄⠄⠄⠄⠄⠄⠄⠄⠄⠄⠄⠄⠄⠄⠄⠄⠄⠄⠄⠄⠄⠄⠄⠄⠄
   // │⠄⠄⠄⠄⠄⠄⠄⠄⠄⠄⠄⠄⠄⠄⠄⠄⠄⠄⠄⣠⠔⠚⠉⠄⠄⠄⠈⠉⠒⢤⡀⠄⠄⠄⠄⠄⠄⠄⠄⠄⠄⠄⠄⠄⠄⠄⠄⠄⠄⠄⠄⠄⠄⠄⠄⠄⠄⠄⠄⠄⠄⠄⠄⠄⠄⠄⠄⠄⠄⠄⠄⠄⠄⠄⠄⠄⠄⠄⠄⠄⠄⠄⠄⠄⠄⠄⠄⠄⠄⠄⠄⠄⠄⠄⠄⠄⠄⠄⠄⠄
   // │⠄⠄⠄⠄⠄⠄⠄⠄⠄⠄⠄⠄⠄⠄⠄⠄⠄⣠⠞⠁⠄⠄⠄⠄⠄⠄⠄⠄⠄⠄⠉⠦⡀⠄⠄⠄⠄⠄⠄⠄⠄⠄⠄⠄⠄⠄⠄⠄⠄⠄⠄⠄⠄⠄⠄⠄⠄⠄⠄⠄⠄⠄⠄⠄⠄⠄⠄⠄⠄⠄⠄⠄⠄⠄⠄⠄⠄⠄⠄⠄⠄⠄⠄⠄⠄⠄⠄⠄⠄⠄⠄⠄⠄⠄⠄⠄⠄⠄⠄⠄
   // │⠄⠄⠄⠄⠄⠄⠄⠄⠄⠄⠄⠄⠄⠄⠄⢀⠞⠁⠄⠄⠄⠄⠄⠄⠄⠄⣀⣤⠶⠛⠛⠉⠙⢟⠳⠶⣄⡀⠄⠄⠄⠄⠄⠄⠄⠄⠄⠄⠄⠄⠄⠄⠄⠄⠄⠄⠄⠄⠄⠄⠄⠄⠄⠄⠄⠄⠄⠄⠄⠄⠄⠄⠄⠄⠄⠄⠄⠄⠄⠄⠄⠄⠄⠄⠄⠄⠄⠄⠄⠄⠄⠄⠄⠄⠄⠄⠄⠄⠄⠄
   // │⠄⠄⠄⠄⠄⠄⠄⠄⠄⠄⠄⠄⠄⠄⣠⠋⠄⠄⠄⠄⠄⠄⠄⠄⣠⠾⠋⠄⠄⠄⠄⠄⠄⠄⠳⡀⠈⠙⢶⣄⠄⠄⠄⠄⠄⠄⠄⠄⠄⠄⠄⠄⠄⠄⠄⠄⠄⠄⠄⠄⠄⠄⠄⠄⠄⠄⠄⠄⠄⠄⠄⠄⠄⠄⠄⠄⠄⠄⠄⠄⠄⠄⠄⠄⠄⠄⠄⠄⠄⠄⠄⠄⠄⠄⠄⠄⠄⠄⠄⠄
   // │⠄⠄⠄⠄⠄⠄⠄⠄⠄⠄⠄⠄⢀⡔⠁⠄⠄⠄⠄⠄⠄⠄⣠⠞⠁⠄⠄⠄⠄⠄⠄⠄⠄⠄⠄⠙⣄⠄⠄⠙⢷⣄⠄← ─ OUTPUT  ⠄⠄⠄⠄⠄⠄⠄⠄⠄⠄⠄⠄⠄⠄⠄⠄⠄⠄⠄⠄⠄⠄⠄⠄⠄⠄⠄⠄⠄⠄⠄⠄⠄⠄⠄⠄⠄⠄⠄⠄⠄⠄⠄⠄⠄⠄
   // │⠄⠄⠄⠄⠄⠄⠄⠄⠄⠄⠄⢀⡞⠄⠄⠄⠄⠄⠄⠄⣠⡞⠁⠄⠄⠄⠄⠄⠄⠄⠄⠄⠄⠄⠄⠄⠘⢆⠄⠄⠄⠙⣦⡀⠄⠄⠄⠄⠄⠄⠄⠄⠄⠄⠄⠄⠄⠄⠄⠄⠄⠄⠄⠄⠄⠄⠄⠄⠄⠄⠄⠄⠄⠄⠄⠄⠄⠄⠄⠄⠄⠄⠄⠄⠄⠄⠄⠄⠄⠄⠄⠄⠄⠄⠄⠄⠄⠄⠄⠄
   // │⠄⠄⠄⠄⠄⠄⠄⠄⠄⠄⢀⠞⠄⠄⠄⠄⠄⠄⢀⣼⠋⠄⠄⠄⠄⠄⠄⠄⠄⠄⠄⠄⠄⠄⠄⠄⠄⠈⢦⠄⠄⠄⠈⢳⣄⠄⠄⠄⠄⠄⠄⠄⠄⠄⠄⠄⠄⠄⠄⠄⠄⠄⠄⠄⠄⠄⠄⠄⠄⠄⠄⠄⠄⠄⠄⠄⠄⠄⠄⠄⠄⠄⠄⠄⠄⠄⠄⠄⠄⠄⠄⠄⠄⠄⠄⠄⠄⠄⠄⠄
   // │⠄⠄⠄⠄⠄⠄⠄⠄⠄⢀⡎⠄⠄⠄⠄⠄⠄⢠⡿⠁⠄⠄⠄⠄⠄⠄⠄⠄⠄⠄⠄⠄⠄⠄⠄⠄⠄⠄⠈⢇⠄⠄⠄⠄⠻⣆⠄⠄⠄⠄⠄⠄⠄⠄⠄⠄⠄⠄⠄⠄⠄⠄⠄⠄⠄⠄⠄⠄⠄⠄⠄⠄⠄⠄⠄⠄⠄⠄⠄⠄⠄⠄⠄⠄⠄⠄⠄⠄⠄⠄⠄⠄⠄⠄⠄⠄⠄⠄⠄⠄
   // │⠄⠄⠄⠄⠄⠄⠄⠄⢀⠎⠄⠄⠄⠄⠄⠄⣴⠏⠄⠄⠄⠄⠄⠄⠄⠄⠄⠄⠄⠄⠄⠄⠄⠄⠄⠄⠄⠄⠄⠈⢧⠄⠄⠄⠄⠙⣧⡀⠄⠄⠄⠄⠄⠄⠄⠄⠄⠄⠄⠄⠄⠄⠄⠄⠄⠄⠄⠄⠄⠄⠄⠄⠄⠄⠄⠄⠄⠄⠄⠄⠄⠄⠄⠄⠄⠄⠄⠄⠄⠄⠄⠄⠄⠄⠄⠄⠄⠄⠄⠄
   // │⠄⠄⠄⠄⠄⠄⠄⢀⠞⠄⠄⠄⠄⠄⢀⣼⠃⠄⠄⠄⠄⠄⠄⠄⠄⠄⠄⠄⠄⠄⠄⠄⠄⠄⠄⠄⠄⠄⠄⠄⠈⢧⠄⠄⠄⠄⠘⢷⡀⠄⠄⠄⠄⠄⠄⠄⠄⠄⠄⠄⠄⠄⠄⠄⠄⠄⠄⠄⠄⠄⠄⠄⠄⠄⠄⠄⠄⠄⠄⠄⠄⠄⠄⠄⠄⠄⠄⠄⠄⠄⠄⠄⠄⠄⠄⠄⠄⠄⠄⠄
   // │⠄⠄⠄⠄⠄⠄⢀⡞⠄⠄⠄⠄⠄⢠⡿⠁⠄⠄⠄⠄⠄⠄⠄⠄⠄⠄⠄⠄⠄⠄⠄⠄⠄⠄⠄⠄⠄⠄⠄⠄⠄⠈⢆⠄⠄⠄⠄⠈⢷⡀⠄⠄⠄⠄⠄⠄⠄⠄⠄⠄⠄⠄⠄⠄⠄⠄⠄⠄⠄⠄⠄⠄⠄⠄⠄⠄⠄⠄⠄⠄⠄⠄⠄⠄⠄⠄⠄⠄⠄⠄⠄⠄⠄⠄⠄⠄⠄⠄⠄⠄
   // │⠄⠄⠄⠄⠄⠄⡜⠄⠄⠄⠄⠄⣰⡟⠄⠄⠄⠄⠄⠄⠄⠄⠄⠄⠄⠄⠄⠄⠄⠄⠄⠄⠄⠄⠄⠄⠄⠄⠄⠄⠄⠄⠘⡆⠄⠄⠄⠄⠈⢷⡄⠄⠄⠄⠄⠄⠄⠄⠄⠄⠄⠄⠄⠄⠄⠄⠄⠄⠄⠄⠄⠄⠄⠄⠄⠄⠄⠄⠄⠄⠄⠄⠄⠄⠄⠄⠄⠄⠄⠄⠄⠄⠄⠄⠄⠄⠄⠄⠄⠄
   // │⠄⠄⠄⠄⠄⡼⠁⠄⠄⠄⠄⣴⠏⠄⠄⠄⠄⠄⠄⠄⠄⠄⠄⠄⠄⠄⠄⠄⠄⠄⠄⠄⠄⠄⠄⠄⠄⠄⠄⠄⠄⠄⠄⠘⡄⠄⠄⠄⠄⠈⢻⡀⠄⠄⠄⠄⠄⠄⠄⠄⠄⠄⠄⠄⠄⠄⠄⠄⠄⠄⠄⠄⠄⠄⠄⠄⠄⠄⠄⠄⠄⠄⠄⠄⠄⠄⠄⠄⠄⠄⠄⠄⠄⠄⠄⠄⠄⠄⠄⠄
   // │⠄⠄⠄⠄⡼⠁⠄⠄⠄⢀⡾⠁⠄⠄⠄⠄⠄⠄⠄⠄⠄⠄⠄⠄⠄⠄⠄⠄⠄⠄⠄⠄⠄⠄⠄⠄⠄⠄⠄⠄⠄⠄⠄⠄⠹⡄⠄⠄⠄⠄⠄⢿⡄⠄⠄⠄⠄⠄⠄⠄⠄⠄⠄⠄⠄⠄⠄⠄⠄⠄⠄⠄⠄⠄⠄⠄⠄⠄⠄⠄⠄⠄⠄⠄⠄⠄⠄⠄⠄⠄⠄⠄⠄⠄⠄⠄⠄⠄⠄⠄
   // │⠄⠄⠄⢰⠁⠄⠄⠄⣠⡟⠁⠄⠄⠄⠄⠄⠄⠄⠄⠄⠄⠄⠄⠄⠄⠄⠄⠄⠄⠄⠄⠄⠄⠄⠄⠄⠄⠄⠄⠄⠄⠄⠄⠄⠄⠹⡀⠄⠄⠄⠄⠄⢷⡄⠄⠄⠄⠄⠄⠄⠄⠄⠄⠄⠄⠄⠄⠄⠄⠄⠄⠄⠄⠄⠄⠄⠄⠄⠄⠄⠄⠄⠄⠄⠄⠄⠄⠄⠄⠄⠄⠄⠄⠄⠄⠄⠄⠄⠄⠄
   // │⠄⠄⢠⠇⠄⠄⢀⣰⠟⠄⠄⠄⠄⠄⠄⠄⠄⠄⠄⠄⠄⠄⠄⠄⠄⠄⠄⠄⠄⠄⠄⠄⠄⠄⠄⠄⠄⠄⠄⠄⠄⠄⠄⠄⠄⠄⢳⡀⠄⠄⠄⠄⠈⢷⡀⠄⠄⠄⠄⠄⠄⠄⠄⠄⠄⠄⠄⠄⠄⠄⠄⠄⠄⠄⠄⠄⠄⠄⠄⠄⠄⠄⠄⠄⠄⠄⠄⠄⠄⠄⠄⠄⠄⠄⠄⠄⠄⠄⠄⠄
   // │⠄⢀⠎⠄⠄⣠⡾⠃⠄⠄⠄⠄⠄⠄⠄⠄⠄⠄⠄⠄⠄⠄⠄⠄⠄⠄⠄⠄⠄⠄⠄⠄⠄⠄⠄⠄⠄⠄⠄⠄⠄⠄⠄⠄⠄⠄⠄⢣⠄⠄⠄⠄⠄⠈⢷⡀⠄⠄⠄⠄⠄⠄⠄⠄⠄⠄⠄⠄⠄⠄⠄⠄⠄⠄⠄⠄⠄⠄⠄⠄⠄⠄⠄⠄⠄⠄⠄⠄⠄⠄⠄⠄⠄⠄⠄⠄⠄⠄⠄⠄
   // │⠄⡞⠄⢀⣴⠋⠄⠄⠄⠄⠄⠄⠄⠄⠄⠄⠄⠄⠄⠄⠄⠄⠄⠄⠄⠄⠄⠄⠄⠄⠄⠄⠄⠄⠄⠄⠄⠄⠄⠄⠄⠄⠄⠄⠄⠄⠄⠈⣆⠄⠄⠄⠄⠄⠈⢿⡀⠄⠄⠄⠄⠄⠄⠄⠄⠄⠄⠄⠄⠄⠄⠄⠄⠄⠄⠄⠄⠄⠄⠄⠄⠄⠄⠄⠄⠄⠄⠄⠄⠄⠄⠄⠄⠄⠄⠄⠄⠄⠄⠄
   // │⣜⣠⡾⠋⠄⠄⠄⠄⠄⠄⠄⠄⠄⠄⠄⠄⠄⠄⠄⠄⠄⠄⠄⠄⠄⠄⠄⠄⠄⠄⠄⠄⠄⠄⠄⠄⠄⠄⠄⠄⠄⠄⠄⠄⠄⠄⠄⠄⠘⡆⠄⠄⠄⠄⠄⠈⣷⡀⠄⠄⠄⠄⠄⠄⠄⠄⠄⠄⠄⠄⠄⠄⠄⠄⠄⠄⠄⠄⠄⠄⠄⠄⠄⠄⠄⠄⠄⠄⠄⠄⠄⠄⠄⠄⠄⠄⠄⠄⠄⡼
   // ┼ ─ ─ ─ ─ ┼ ─ ─ ─ ─ ┼ ─ ─ ─ ─ ┼ ─ ─ ─ ─ ┼ ─ ─ ─ ─ ┼─ ─ ─ ─ ┼ ─ ─ ─ ─ ┼ ─ ─ ─ ─ ┼ ─ ─ ─ ─ ┼ ─ ─ ─ ─ 
   // 0.0     10       20       30       40       50       60       70       80       90      100 s
   // │⠄⠄⠄⠄⠄⠄⠄⠄⠄⠄⠄⠄⠄⠄⠄⠄⠄⠄⠄⠄⠄⠄⠄⠄⠄⠄⠄⠄⠄⠄⠄⠄⠄⠄⠄⠄⠄⠄⠄⠄⠄⠄⠄⠄⠄⠄⠄⠄⠄⠄⠄⢧⠄⠄⠄⠄⠄⠄⠘⣧⡀⠄⠄⠄⠄⠄⠄⠄⠄⠄⠄⠄⠄⠄⠄⠄⠄⠄⠄⠄⠄⠄⠄⠄⠄⠄⠄⠄⠄⠄⠄⠄⠄⠄⠄⠄⢠⠏⠄⠄
   // │⠄⠄⠄⠄⠄⠄⠄⠄⠄⠄⠄⠄⠄⠄⠄⠄⠄⠄⠄⠄⠄⠄⠄⠄⠄⠄⠄⠄⠄⠄⠄⠄⠄⠄⠄⠄⠄⠄⠄⠄⠄⠄⠄⠄⠄⠄⠄⠄⠄⠄⠄⠈⢇⠄⠄⠄⠄⠄⠄⠘⣧⠄⠄⠄⠄⠄⠄⠄⠄⠄⠄⠄⠄⠄⠄⠄⠄⠄⠄⠄⠄⠄⠄⠄⠄⠄⠄⠄⠄⠄⠄⠄⠄⠄⠄⠄⡎⠄⠄⠄
   // │⠄⠄⠄⠄⠄⠄⠄⠄⠄⠄⠄⠄⠄⠄⠄⠄⠄⠄⠄⠄⠄⠄⠄⠄⠄⠄⠄⠄⠄⠄⠄⠄⠄⠄⠄⠄⠄⠄⠄⠄⠄⠄⠄⠄⠄⠄⠄⠄⠄⠄⠄⠄⠘⣆⠄⠄⠄⠄⠄⠄⠘⣦⠄⠄⠄⠄⠄⠄⠄⠄⠄⠄⠄⠄⠄⠄⠄⠄⠄⠄⠄⠄⠄⠄⠄⠄⠄⠄⠄⠄⠄⠄⠄⠄⠄⡞⠄⠄⠄⠄
   // │⠄⠄⠄⠄⠄⠄⠄⠄⠄⠄⠄⠄⠄⠄⠄⠄⠄⠄⠄⠄⠄⠄⠄⠄⠄⠄⠄⠄⠄⠄⠄⠄⠄⠄⠄⠄⠄⠄⠄⠄⠄⠄⠄⠄⠄⠄⠄⠄⠄⠄⠄⠄⠄⠘⡄⠄⠄⠄⠄⠄⠄⠙⣇⠄⠄⠄⠄⠄⠄⠄⠄⠄⠄⠄⠄⠄⠄⠄⠄⠄⠄⠄⠄⠄⠄⠄⠄⠄⠄⠄⠄⠄⠄⠄⡼⠄⠄⠄⠄⠄
   // │⠄⠄⠄⠄⠄⠄⠄⠄⠄⠄⠄⠄⠄⠄⠄⠄⠄⠄⠄⠄⠄⠄⠄⠄⠄⠄⠄⠄⠄⠄⠄⠄⠄⠄⠄⠄⠄⠄⠄⠄⠄⠄⠄⠄⠄⠄⠄⠄⠄⠄⠄⠄⠄⠄⠹⡀⠄⠄⠄⠄⠄⠄⠸⣧⠄⠄⠄⠄⠄⠄⠄⠄⠄⠄⠄⠄⠄⠄⠄⠄⠄⠄⠄⠄⠄⠄⠄⠄⠄⠄⠄⠄⠄⣰⠁⠄⠄⠄⠄⢠
   // │⠄⠄⠄⠄⠄⠄⠄⠄⠄⠄⠄⠄⠄⠄⠄⠄⠄⠄⠄⠄⠄⠄⠄⠄⠄⠄⠄⠄⠄⠄⠄⠄⠄⠄⠄⠄⠄⠄⠄⠄⠄⠄⠄⠄⠄⠄⠄⠄⠄⠄⠄⠄⠄⠄⠄⠹⡀⠄⠄⠄⠄⠄⠄⠘⣧⠄⠄⠄⠄⠄⠄⠄⠄⠄⠄⠄⠄⠄⠄⠄⠄⠄⠄⠄⠄⠄⠄⠄⠄⠄⠄⠄⢰⠃⠄⠄⠄⠄⢀⡿
   // │⠄⠄⠄⠄⠄⠄⠄⠄⠄⠄⠄⠄⠄⠄⠄⠄⠄⠄⠄⠄⠄⠄⠄⠄⠄⠄⠄⠄⠄⠄⠄⠄⠄⠄⠄⠄⠄⠄⠄⠄⠄⠄⠄⠄⠄⠄⠄⠄⠄⠄⠄⠄⠄⠄⠄⠄⢳⡀⠄⠄⠄⠄⠄⠄⠙⣧⡀⠄⠄⠄⠄⠄⠄⠄⠄⠄⠄⠄⠄⠄⠄⠄⠄⠄⠄⠄⠄⠄⠄⠄⠄⣠⠃⠄⠄⠄⠄⢠⡿⠁
   // │⠄⠄⠄⠄⠄⠄⠄⠄⠄⠄⠄⠄⠄⠄⠄⠄⠄⠄⠄⠄⠄⠄⠄⠄⠄⠄⠄⠄⠄⠄⠄⠄⠄⠄⠄⠄⠄⠄⠄⠄⠄⠄⠄⠄⠄⠄⠄⠄⠄⠄⠄⠄⠄⠄⠄⠄⠄⢳⠄⠄⠄⠄⠄⠄⠄⠘⢷⡀⠄⠄⠄⠄⠄⠄⠄⠄⠄⠄⠄⠄⠄⠄⠄⠄⠄⠄⠄⠄⠄⠄⢠⠃⠄⠄⠄⠄⢰⡟⠄⠄
   // │⠄⠄⠄⠄⠄⠄⠄⠄⠄⠄⠄⠄⠄⠄⠄⠄⠄⠄⠄⠄⠄⠄⠄⠄⠄⠄⠄⠄⠄⠄⠄⠄⠄⠄⠄⠄⠄⠄⠄⠄⠄⠄⠄⠄⠄⠄⠄⠄⠄⠄⠄⠄⠄⠄⠄⠄⠄⠄⢳⠄⠄⠄⠄⠄⠄⠄⠈⢳⡄⠄⠄⠄⠄⠄⠄⠄⠄⠄⠄⠄⠄⠄⠄⠄⠄⠄⠄⠄⠄⢠⠎⠄⠄⠄⠄⣰⠏⠄⠄⠄
   // │⠄⠄⠄⠄⠄⠄⠄⠄⠄⠄⠄⠄⠄⠄⠄⠄⠄⠄⠄⠄⠄⠄⠄⠄⠄⠄⠄⠄⠄⠄⠄⠄⠄⠄⠄⠄⠄⠄⠄⠄⠄⠄⠄⠄⠄⠄⠄⠄⠄⠄⠄⠄⠄⠄⠄⠄⠄⠄⠄⢣⠄⠄⠄⠄⠄⠄⠄⠄⢿⡄⠄⠄⠄⠄⠄⠄⠄⠄⠄⠄⠄⠄⠄⠄⠄⠄⠄⠄⢀⠏⠄⠄⠄⢀⣴⠋⠄⠄⠄⠄
   // │⠄⠄⠄⠄⠄⠄⠄⠄⠄⠄⠄⠄⠄⠄⠄⠄⠄⠄⠄⠄⠄⠄⠄⠄⠄⠄⠄⠄⠄⠄⠄⠄⠄⠄⠄⠄⠄⠄⠄⠄⠄⠄⠄⠄⠄⠄⠄⠄⠄⠄⠄⠄⠄⠄⠄⠄⠄⠄⠄⠄⢣←--   τ   -→⠹⣦⠄⠄⠄⠄⠄⠄⠄⠄⠄⠄⠄⠄⠄⠄⠄⠄⢠⠋⠄⠄⠄⢠⡾⠁⠄⠄⠄⠄⠄
   // │⠄⠄⠄⠄⠄⠄⠄⠄⠄⠄⠄⠄⠄⠄⠄⠄⠄⠄⠄⠄⠄⠄⠄⠄⠄⠄⠄⠄⠄⠄⠄⠄⠄⠄⠄⠄⠄⠄⠄⠄⠄⠄⠄⠄⠄⠄⠄⠄⠄⠄⠄⠄⠄⠄⠄⠄⠄⠄⠄⠄⠄⠳⡀⠄⠄⠄⠄⠄⠄⠄⠈⢷⡄⠄⠄⠄⠄⠄⠄⠄⠄⠄⠄⠄⠄⠄⢠⠃⠄⠄⠄⣴⠏⠄⠄⠄⠄⠄⠄⠄
   // │⠄⠄⠄⠄⠄⠄⠄⠄⠄⠄⠄⠄⠄⠄⠄⠄⠄⠄⠄⠄⠄⠄⠄⠄⠄⠄⠄⠄⠄⠄⠄⠄⠄⠄⠄⠄⠄⠄⠄⠄⠄⠄⠄⠄⠄⠄⠄⠄⠄⠄⠄⠄⠄⠄⠄⠄⠄⠄⠄⠄⠄⠄⠱⡄⠄⠄⠄⠄⠄⠄⠄⠄⠹⢦⣀⠄⠄⠄⠄⠄⠄⠄⠄⠄⠄⡠⠃⠄⠄⣠⠞⠁⠄⠄⠄⠄⠄⠄⠄⠄
   // │⠄⠄⠄⠄⠄⠄⠄⠄⠄⠄⠄⠄⠄⠄⠄⠄⠄⠄⠄⠄⠄⠄⠄⠄⠄⠄⠄⠄⠄⠄⠄⠄⠄⠄⠄⠄⠄⠄⠄⠄⠄⠄⠄⠄⠄⠄⠄⠄⠄⠄⠄⠄⠄⠄⠄⠄⠄⠄⠄⠄⠄⠄⠄⠙⣄⠄⠄⠄⠄⠄⠄⠄⠄⠈⠙⢶⣄⠄⠄⠄⠄⠄⠄⢀⡔⠁⢀⣠⠞⠁⠄⠄⠄⠄⠄⠄⠄⠄⠄⠄
   // │⠄⠄⠄⠄⠄⠄⠄⠄⠄⠄⠄⠄⠄⠄⠄⠄⠄⠄⠄⠄⠄⠄⠄⠄⠄⠄⠄⠄⠄⠄⠄⠄⠄⠄⠄⠄⠄⠄⠄⠄⠄⠄⠄⠄⠄⠄⠄⠄⠄⠄⠄⠄⠄⠄⠄⠄⠄⠄⠄⠄⠄⠄⠄⠄⠈⠳⡀⠄⠄⠄⠄⠄⠄⠄⠄⠄⠉⠻⠶⣤⣄⣀⣠⣮⡴⠶⠋⠁⠄⠄⠄⠄⠄⠄⠄⠄⠄⠄⠄⠄
   // │⠄⠄⠄⠄⠄⠄⠄⠄⠄⠄⠄⠄⠄⠄⠄⠄⠄⠄⠄⠄⠄⠄⠄⠄⠄⠄⠄⠄⠄⠄⠄⠄⠄⠄⠄⠄⠄⠄⠄⠄⠄⠄⠄⠄⠄⠄⠄⠄⠄⠄⠄⠄⠄⠄⠄⠄⠄⠄⠄⠄⠄⠄⠄⠄⠄⠄⠙⢆⡀⠄⠄⠄⠄⠄⠄⠄⠄⠄⠄⠄⢀⠞⠉⠄⠄⠄⠄⠄⠄⠄⠄⠄⠄⠄⠄⠄⠄⠄⠄⠄
   // │⠄⠄⠄⠄⠄⠄⠄⠄⠄⠄⠄⠄⠄⠄⠄⠄⠄⠄⠄⠄⠄⠄⠄⠄⠄⠄⠄⠄⠄⠄⠄⠄⠄⠄⠄⠄⠄⠄⠄⠄⠄⠄⠄⠄⠄⠄⠄⠄⠄⠄⠄⠄⠄⠄⠄⠄⠄⠄⠄⠄⠄⠄⠄⠄⠄⠄⠄⠄⠙⠢⣄⠄⠄⠄⠄⠄⠄⢀⡠⠞⠁⠄⠄⠄⠄⠄⠄⠄⠄⠄⠄⠄⠄⠄⠄⠄⠄⠄⠄⠄
   // │⠄⠄⠄⠄⠄⠄⠄⠄⠄⠄⠄⠄⠄⠄⠄⠄⠄⠄⠄⠄⠄⠄⠄⠄⠄⠄⠄⠄⠄⠄⠄⠄⠄⠄⠄⠄⠄⠄⠄⠄⠄⠄⠄⠄⠄⠄⠄⠄⠄⠄⠄⠄⠄⠄⠄⠄⠄⠄⠄⠄⠄⠄⠄⠄⠄⠄⠄⠄⠄⠄⠄⠉⠓⠒⠒⠒⠋⠁⠄⠄⠄⠄⠄⠄⠄⠄⠄⠄⠄⠄⠄⠄⠄⠄⠄⠄⠄⠄⠄⠄
   // 
   //    Increasing τ gives a slower response.
   // 
   //    Output follows input with a lag = τ   Time to reach steady state = 5τ
   // 
   // 
   // 
   // ▂▂▂▂▂▂▂▂▂▂▂▂▂▂▂▂▂▂▂▂▂▂▂▂▂▂▂▂▂▂▂▂▂▂▂▂▂▂▂▂▂▂▂▂
   // 2.5      Operating modes
   // 
   // 
   // The block supports two modes of operation:
   // 
   //    •   Automatic mode:
   //      The module automatically calculates the elapsed time since the simulation started 
   //      and generates the appropriate output value for any form of input.
   // 
   //      Automatic mode can accommodate any form of input (step, ramp, sinusoid, 
   //      freeform &c.).
   // 
   //    •   Manual mode:
   //      The current elapsed time and fixed input value is supplied manually to the module; 
   //      the module will then calculate the output value based on a step input at this input 
   //      value and at this time value.
   // 
   //      Manual mode only supports a step form of input (the input is considered to be a step 
   //      input that changed to the manually specified input value at time = 0, and that prior to 
   //      this the input was zero. I.e. a step input that changed from zero to the specified value 
   //      at time = 0).
   // 
   // 
   //                ━━━   ⬙⬙⬙⬙⬙⬙   ━━━
END_REGION

REGION Network 2: Block description — Section 3
   // ▄▄▄▄▄▄▄▄▄▄▄▄▄▄▄▄▄▄▄▄▄▄▄▄▄▄▄▄▄▄▄▄▄▄▄▄▄▄▄▄▄▄▄▄
   // 3.     DETAILED BLOCK DESCRIPTION
   // 
   // 
   // This module, FC19511_StdDebugInst1Order uses user data types to provide the primary 
   // interface to the block. There are four formal parameters:
   // 
   //  ――――――――――――――――――――――――――――――――――――――――――
   //  PARAM         FUNCTION                    TYPE      IN-OUT 
   //  ――――――――――――――――――――――――――――――――――――――――――
   //  SYS_SIGNALS      Common system signals              UT21000    In
   //           logic and timing signals for parametric access
   // 
   //  TRIGGER       Activates the simulation (the simulation will run     Bool      In
   //           whilever this signal is high), the elapsed time 
   //           is measured from the rising edge of this signal
   // 
   //  INPUT        The input time function, x(t) in the calculations     Real      In
   // 
   //  DYNAMIC_DATA      Data structure that holds the live data for the       UT39512    InOut
   //           simulation (damping factor, natural frequency, 
   //           system gain, elapsed time &c.)
   // 
   //  OUTPUT       The output time response, y(t) in the calculations   Real      Out
   //  ――――――――――――――――――――――――――――――――――――――――――
   // 
   // The DYNAMIC_DATA parameter is a UDT that holds all the data for the simulation.
   // 
   //  ――――――――――――――――――――――――――――――――――――――――――
   //  PARAM         ASSOCIATED UDT          ASSOCIATED DATA BLOCK
   //  ――――――――――――――――――――――――――――――――――――――――――
   //  DYNAMIC_DATA   UT39511_Dy_DebugInst1Order      DB39511_Dy_DebugInst1Order
   //  ――――――――――――――――――――――――――――――――――――――――――
   // 
   // 
   // Section 6 contains a full list of all variables within these UDTs.
   // 
   // 
   // 
   // ▂▂▂▂▂▂▂▂▂▂▂▂▂▂▂▂▂▂▂▂▂▂▂▂▂▂▂▂▂▂▂▂▂▂▂▂▂▂▂▂▂▂▂▂
   // 3.1      The primary simulation signals
   // 
   // 
   // The simulation is based upon various signals passed to the module and the elapsed time since 
   // the simulation started:
   // 
   //  ――――――――――――――――――――――――――――――――――――――――――
   //  SIGNAL         FUNCTION               RANGE       ACCESSED VIA
   //  ――――――――――――――――――――――――――――――――――――――――――
   //  INPUT         The INPUT parameter is the x value    Unrestricted     Parameter 
   //            in the calculations of § 3.2
   // 	
   //  OUTPUT        The OUTPUT parameter is the y value   Unrestricted     Parameter 
   //            in the calculations of § 3.2
   // 
   //  TRIGGER        The TRIGGER parameter activates      0 or 1     Parameter
   //            the simulation
   // 
   //  k_Gain          The system gain (K) term         Unrestricted     UT39511
   //            in the calculations of § 3.2       typ. 1-10
   // 
   //  k_TimeConstant     The system time constant (τ) term in   +ve number      UT39511
   //            the calculations of § 3.2.
   //            In units of seconds (s)
   // 
   //  actual_PrevOutput   The resulting output calculated in the  Unrestricted     UT39511
   //            previous iteration of the calculation
   // 
   //  actual_StartTime   The CPU time when the simulation    DTL value    UT39511
   //            started (rising edge of TRIGGER)      of RTC
   // 
   //  actual_Time      The current CPU time, for the current    DTL value    UT39511
   //            iteration of the calculation         of RTC
   //            (time at y[n])
   // 
   //  actual_PrevTime    The CPU time of the last iteration    DTL value    UT39511
   //            of the calculation              of RTC
   //            (time at y[n-1])
   // 
   //  actual_RunTime     The elapsed time of the simulation      +ve number      UT39511
   //            in seconds (s)              calculated by
   //                              the module
   // 
   //  actual_DeltaTime     Time between the current iteration      +ve number      UT39511
   //            and the previous iteration, Δt in the     calculated by 
   //            calculations:             the module
   //            = actual_Time – actual_PrevTime
   //            In units of seconds (s)
   //  ――――――――――――――――――――――――――――――――――――――――――
   // 
   // 
   // The system time constant (k_TimeConstant), determines the lag of the system, the higher the 
   // value, the slower the response.
   // 
   // The system gain (k_Gain), is simply a common multiplier that amplifies the output response. 
   // By default the system gain is set to a value of one (i.e. unity gain).
   // 
   // The elapsed time actual_RunTime is calculated from the real time clock within the CPU. On the 
   // rising edge of the TRIGGER parameter, the CPU real time clock is read and the value stored in 
   // the variable actual_StartTime, on each subsequent call to the block, the real time clock is 
   // once again read and stored in the variable actual_Time. The elapsed time is calculated by 
   // subtracting the actual_StartTime value from the actual_Time value and converting the result 
   // to seconds this is then stored as the actual_RunTime value.
   // 
   // The TRIGGER signal is simply used to start and stop the simulation. A rising edge on the 
   // TRIGGER signal causes the current CPU time to be stored (actual_StartTime) and sets the 
   // elapsed time to zero (actual_RunTime). The simulation will run whilever the TRIGGER signal is 
   // high (has a value of 1), each time the module is called, the elapsed time (actual_RunTime) is 
   // updated (see the previous paragraph) and the output calculated accordingly.
   // 
   // If the simulation is active (the TRIGGER signal is high, has a value of 1) the time between the 
   // current module call (actual_Time) and the previous module call (actual_PrevTime) is calculated 
   // and stored in the variable actual_DeltaTime (∆t in the calculations), this is calculated as follows:
   // 
   //      actual_DeltaTime= actual_Time-actual_PrevTime
   // 
   // At the end of the current module call, the actual_PrevTime is set to the actual_Time, for the 
   // next iteration of the calculation.
   // 
   // At the end of the current module call, the actual_PrevOutput is set to the OUTPUT, value for the 
   // next iteration of the calculation.
   // 
   // If the TRIGGER signal is low (0), the simulation is instantly stopped and the OUTPUT parameter is 
   // set to zero.
   // 
   // 
   // 
   // ▂▂▂▂▂▂▂▂▂▂▂▂▂▂▂▂▂▂▂▂▂▂▂▂▂▂▂▂▂▂▂▂▂▂▂▂▂▂▂▂▂▂▂▂
   // 3.2      The response calculation
   // 
   // 
   // Two forms of calculation are carried out by the module, the first is the iterative, real-time 
   // calculation for the automatic response, this is given in equation (2.2). The second is the discrete 
   // manual response calculation given in equation (2.3). These are reproduced below.
   // 
   // The calculations below use Greek characters for the main variables, the calculations use various 
   // parameters and UDT variables that have plain English names, The association between these 
   // variables and the Greek nomenclature is given below.
   // 
   // 
   // ――――――――――――――――――――――――――――――――――――――――――――――――
   // REAL-TIME AUTOMATIC SIMULATION         from equation 2.2
   // 
   //    y[n] = Ka x[n]  ┼ (1-a) y[n-1]  (3.1)
   // 
   //              ΔT
   //    where:   a = ----------
   //            τ+ΔT
   // ――――――――――――――――――――――――――――――――――――――――――――――――
   // DISCRETE MANUAL RESPONSE TO A STEP INPUT      from equation 2.3
   // 
   //          ┌      -t/τ  ┐
   //    y(t) = KX│ 1 ─  e   │    (3.2)
   //          └       ┘
   // ――――――――――――――――――――――――――――――――――――――――――――――――
   // Where:    K      is the system gain (a constant number)             k_Gain
   //      τ      is the system time constant (in seconds)             k_TimeConstant
   //      Δt    is the sampling interval between calculations (in seconds)  actual_DeltaTime
   //      X/x[n] is the input at the current iteration or in manual mode    parameter INPUT
   //      y/y[n]  is the output at the current iteration or in manual mode    parameter OUTPUT
   //      y[n-1] is the output at the previous iteration             actual_PrevOutput
   // 
   // Note:    If the system gain k_Gain is set zero, the OUTPUT will be zero under all circumstances.
   // 
   // Each of these calculations can be accommodated with the mathematical functions available to a 
   // Siemens Controller, see § 3.4.
   // 
   // 
   // 
   // 
   // ▂▂▂▂▂▂▂▂▂▂▂▂▂▂▂▂▂▂▂▂▂▂▂▂▂▂▂▂▂▂▂▂▂▂▂▂▂▂▂▂▂▂▂▂
   // 3.3      Status and informative signals
   // 
   // 
   // The module produces various status signals that reflect the nature of the simulation:
   // 
   //  DATA STRUCTURE      UT39511_Dy_DebugInst1Order
   //  ――――――――――――――――――――――――――――――――――――――――――
   //  SIGNAL           FUNCTION            TYPE   DETAILS
   //  ――――――――――――――――――――――――――――――――――――――――――
   //  status_Running        The simulation is running     Bool    1 = Simulation is running 
   //                               0 = Simulation is stopped
   // 
   //  status_Stopped       The simulation is stopped    Bool    1 = Simulation is stopped 
   //                               0 = Simulation is running
   // 
   //  status_SteadyState      Simulation has achieved   Bool    1 = Stady state achieved
   //                 steady state ±2%           0 = Not in steady state
   // 
   //  cal_TimeSteady       Time to reach steady state      Real Seconds
   // 
   // 
   //  ――――――――――――――――――――――――――――――――――――――――――
   // 
   // The status_Running and status_Stopped are determined purely by the status of the TRIGGER 
   // parameter, if this is set high (1), status_Running will be high and status_Stopped low. If  TRIGGER 
   // parameter, if this is set low (0), status_Running will be low and status_Stopped high. The 
   // status_Running and status_Stopped signals are always the inverse of each other.
   // 
   // If the simulation has reached a steady state, i.e. the non-linear relationship between the output 
   // and the input that occurs at the start of the simulation has concluded, the status_SteadyState 
   // signal will be set high (1), it will be low (0) until the steady state conditions are achieved 
   // (typically, this is at 5×τ seconds after the start of the simulation).
   // 
   // In addition, the variable cal_TimeSteady give the time at which the steady state will be reached 
   // (in seconds), this is true for all forms of input.
   // 
   // 
   // 
   // ▂▂▂▂▂▂▂▂▂▂▂▂▂▂▂▂▂▂▂▂▂▂▂▂▂▂▂▂▂▂▂▂▂▂▂▂▂▂▂▂▂▂▂▂
   // 3.4     Expressing the calculations in Controller operations
   // 
   // The calculations above must be rendered in a form suitable for the Simatic S7-1500 Controller, 
   // using the mathematical operations available to that Controller, these are listed in Table 2.1.
   // 
   // To perform the calculations in the Controller it will be necessary to use partial calculation to 
   // hold separate components of the overall calculation and combine these to produce the final 
   // result. 
   // 
   // The following sections breakdown each of the response calculations into these partial 
   // calculations and demonstrate how these are then combined to provide a final result that is 
   // compatible with the Controller mathematical operations and Controller notations.
   // 
   // 
   // 
   // ▁▁▁▁▁▁▁▁▁▁▁▁▁▁▁▁▁▁▁▁▁▁▁▁▁▁▁▁▁▁▁▁▁▁▁▁▁▁▁▁▁▁▁▁
   // 3.4.1     Real-time simulation calculation
   // 
   // 
   // CALCULATION:
   //                               ΔT
   //    y[n] = Ka x[n]  ┼ (1-a) y[n-1]   where: a = ----------
   //                             τ+ΔT
   // 
   // Is rendered into the correct format as follows:
   // 
   // 
   //  cal_01 = ΔT             =  actual_Time - actual_PrevTime
   // 
   //  cal_02 = τ + ΔT             = k_TimeConstant + cal_01
   // 
   //                ΔT
   //  cal_03 = a = ----------          = cal_01 ÷ cal_02
   //                 τ+ΔT
   // 
   //  cal_04 = 1 - a             = 1 - cal_03
   // 
   // 
   //  cal_05 = Kax[n]            = k_Gain × cal_03 × INPUT
   // 
   //  cal_06 = (1-a) y[n-1]          = cal_04 × actual_PrevOutput
   // 
   // 
   //  OUTPUT  = Ka x[n]  ┼ (1-a) y[n-1]      = cal_05 × cal_06
   // 
   // 
   // 
   // ▁▁▁▁▁▁▁▁▁▁▁▁▁▁▁▁▁▁▁▁▁▁▁▁▁▁▁▁▁▁▁▁▁▁▁▁▁▁▁▁▁▁▁▁
   // 3.4.2     Discrete manual response to a step input
   // 
   // 
   // CALCULATION:
   // 
   //          ┌      -t/τ  ┐
   //    y(t) = KX│ 1 ─  e   │
   //          └       ┘
   // 
   // 
   // Is rendered into the correct format as follows:
   // 
   // 
   //  cal_01 =  t/τ             = - 1 × actual_RunTime ÷  k_TimeConstant
   // 
   //          - t/τ
   //  cal_02 = ｅ              = EXP (cal_01)
   // 
   //                - t/τ
   //  cal_03 = 1 ─  ｅ              = 1 - cal_02
   // 
   // 
   //              ┌      -t/τ  ┐
   //  OUTPUT  = KX│ 1 ─  e   │       = k_Gain × INPUT × cal_03
   //              └       ┘
   // 
   // 
   // 
   // ▂▂▂▂▂▂▂▂▂▂▂▂▂▂▂▂▂▂▂▂▂▂▂▂▂▂▂▂▂▂▂▂▂▂▂▂▂▂▂▂▂▂▂▂
   // 3.5     Operating modes
   // 
   // 
   // This block FC19511_StdDebugInst1Order supports manual and automatic operating modes, the 
   // default mode is automatic.
   // 
   // The module can be switched between automatic and manual modes with the 
   // mode_AutMan signal:
   // 
   //  DATA STRUCTURE    UT39511_Dy_DebugInst1Order
   //  ――――――――――――――――――――――――――――――――――――――――――
   //  SIGNAL         FUNCTION               TYPE     DETAILS
   //  ――――――――――――――――――――――――――――――――――――――――――
   //  Mode_AutMan     Specifies the operating mode of     Bool  1 = automatic mode
   //            the simulation                 0 = manual mode
   // 
   //  Mode_ManTime     Specifies the manual time value of       Real     Elapsed time
   //            the simulation in seconds           in seconds
   // 
   //  status_Aut      The simulation is in automatic mode   Bool  1 = auto mode
   //                                  0 = not in auto
   // 
   //  status_Man       The simulation is in manual mode    Bool  1 = manual mode
   //                                  0 = not in manual
   //  ――――――――――――――――――――――――――――――――――――――――――  
   // 
   // 
   // 
   // ▁▁▁▁▁▁▁▁▁▁▁▁▁▁▁▁▁▁▁▁▁▁▁▁▁▁▁▁▁▁▁▁▁▁▁▁▁▁▁▁▁▁▁▁
   // 3.5.1    Automatic mode
   // 
   // 
   // By default the module will be in automatic mode. 
   // 
   // In automatic mode, if the simulation is active (TRIGGER = 1), the module carries out the real-time 
   // calculation given in § 3.4.1. 
   // 
   // In automatic mode, a real time simulation occurs, generating responses similar to those shown 
   // in the plots of § 2.4 (depending on the nature of the input).
   //  
   // 
   // 
   // 
   // ▁▁▁▁▁▁▁▁▁▁▁▁▁▁▁▁▁▁▁▁▁▁▁▁▁▁▁▁▁▁▁▁▁▁▁▁▁▁▁▁▁▁▁▁
   // 3.5.2    Manual mode
   // 
   // 
   // In manual mode, if the simulation is active (TRIGGER = 1), the module carries out the discrete 
   // response to a step input calculation given in § 3.4.2. 
   // 
   // The difference with manual mode, is that the time used in the calculation must be uniquely 
   // specified; a manual time value must be provided.
   // 
   // The manual time is given in the variable mode_ManTime and is specified in seconds.
   // 
   // If mode mode_ManTime remains constant between module calls, the module will return the 
   // same OUTPUT value each time (assuming all other signals remain unchanged).
   // 
   // The manual mode response is that of a step input, the value of the INPUT parameter is taken as 
   // the starting value of the step at time = 0.
   // 
   // 
   //                ━━━   ⬙⬙⬙⬙⬙⬙   ━━━
END_REGION

